   // sequencer 5: S400-S499 Robot3 FixtureCode reading
   STEP Robot3FixtrueScanStart:   // S400, max time T#10S, warning time T#7S
              N    "AutoProcessData".GripperCode_R3[1]:=''
              N    "AutoProcessData".GripperCode_R3[2]:=''
              N    "AutoProcessData".GripperCode_R3[3]:=''
              N    "AutoProcessData".GripperCode_R3[4]:=''
              N    "AutoProcessData".FixtureCode_A2[1]:=''
              N    "AutoProcessData".FixtureCode_A2[2]:=''
              N    "AutoProcessData".FixtureCode_A2[3]:=''
              N    "AutoProcessData".FixtureCode_A2[4]:=''
              N    "AutoProcessData".FixtureCode_A2[5]:=''
              N    "AutoProcessData".FixtureCode_A2[6]:=''
              N    "AutoProcessData".FixtureCode_A2[7]:=''
              N    "AutoProcessData".FixtureCode_A2[8]:=''
   END_STEP
   TRANSITION Trans400 FROM Robot3FixtrueScanStart TO Robot3CheckScanStatus   // T400
      := NOT "KukaRobot2_CtrlDB".sROBtoPLC.User.Cycle.DO297_MaintainInside;
   END_TRANSITION
   STEP AllScanFinish:   // S408, max time T#10S, warning time T#7S
   END_STEP
   TRANSITION Trans403 FROM AllScanFinish TO ProcessStart   // T403, jump
      := "AutoProcessData".GlobalData.Table1CodeOKFlag AND "AutoProcessData".GlobalData.Table2CodeOKFlag AND "AutoProcessData".GlobalData.Robot1GripperCodeOKFlag AND "AutoProcessData".GlobalData.Robot2GripperCodeOKFlag AND "AutoProcessData".GlobalData.Robot3GripperCodeOKFlag AND "AutoProcessData".GlobalData.Fixture1CodeOKFlag AND "AutoProcessData".GlobalData.Fixture2CodeOKFlag AND "ST10_RecipeDB".Recipe.Equal AND NOT "ChangeOver_DB".Global.ScanFixtureFlag AND NOT "ChangeOver_DB".Global.ChangeOverRequest;
   END_TRANSITION
   TRANSITION Trans420 FROM AllScanFinish TO ProcessStart   // T420, jump
      := ("ChangeOver_DB".Global.ChangeOverRequest OR "ChangeOver_DB".Global.ChangeOverSelected) AND NOT "ChangeOver_DB".Global.ChangeOverSelected;
   END_TRANSITION
   STEP DataMove_7:   // S279, max time T#10S, warning time T#7S
              N    "AutoProcessData".FixtureCode_A2[2]:="KeyenceSR1000Ctrl_807A1DB".sHMI.Status.CurrentCode
   END_STEP
   TRANSITION Trans336 FROM DataMove_7 TO WaitRobotScanPos3Reach_1   // T312
      := "AlwaysTRUE";
   END_TRANSITION
   STEP Robot3StartToMaintenance:   // S409, max time T#10S, warning time T#7S
   END_STEP
   TRANSITION Trans405 FROM Robot3StartToMaintenance TO Step712   // T405, jump
      := TRUE;
   END_TRANSITION
   STEP DataMove_8:   // S284, max time T#10S, warning time T#7S
              N    "AutoProcessData".FixtureCode_A2[1]:="KeyenceSR1000Ctrl_807A1DB".sHMI.Status.CurrentCode
   END_STEP
   TRANSITION Trans290 FROM DataMove_8 TO WaitRobotScanPos2Reach_1   // T301
      := "AlwaysTRUE";
   END_TRANSITION
   STEP RequestRobotScanFixture:   // S312, max time T#10S, warning time T#7S
              N    "AutoProcessControl".Fixture2Code.Robot3CodeReadReq
   END_STEP
   TRANSITION Trans609 FROM RequestRobotScanFixture TO WaitRobotScanPos1Reach_3   // T634
      := "KukaRobot3_CtrlDB".sROBtoPLC.User.Cycle.DO225_ScanPosInside;
   END_TRANSITION
   STEP "Start 1st reading_1":   // S289, max time T#10S, warning time T#7S
          S1  S    "KeyenceSR1000Ctrl_807A1DB".ioAutoTrigger
   END_STEP
   TRANSITION Trans284 FROM "Start 1st reading_1" TO "Wait reading complete_6"   // T283
      := NOT "KeyenceSR1000Ctrl_807A1DB".sHMI.Status.Ready;
   END_TRANSITION
   STEP "Check reader Ready_6":   // S290, max time T#10S, warning time T#7S
   END_STEP
   TRANSITION Trans280 FROM "Check reader Ready_6" TO "Start 1st reading_1"   // T297
      := "KeyenceSR1000Ctrl_807A1DB".sHMI.Status.Ready;
   END_TRANSITION
   STEP "Wait reading complete_6":   // S291, max time T#10S, warning time T#7S
   END_STEP
   TRANSITION ReadOK_8 FROM "Wait reading complete_6" TO DataMove_8   // T285
      := "KeyenceSR1000Ctrl_807A1DB".sHMI.Status.Complete;
   END_TRANSITION
   STEP WaitRobotScanPos1Reach_2:   // S367, max time T#10S, warning time T#7S
              N    "KukaRobot3_CtrlDB".sPLCtoROB.User.Cycle.DI230_ScanPos5Complete
   END_STEP
   TRANSITION Trans618 FROM WaitRobotScanPos1Reach_2 TO "Check reader Ready_23"   // T636
      := "KukaRobot3_CtrlDB".sROBtoPLC.User.Cycle.DO233_ScanPoseFinish;
   END_TRANSITION
   STEP WaitRobotScanPos5Reach_1:   // S368, max time T#10S, warning time T#7S
              N    "KukaRobot3_CtrlDB".sPLCtoROB.User.Cycle.DI229_ScanPos4Complete
   END_STEP
   TRANSITION Trans619 FROM WaitRobotScanPos5Reach_1 TO "Check reader Ready_7"   // T637
      := "KukaRobot3_CtrlDB".sROBtoPLC.User.Cycle.DO230_ScanPos5Reach;
   END_TRANSITION
   STEP WaitRobotScanPos2Reach_1:   // S369, max time T#10S, warning time T#7S
              N    "KukaRobot3_CtrlDB".sPLCtoROB.User.Cycle.DI226_ScanPos1Complete
   END_STEP
   TRANSITION Trans623 FROM WaitRobotScanPos2Reach_1 TO "Check reader Ready_18"   // T641
      := "KukaRobot3_CtrlDB".sROBtoPLC.User.Cycle.DO227_ScanPos2Reach;
   END_TRANSITION
   STEP WaitRobotScanPos4Reach_1:   // S370, max time T#10S, warning time T#7S
              N    "KukaRobot3_CtrlDB".sPLCtoROB.User.Cycle.DI228_ScanPos3Complete
   END_STEP
   TRANSITION Trans621 FROM WaitRobotScanPos4Reach_1 TO "Check reader Ready_8"   // T639
      := "KukaRobot3_CtrlDB".sROBtoPLC.User.Cycle.DO229_ScanPos4Reach;
   END_TRANSITION
   STEP "Start 5st reading_1":   // S292, max time T#10S, warning time T#7S
          S1  S    "KeyenceSR1000Ctrl_807A1DB".ioAutoTrigger
   END_STEP
   TRANSITION Trans307 FROM "Start 5st reading_1" TO "Wait reading complete_7"   // T314
      := NOT "KeyenceSR1000Ctrl_807A1DB".sHMI.Status.Ready;
   END_TRANSITION
   STEP "Check reader Ready_7":   // S293, max time T#10S, warning time T#7S
   END_STEP
   TRANSITION Trans308 FROM "Check reader Ready_7" TO "Start 5st reading_1"   // T327
      := "KeyenceSR1000Ctrl_807A1DB".sHMI.Status.Ready;
   END_TRANSITION
   STEP "Wait reading complete_7":   // S294, max time T#10S, warning time T#7S
   END_STEP
   TRANSITION ReadOK_18 FROM "Wait reading complete_7" TO DataMove_9   // T316
      := "KeyenceSR1000Ctrl_807A1DB".sHMI.Status.Complete;
   END_TRANSITION
   STEP "Wait reading complete_8":   // S301, max time T#10S, warning time T#7S
   END_STEP
   TRANSITION ReadOK_9 FROM "Wait reading complete_8" TO DataMove_18   // T302
      := "KeyenceSR1000Ctrl_807A1DB".sHMI.Status.Complete;
   END_TRANSITION
   STEP "Check reader Ready_8":   // S302, max time T#10S, warning time T#7S
   END_STEP
   TRANSITION Trans298 FROM "Check reader Ready_8" TO "Start 4st reading_1"   // T308
      := "KeyenceSR1000Ctrl_807A1DB".sHMI.Status.Ready;
   END_TRANSITION
   STEP DataMove_9:   // S309, max time T#10S, warning time T#7S
              N    "AutoProcessData".FixtureCode_A2[5]:="KeyenceSR1000Ctrl_807A1DB".sHMI.Status.CurrentCode
   END_STEP
   TRANSITION Trans303 FROM DataMove_9 TO WaitRobotScanPos1Reach_2   // T324
      := "AlwaysTRUE";
   END_TRANSITION
   STEP DataMove_18:   // S310, max time T#10S, warning time T#7S
              N    "AutoProcessData".FixtureCode_A2[4]:="KeyenceSR1000Ctrl_807A1DB".sHMI.Status.CurrentCode
   END_STEP
   TRANSITION Trans309 FROM DataMove_18 TO WaitRobotScanPos5Reach_1   // T309
      := "AlwaysTRUE";
   END_TRANSITION
   STEP "Start 4st reading_1":   // S313, max time T#10S, warning time T#7S
          S1  S    "KeyenceSR1000Ctrl_807A1DB".ioAutoTrigger
   END_STEP
   TRANSITION Trans310 FROM "Start 4st reading_1" TO "Wait reading complete_8"   // T304
      := NOT "KeyenceSR1000Ctrl_807A1DB".sHMI.Status.Ready;
   END_TRANSITION
   STEP "Check reader Ready_9":   // S314, max time T#10S, warning time T#7S
   END_STEP
   TRANSITION Trans311 FROM "Check reader Ready_9" TO "Start 3st reading_1"   // T305
      := "KeyenceSR1000Ctrl_807A1DB".sHMI.Status.Ready;
   END_TRANSITION
   STEP "Wait reading complete_9":   // S315, max time T#10S, warning time T#7S
   END_STEP
   TRANSITION ReadOK_19 FROM "Wait reading complete_9" TO DataMove_19   // T311
      := "KeyenceSR1000Ctrl_807A1DB".sHMI.Status.Complete;
   END_TRANSITION
   STEP WaitRobotScanPos3Reach_1:   // S377, max time T#10S, warning time T#7S
              N    "KukaRobot3_CtrlDB".sPLCtoROB.User.Cycle.DI227_ScanPos2Complete
   END_STEP
   TRANSITION Trans622 FROM WaitRobotScanPos3Reach_1 TO "Check reader Ready_9"   // T640
      := "KukaRobot3_CtrlDB".sROBtoPLC.User.Cycle.DO228_ScanPos3Reach;
   END_TRANSITION
   STEP "Check reader Ready_18":   // S318, max time T#10S, warning time T#7S
   END_STEP
   TRANSITION Trans288 FROM "Check reader Ready_18" TO "Start 2st reading_1"   // T291
      := "KeyenceSR1000Ctrl_807A1DB".sHMI.Status.Ready;
   END_TRANSITION
   STEP "Wait reading complete_18":   // S319, max time T#10S, warning time T#7S
   END_STEP
   TRANSITION ReadOK_7 FROM "Wait reading complete_18" TO DataMove_7   // T288
      := "KeyenceSR1000Ctrl_807A1DB".sHMI.Status.Complete;
   END_TRANSITION
   STEP DataMove_19:   // S320, max time T#10S, warning time T#7S
              N    "AutoProcessData".FixtureCode_A2[3]:="KeyenceSR1000Ctrl_807A1DB".sHMI.Status.CurrentCode
   END_STEP
   TRANSITION Trans312 FROM DataMove_19 TO WaitRobotScanPos4Reach_1   // T310
      := "AlwaysTRUE";
   END_TRANSITION
   STEP "Start 3st reading_1":   // S321, max time T#10S, warning time T#7S
          S1  S    "KeyenceSR1000Ctrl_807A1DB".ioAutoTrigger
   END_STEP
   TRANSITION Trans294 FROM "Start 3st reading_1" TO "Wait reading complete_9"   // T303
      := NOT "KeyenceSR1000Ctrl_807A1DB".sHMI.Status.Ready;
   END_TRANSITION
   STEP "Start 2st reading_1":   // S322, max time T#10S, warning time T#7S
          S1  S    "KeyenceSR1000Ctrl_807A1DB".ioAutoTrigger
   END_STEP
   TRANSITION Trans289 FROM "Start 2st reading_1" TO "Wait reading complete_18"   // T294
      := NOT "KeyenceSR1000Ctrl_807A1DB".sHMI.Status.Ready;
   END_TRANSITION
   STEP Robot3CheckScanResult:   // S323, max time T#10S, warning time T#7S
   END_STEP
   TRANSITION R3ScanOk FROM Robot3CheckScanResult TO AllScanFinish   // T357
      := "AutoProcessData".GlobalData.Fixture2CodeOKFlag AND "AutoProcessData".GlobalData.Robot3GripperCodeOKFlag;
   END_TRANSITION
   TRANSITION R3ScanNG FROM Robot3CheckScanResult TO Robot3StartToMaintenance   // T404
      := #Robot3CheckScanResult.T > t#2S;
   END_TRANSITION
   STEP WaitRobotScanPos1Reach_3:   // S324, max time T#10S, warning time T#7S
   END_STEP
   TRANSITION Trans610 FROM WaitRobotScanPos1Reach_3 TO "Check reader Ready_6"   // T642
      := "KukaRobot3_CtrlDB".sROBtoPLC.User.Cycle.DO226_ScanPos1Reach;
   END_TRANSITION
   STEP RequestRobotScan_1:   // S379, max time T#10S, warning time T#7S
              N    "AutoProcessControl".Robot_3.GripScanRequest
   END_STEP
   TRANSITION Trans639 FROM RequestRobotScan_1 TO WaitRobotScanGripPos1Reach_1   // T643
      := NOT "KukaRobot3_CtrlDB".sROBtoPLC.User.Cycle.DO225_ScanPosInside AND "KukaRobot3_CtrlDB".sROBtoPLC.User.Cycle.DO305_GripScanInside;
   END_TRANSITION
   STEP WaitRobotScanGripPos1Reach_1:   // S380, max time T#10S, warning time T#7S
   END_STEP
   TRANSITION Trans640 FROM WaitRobotScanGripPos1Reach_1 TO "Check reader Ready_19"   // T644
      := "KukaRobot3_CtrlDB".sROBtoPLC.User.Cycle.DO307_ScanPos1Reach;
   END_TRANSITION
   STEP "Check reader Ready_19":   // S381, max time T#10S, warning time T#7S
   END_STEP
   TRANSITION Trans641 FROM "Check reader Ready_19" TO "Start 10st reading_2"   // T645
      := "KeyenceSR1000Ctrl_803A1DB".oReady;
   END_TRANSITION
   STEP "Start 10st reading_2":   // S382, max time T#10S, warning time T#7S
          S1  S    "KeyenceSR1000Ctrl_803A1DB".ioAutoTrigger
   END_STEP
   TRANSITION Trans643 FROM "Start 10st reading_2" TO "Wait reading complete_19"   // T646
      := NOT "KeyenceSR1000Ctrl_803A1DB".sHMI.Status.Ready;
   END_TRANSITION
   STEP "Wait reading complete_19":   // S325, max time T#10S, warning time T#7S
   END_STEP
   TRANSITION ReadOK_20 FROM "Wait reading complete_19" TO DataMove_20   // T386
      := "KeyenceSR1000Ctrl_803A1DB".sHMI.Status.Complete;
   END_TRANSITION
   STEP DataMove_20:   // S326, max time T#10S, warning time T#7S
              N    "AutoProcessData".GripperCode_R3[1]:="KeyenceSR1000Ctrl_803A1DB".sHMI.Status.CurrentCode
   END_STEP
   TRANSITION Trans337 FROM DataMove_20 TO RobotScanGripPos1Comp_2   // T387
      := "AlwaysTRUE";
   END_TRANSITION
   STEP RobotScanGripPos1Comp_2:   // S327, max time T#10S, warning time T#7S
              R    "KukaRobot3_CtrlDB".sPLCtoROB.User.Cycle.DI307_ScanPartFinish
              N    "KukaRobot3_CtrlDB".sPLCtoROB.User.Cycle.DI306_ScanPartComplete
   END_STEP
   TRANSITION Trans338 FROM RobotScanGripPos1Comp_2 TO WaitRobotScanGripPos2Reach_2   // T388
      := NOT "KukaRobot3_CtrlDB".sROBtoPLC.User.Cycle.DO307_ScanPos1Reach;
   END_TRANSITION
   STEP WaitRobotScanGripPos2Reach_2:   // S328, max time T#10S, warning time T#7S
   END_STEP
   TRANSITION Trans339 FROM WaitRobotScanGripPos2Reach_2 TO "Check reader Ready_20"   // T389
      := "KukaRobot3_CtrlDB".sROBtoPLC.User.Cycle.DO308_ScanPos2Reach;
   END_TRANSITION
   STEP "Check reader Ready_20":   // S384, max time T#10S, warning time T#7S
   END_STEP
   TRANSITION Trans644 FROM "Check reader Ready_20" TO "Start 11st reading_6"   // T647
      := "KeyenceSR1000Ctrl_803A1DB".oReady;
   END_TRANSITION
   STEP "Start 11st reading_6":   // S387, max time T#10S, warning time T#7S
          S1  S    "KeyenceSR1000Ctrl_803A1DB".ioAutoTrigger
   END_STEP
   TRANSITION Trans645 FROM "Start 11st reading_6" TO "Wait reading complete_20"   // T648
      := NOT "KeyenceSR1000Ctrl_803A1DB".sHMI.Status.Ready;
   END_TRANSITION
   STEP "Wait reading complete_20":   // S390, max time T#10S, warning time T#7S
   END_STEP
   TRANSITION ReadOK_21 FROM "Wait reading complete_20" TO DataMove_21   // T390
      := "KeyenceSR1000Ctrl_803A1DB".sHMI.Status.Complete;
   END_TRANSITION
   STEP DataMove_21:   // S392, max time T#10S, warning time T#7S
              N    "AutoProcessData".GripperCode_R3[2]:="KeyenceSR1000Ctrl_803A1DB".sHMI.Status.CurrentCode
   END_STEP
   TRANSITION Trans340 FROM DataMove_21 TO RobotScanGripPos2Comp_2   // T391
      := "AlwaysTRUE";
   END_TRANSITION
   STEP RobotScanGripPos2Comp_2:   // S393, max time T#10S, warning time T#7S
              R    "KukaRobot3_CtrlDB".sPLCtoROB.User.Cycle.DI307_ScanPartFinish
              N    "KukaRobot3_CtrlDB".sPLCtoROB.User.Cycle.DI306_ScanPartComplete
   END_STEP
   TRANSITION Trans341 FROM RobotScanGripPos2Comp_2 TO WaitRobotScanGripPos3Reach_2   // T392
      := NOT "KukaRobot3_CtrlDB".sROBtoPLC.User.Cycle.DO308_ScanPos2Reach;
   END_TRANSITION
   STEP WaitRobotScanGripPos3Reach_2:   // S394, max time T#10S, warning time T#7S
   END_STEP
   TRANSITION Trans342 FROM WaitRobotScanGripPos3Reach_2 TO "Check reader Ready_21"   // T393
      := "KukaRobot3_CtrlDB".sROBtoPLC.User.Cycle.DO309_ScanPos3Reach;
   END_TRANSITION
   STEP "Check reader Ready_21":   // S395, max time T#10S, warning time T#7S
   END_STEP
   TRANSITION Trans646 FROM "Check reader Ready_21" TO "Start 11st reading_7"   // T649
      := "KeyenceSR1000Ctrl_803A1DB".oReady;
   END_TRANSITION
   STEP "Start 11st reading_7":   // S396, max time T#10S, warning time T#7S
          S1  S    "KeyenceSR1000Ctrl_803A1DB".ioAutoTrigger
   END_STEP
   TRANSITION Trans647 FROM "Start 11st reading_7" TO "Wait reading complete_21"   // T650
      := NOT "KeyenceSR1000Ctrl_803A1DB".sHMI.Status.Ready;
   END_TRANSITION
   STEP "Wait reading complete_21":   // S397, max time T#10S, warning time T#7S
   END_STEP
   TRANSITION ReadOK_22 FROM "Wait reading complete_21" TO DataMove_22   // T394
      := "KeyenceSR1000Ctrl_803A1DB".sHMI.Status.Complete;
   END_TRANSITION
   STEP DataMove_22:   // S398, max time T#10S, warning time T#7S
              N    "AutoProcessData".GripperCode_R3[3]:="KeyenceSR1000Ctrl_803A1DB".sHMI.Status.CurrentCode
   END_STEP
   TRANSITION Trans343 FROM DataMove_22 TO RobotScanGripPos3Comp_2   // T395
      := "AlwaysTRUE";
   END_TRANSITION
   STEP RobotScanGripPos3Comp_2:   // S399, max time T#10S, warning time T#7S
              R    "KukaRobot3_CtrlDB".sPLCtoROB.User.Cycle.DI307_ScanPartFinish
              N    "KukaRobot3_CtrlDB".sPLCtoROB.User.Cycle.DI306_ScanPartComplete
   END_STEP
   TRANSITION Trans344 FROM RobotScanGripPos3Comp_2 TO WaitRobotScanGripPos4Reach_2   // T396
      := NOT "KukaRobot3_CtrlDB".sROBtoPLC.User.Cycle.DO309_ScanPos3Reach;
   END_TRANSITION
   STEP WaitRobotScanGripPos4Reach_2:   // S401, max time T#10S, warning time T#7S
   END_STEP
   TRANSITION Trans345 FROM WaitRobotScanGripPos4Reach_2 TO "Check reader Ready_22"   // T397
      := "KukaRobot3_CtrlDB".sROBtoPLC.User.Cycle.DO310_ScanPos4Reach;
   END_TRANSITION
   STEP "Check reader Ready_22":   // S402, max time T#10S, warning time T#7S
   END_STEP
   TRANSITION Trans648 FROM "Check reader Ready_22" TO "Start 11st reading_8"   // T651
      := "KeyenceSR1000Ctrl_803A1DB".oReady;
   END_TRANSITION
   STEP "Start 11st reading_8":   // S403, max time T#10S, warning time T#7S
          S1  S    "KeyenceSR1000Ctrl_803A1DB".ioAutoTrigger
   END_STEP
   TRANSITION Trans649 FROM "Start 11st reading_8" TO "Wait reading complete_22"   // T652
      := NOT "KeyenceSR1000Ctrl_803A1DB".sHMI.Status.Ready;
   END_TRANSITION
   STEP "Wait reading complete_22":   // S404, max time T#10S, warning time T#7S
   END_STEP
   TRANSITION ReadOK_23 FROM "Wait reading complete_22" TO DataMove_23   // T398
      := "KeyenceSR1000Ctrl_803A1DB".sHMI.Status.Complete;
   END_TRANSITION
   STEP DataMove_23:   // S405, max time T#10S, warning time T#7S
              N    "AutoProcessData".GripperCode_R3[4]:="KeyenceSR1000Ctrl_803A1DB".sHMI.Status.CurrentCode
   END_STEP
   TRANSITION Trans346 FROM DataMove_23 TO RobotScanGripPos4Comp_2   // T399
      := "AlwaysTRUE";
   END_TRANSITION
   STEP RobotScanGripPos4Comp_2:   // S406, max time T#10S, warning time T#7S
              N    "KukaRobot3_CtrlDB".sPLCtoROB.User.Cycle.DI307_ScanPartFinish
              N    "KukaRobot3_CtrlDB".sPLCtoROB.User.Cycle.DI306_ScanPartComplete
   END_STEP
   TRANSITION Trans347 FROM RobotScanGripPos4Comp_2 TO WaitRobot2ScanFinishAndInHome   // T401
      := "KukaRobot3_CtrlDB".sROBtoPLC.User.Cycle.DO306_GripScanFinish;
   END_TRANSITION
   STEP WaitRobot2ScanFinishAndInHome:   // S407, max time T#10S, warning time T#7S
   END_STEP
   TRANSITION Trans371 FROM WaitRobot2ScanFinishAndInHome TO RequestRobotScanFixture   // T402
      := "Robot_DB".Robot_2.GripCompareCodeOK AND "KukaRobot2_CtrlDB".sROBtoPLC.Sys.SO.IN_HOME AND "KukaRobot2_CtrlDB".sROBtoPLC.User.Home.DO181_Robot3Area;
   END_TRANSITION
   STEP Robot3CheckScanStatus:   // S411, max time T#10S, warning time T#7S
   END_STEP
   TRANSITION GripScanNG1 FROM Robot3CheckScanStatus TO RequestRobotScan_1   // T406
      := NOT "AutoProcessData".GlobalData.Robot3GripperCodeOKFlag;
   END_TRANSITION
   TRANSITION GripScanOK FROM Robot3CheckScanStatus TO RequestRobotScanFixture   // T407
      := "AutoProcessData".GlobalData.Robot3GripperCodeOKFlag AND NOT "AutoProcessData".GlobalData.Fixture2CodeOKFlag;
   END_TRANSITION
   TRANSITION ALLScanOk FROM Robot3CheckScanStatus TO Robot3CheckScanResult   // T712
      := "AutoProcessData".GlobalData.Robot3GripperCodeOKFlag AND "AutoProcessData".GlobalData.Fixture2CodeOKFlag;
   END_TRANSITION
   STEP WaitRobotScanPos1Reach_4:   // S412, max time T#10S, warning time T#7S
   END_STEP
   TRANSITION Trans624 FROM WaitRobotScanPos1Reach_4 TO Robot3CheckScanResult   // T653
      := TRUE;
   END_TRANSITION
   STEP "Start 5st reading_2":   // S298, max time T#10S, warning time T#7S
   END_STEP
   TRANSITION Trans349 FROM "Start 5st reading_2" TO "Wait reading complete_23"   // T318
      := TRUE;
   END_TRANSITION
   STEP "Check reader Ready_23":   // S349, max time T#10S, warning time T#7S
   END_STEP
   TRANSITION Trans350 FROM "Check reader Ready_23" TO "Start 5st reading_2"   // T330
      := TRUE;
   END_TRANSITION
   STEP "Wait reading complete_23":   // S413, max time T#10S, warning time T#7S
   END_STEP
   TRANSITION ReadOK_24 FROM "Wait reading complete_23" TO DataMove_24   // T320
      := TRUE;
   END_TRANSITION
   STEP DataMove_24:   // S414, max time T#10S, warning time T#7S
   END_STEP
   TRANSITION Trans348 FROM DataMove_24 TO WaitRobotScanPos1Reach_4   // T328
      := "AlwaysTRUE";
   END_TRANSITION

   // sequencer 6: S700-S710 Robot1_Maintenance Pos
   STEP MaintenanceProcess:   // S700, max time T#10S, warning time T#7S
   END_STEP
   TRANSITION Trans625 FROM MaintenanceProcess TO ReqRobotToMantenPos   // T700
      := "KukaRobot2_CtrlDB".sROBtoPLC.User.Cycle.DO298_MaintainFinish OR "KukaRobot2_CtrlDB".sROBtoPLC.Sys.SO.IN_HOME;
   END_TRANSITION
   STEP ReqRobotToMantenPos:   // S701, max time T#10S, warning time T#7S
              N    "ChangeOver_DB".Robot_1.Req_RobotToMaintenancePos
   END_STEP
   TRANSITION Trans626 FROM ReqRobotToMantenPos TO WaitR1MaintenPosFinsh   // T701
      := "KukaRobot1_CtrlDB".sROBtoPLC.User.Cycle.DO297_MaintainInside;
   END_TRANSITION
   STEP WaitR1MaintenPosFinsh:   // S702, max time T#10S, warning time T#7S
   END_STEP
   TRANSITION Trans627 FROM WaitR1MaintenPosFinsh TO Robot2ToMaintenance   // T702
      := "KukaRobot1_CtrlDB".sROBtoPLC.User.Cycle.DO298_MaintainFinish;
   END_TRANSITION
   STEP Robot2ToMaintenance:   // S704, max time T#10S, warning time T#7S
   END_STEP
   TRANSITION Trans650 FROM Robot2ToMaintenance TO Step720   // T704, jump
      := ("KukaRobot1_CtrlDB".sROBtoPLC.User.Cycle.DO298_MaintainFinish OR "KukaRobot1_CtrlDB".sROBtoPLC.Sys.SO.IN_HOME) AND ("KukaRobot3_CtrlDB".sROBtoPLC.User.Cycle.DO301_HomeFinish OR "KukaRobot3_CtrlDB".sROBtoPLC.Sys.SO.IN_HOME) AND NOT "KukaRobot3_CtrlDB".sROBtoPLC.User.Cycle.DO225_ScanPosInside AND NOT "AutoProcessData".GlobalData.Robot2GripperCodeOKFlag;
   END_TRANSITION

   // sequencer 7: S720-S730 Robot2_Maintenance Pos
   STEP Step720:   // S720, max time T#10S, warning time T#7S
   END_STEP
   TRANSITION Trans720 FROM Step720 TO MaintenanceProcess_1   // T720
      := TRUE;
   END_TRANSITION
   STEP MaintenanceProcess_1:   // S706, max time T#10S, warning time T#7S
   END_STEP
   TRANSITION Trans655 FROM MaintenanceProcess_1 TO ReqRobotToMantenPos_1   // T706
      := ("KukaRobot3_CtrlDB".sROBtoPLC.User.Cycle.DO298_MaintainFinish OR "KukaRobot3_CtrlDB".sROBtoPLC.Sys.SO.IN_HOME) AND NOT "KukaRobot3_CtrlDB".sROBtoPLC.User.Cycle.DO225_ScanPosInside;
   END_TRANSITION
   STEP ReqRobotToMantenPos_1:   // S707, max time T#10S, warning time T#7S
              N    "ChangeOver_DB".Robot_2.Req_RobotToMaintenancePos
   END_STEP
   TRANSITION Trans656 FROM ReqRobotToMantenPos_1 TO WaitR1MaintenPosFinsh_1   // T707
      := "KukaRobot2_CtrlDB".sROBtoPLC.User.Cycle.DO297_MaintainInside;
   END_TRANSITION
   STEP WaitR1MaintenPosFinsh_1:   // S708, max time T#10S, warning time T#7S
   END_STEP
   TRANSITION Trans657 FROM WaitR1MaintenPosFinsh_1 TO Robot3ToMaintenance   // T708
      := "KukaRobot2_CtrlDB".sROBtoPLC.User.Cycle.DO298_MaintainFinish;
   END_TRANSITION
   STEP Robot3ToMaintenance:   // S710, max time T#10S, warning time T#7S
   END_STEP
   TRANSITION Trans659 FROM Robot3ToMaintenance TO Step712   // T710, jump
      := ("KukaRobot2_CtrlDB".sROBtoPLC.User.Cycle.DO298_MaintainFinish OR "KukaRobot2_CtrlDB".sROBtoPLC.Sys.SO.IN_HOME) AND NOT "KukaRobot2_CtrlDB".sROBtoPLC.User.Cycle.DO249_ScanNGPutInside AND NOT "KukaRobot2_CtrlDB".sROBtoPLC.User.Cycle.DO253_GlueNGPutInside AND NOT "KukaRobot2_CtrlDB".sROBtoPLC.User.Cycle.DO273_PressPutPart1Inside AND NOT "AutoProcessData".GlobalData.Robot3GripperCodeOKFlag AND NOT "AutoProcessData".GlobalData.Fixture2CodeOKFlag;
   END_TRANSITION

   // sequencer 8: S740-S750 Robot3_Maintenance Pos
   STEP Step712:   // S740, max time T#10S, warning time T#7S
   END_STEP
   TRANSITION Trans740 FROM Step712 TO MaintenanceProcess_2   // T740
      := TRUE;
   END_TRANSITION
   STEP MaintenanceProcess_2:   // S713, max time T#10S, warning time T#7S
   END_STEP
   TRANSITION Trans661 FROM MaintenanceProcess_2 TO ReqRobotToMantenPos_2   // T713
      := TRUE;
   END_TRANSITION
   STEP ReqRobotToMantenPos_2:   // S714, max time T#10S, warning time T#7S
              N    "ChangeOver_DB".Robot_3.Req_RobotToMaintenancePos
   END_STEP
   TRANSITION Trans662 FROM ReqRobotToMantenPos_2 TO WaitR1MaintenPosFinsh_2   // T714
      := "KukaRobot3_CtrlDB".sROBtoPLC.User.Cycle.DO297_MaintainInside;
   END_TRANSITION
   STEP WaitR1MaintenPosFinsh_2:   // S715, max time T#10S, warning time T#7S
   END_STEP
   TRANSITION Trans663 FROM WaitR1MaintenPosFinsh_2 TO CheckStationEmpty   // T715
      := "KukaRobot3_CtrlDB".sROBtoPLC.User.Cycle.DO298_MaintainFinish;
   END_TRANSITION
   STEP CycleEnd_2:   // S716, max time T#10S, warning time T#7S
              R    "ChangeOver_DB".Global.ChangeOverRequest
   END_STEP
   TRANSITION Trans664 FROM CycleEnd_2 TO END   // T716
      := "AlwaysFALSE";
   END_TRANSITION
   STEP CheckStationEmpty:   // S416, max time T#10S, warning time T#7S
   END_STEP
   TRANSITION Trans413 FROM CheckStationEmpty TO CheckTypeChenge   // T413
      := "ChangeOver_DB".Global.Station_empty AND "AutoProcessControl".Global.ALL_BeltPalletEmptyFinish;
   END_TRANSITION
   STEP CheckTypeChenge:   // S418, max time T#10S, warning time T#7S
   END_STEP
   TRANSITION ChengeOk FROM CheckTypeChenge TO TypeCheckOk   // T415
      := "ST10_RecipeDB".Recipe.Equal AND ("ST10_RecipeDB".Recipe.RecordName <> '');
   END_TRANSITION
   TRANSITION TypeChange FROM CheckTypeChenge TO CheckTypeTrigger   // T417
      := NOT "ST10_RecipeDB".Recipe.Equal AND "ChangeOver_DB".Global.ChangeOverSelected AND "ChangeOver_DB".Global.ChangeOverRequest;
   END_TRANSITION
   STEP TypeCheckOk:   // S419, max time T#10S, warning time T#7S
   END_STEP
   TRANSITION Trans416 FROM TypeCheckOk TO CycleEnd_2   // T416
      := TRUE;
   END_TRANSITION
   STEP CheckTypeTrigger:   // S420, max time T#10S, warning time T#7S
              N    "ChangeOver_DB".Global.ChangeOverActive
   END_STEP
   TRANSITION Trans418 FROM CheckTypeTrigger TO ResetChangeOverReq   // T418
      := "ST10_RecipeDB".Recipe.Equal AND ("ST10_RecipeDB".Recipe.RecordName <> '') AND NOT "ChangeOver_DB".Global.ChangeOverSelected;
   END_TRANSITION
   STEP ResetChangeOverReq:   // S421, max time T#10S, warning time T#7S
              R    "ChangeOver_DB".Global.ChangeOverRequest
   END_STEP
   TRANSITION Trans419 FROM ResetChangeOverReq TO CycleEnd_2   // T419
      := NOT "ChangeOver_DB".Global.ChangeOverSelected AND NOT "ChangeOver_DB".Global.ChangeOverRequest;
   END_TRANSITION

   // permanent post-instructions
   NETWORK 1
      #ioPM_Inface.StepNum := #RT_DATA.S_DISPLAY;
   NETWORK 2
      IF #iSysInface.Reset THEN #AlarmID := 0; END_IF;
   NETWORK 3
      #TON[10].TON(IN := #工件放行中, PT := T#0.5S);
      IF #TON[10].Q THEN #工件放行中 := FALSE; END_IF;
END_FUNCTION_BLOCK

FUNCTION_BLOCK "ST10_Flow7_CGlueing"   // FB1077, GRAPH
// stored: AcknowledgeErrorsRequired false, AutoNumber false, GraphVersion 6.0, InitialValuesAcquisition false, SetENOAutomatically false
   // inherited from GRAPH_BASE
   VAR_INPUT
      iSysInface : "RCS_SysComInterface_V1";
   END_VAR
   VAR_IN_OUT
      ioPM_Inface : "RCS_PMInterface_V1";
      ioStatus : Int;
   END_VAR
   VAR
      sCtrlMode { S7_SetPoint := 'True'} : "SysFlowCtrlGraph";
      sUpdMES_Data : Bool;   // 更新MES数据
      工件放行中 : Bool;
      前站站号 { ExternalAccessible := 'False'; ExternalVisible := 'False'; ExternalWritable := 'False'} : UInt;
      本站站号 { ExternalAccessible := 'False'; ExternalVisible := 'False'; ExternalWritable := 'False'} : UInt;
      弹窗Temp : Array[1..10] of Int;
      AlarmID : Int;
      TON { S7_SetPoint := 'True'} : Array[0..10] of TON_TIME;
      TOF { S7_SetPoint := 'True'} : Array[0..10] of TOF_TIME;
      sUP { S7_SetPoint := 'True'} : Array[0..10] of Bool;
      更新RFID完成 : Bool;
   END_VAR
   VAR_TEMP
      Tempresult : USInt;
      本站站号乘10 : UInt;
   END_VAR
   VAR CONSTANT
      Z_Axis : Int := 1;
      Y_axis : Int := 3;
      X_Axis : Int := 2;
   END_VAR
   // // TON[0] : 托盘流入1托盘到位传感器 / iA-Rotating product Check
   // // TON[1] : 托盘流入1托盘到位传感器
   // // TON[2] : 托盘流入1产品有无传感器
   // // TON[3] : 托盘流入1产品有无传感器
   // // TON[4] : 托盘流入1姿态检测光电2
   // // TON[5] : 托盘流入1姿态检测光电3
   // // TON[0].Q : 托盘流入1托盘到位 / iA-Rotating product Check
   // // TON[1].Q : 托盘流入1托盘无
   // // TON[2].Q : 托盘流入1有产品
   // // TON[3].Q : 托盘流入1无产品
   // // TON[4].Q : 托盘流入1姿态检测光电2
   // // TON[5].Q : 托盘流入1姿态检测光电3
   // // TOF[1] : iA-Rotating product Check
BEGIN
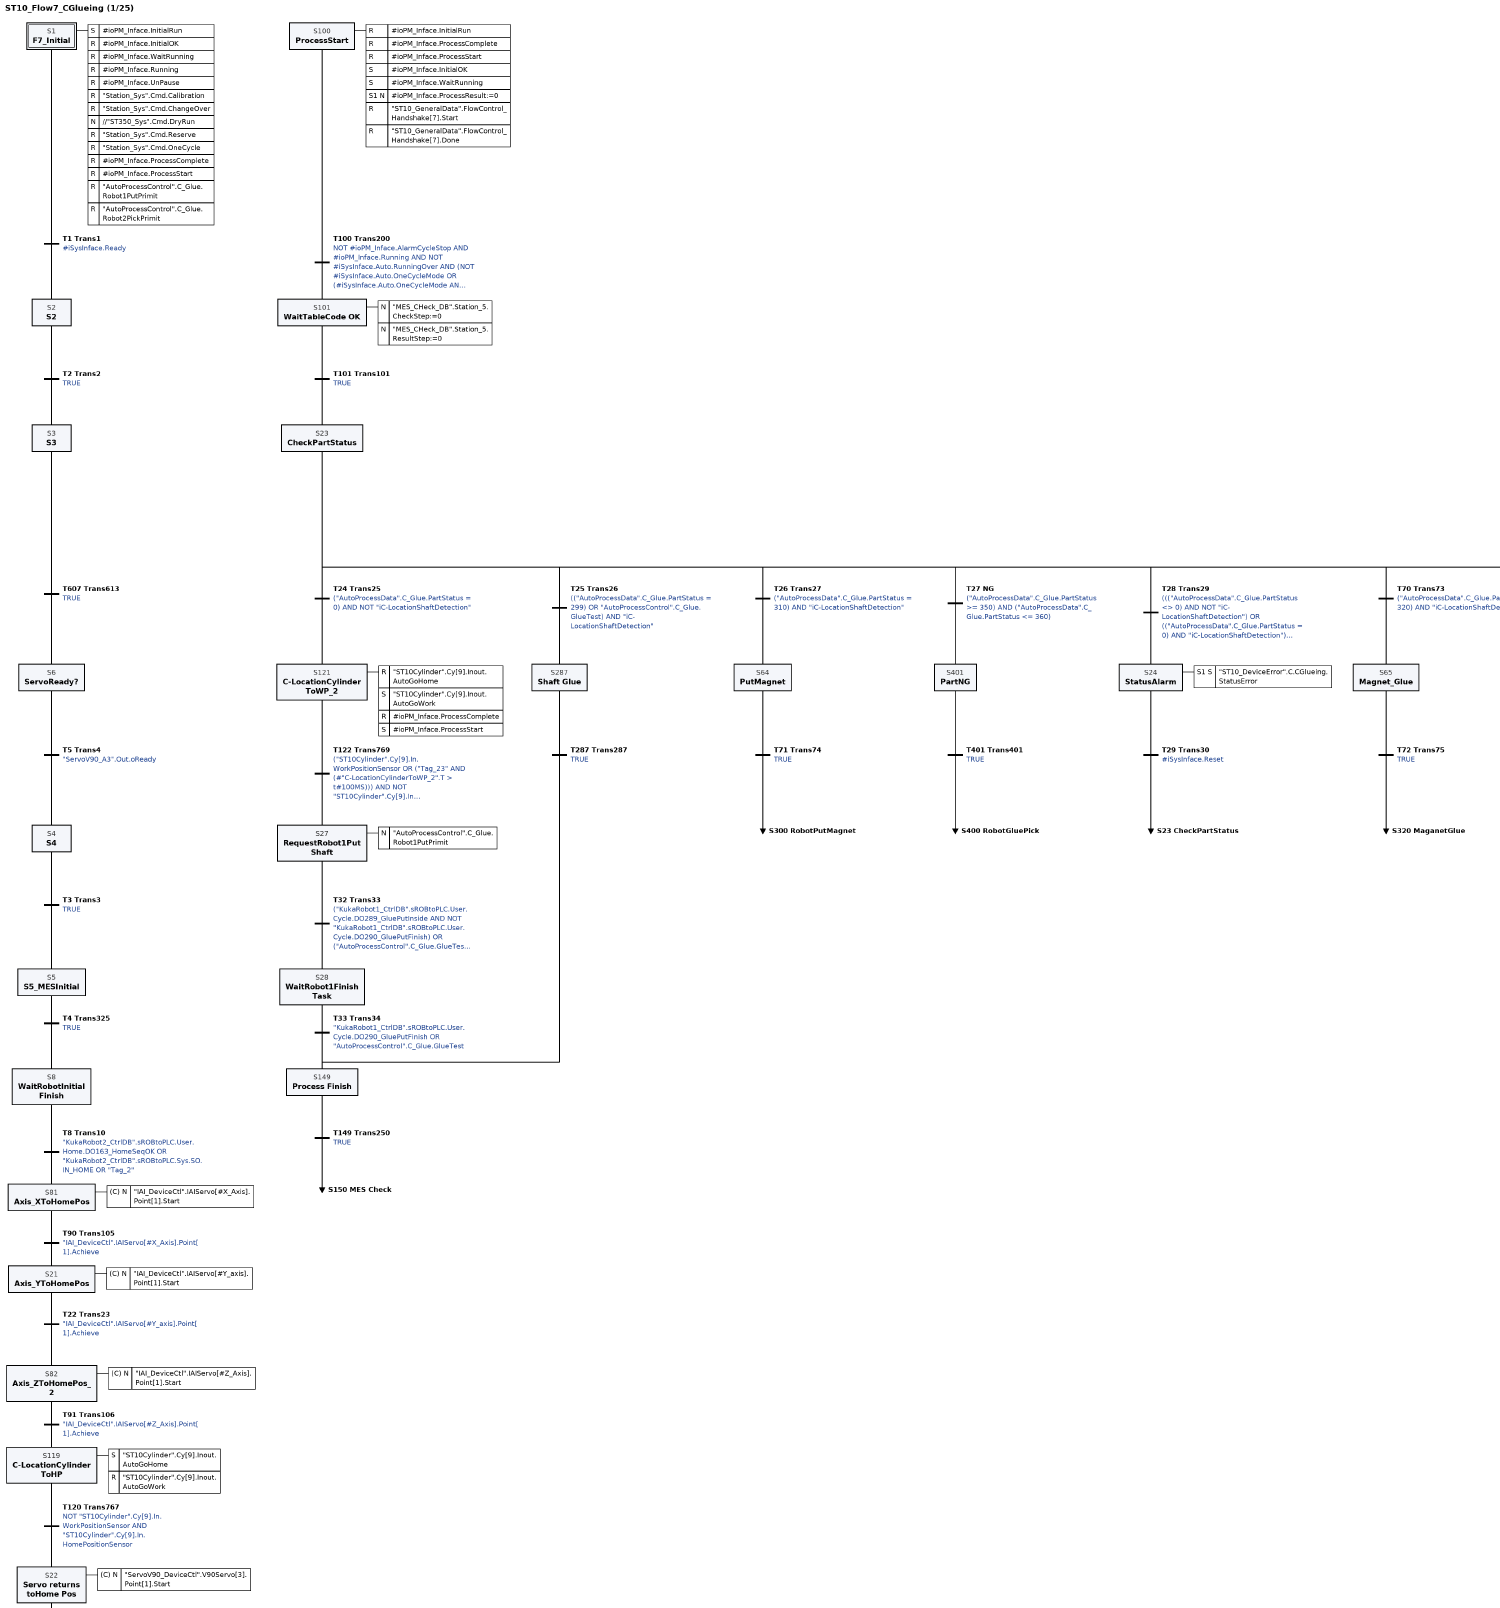
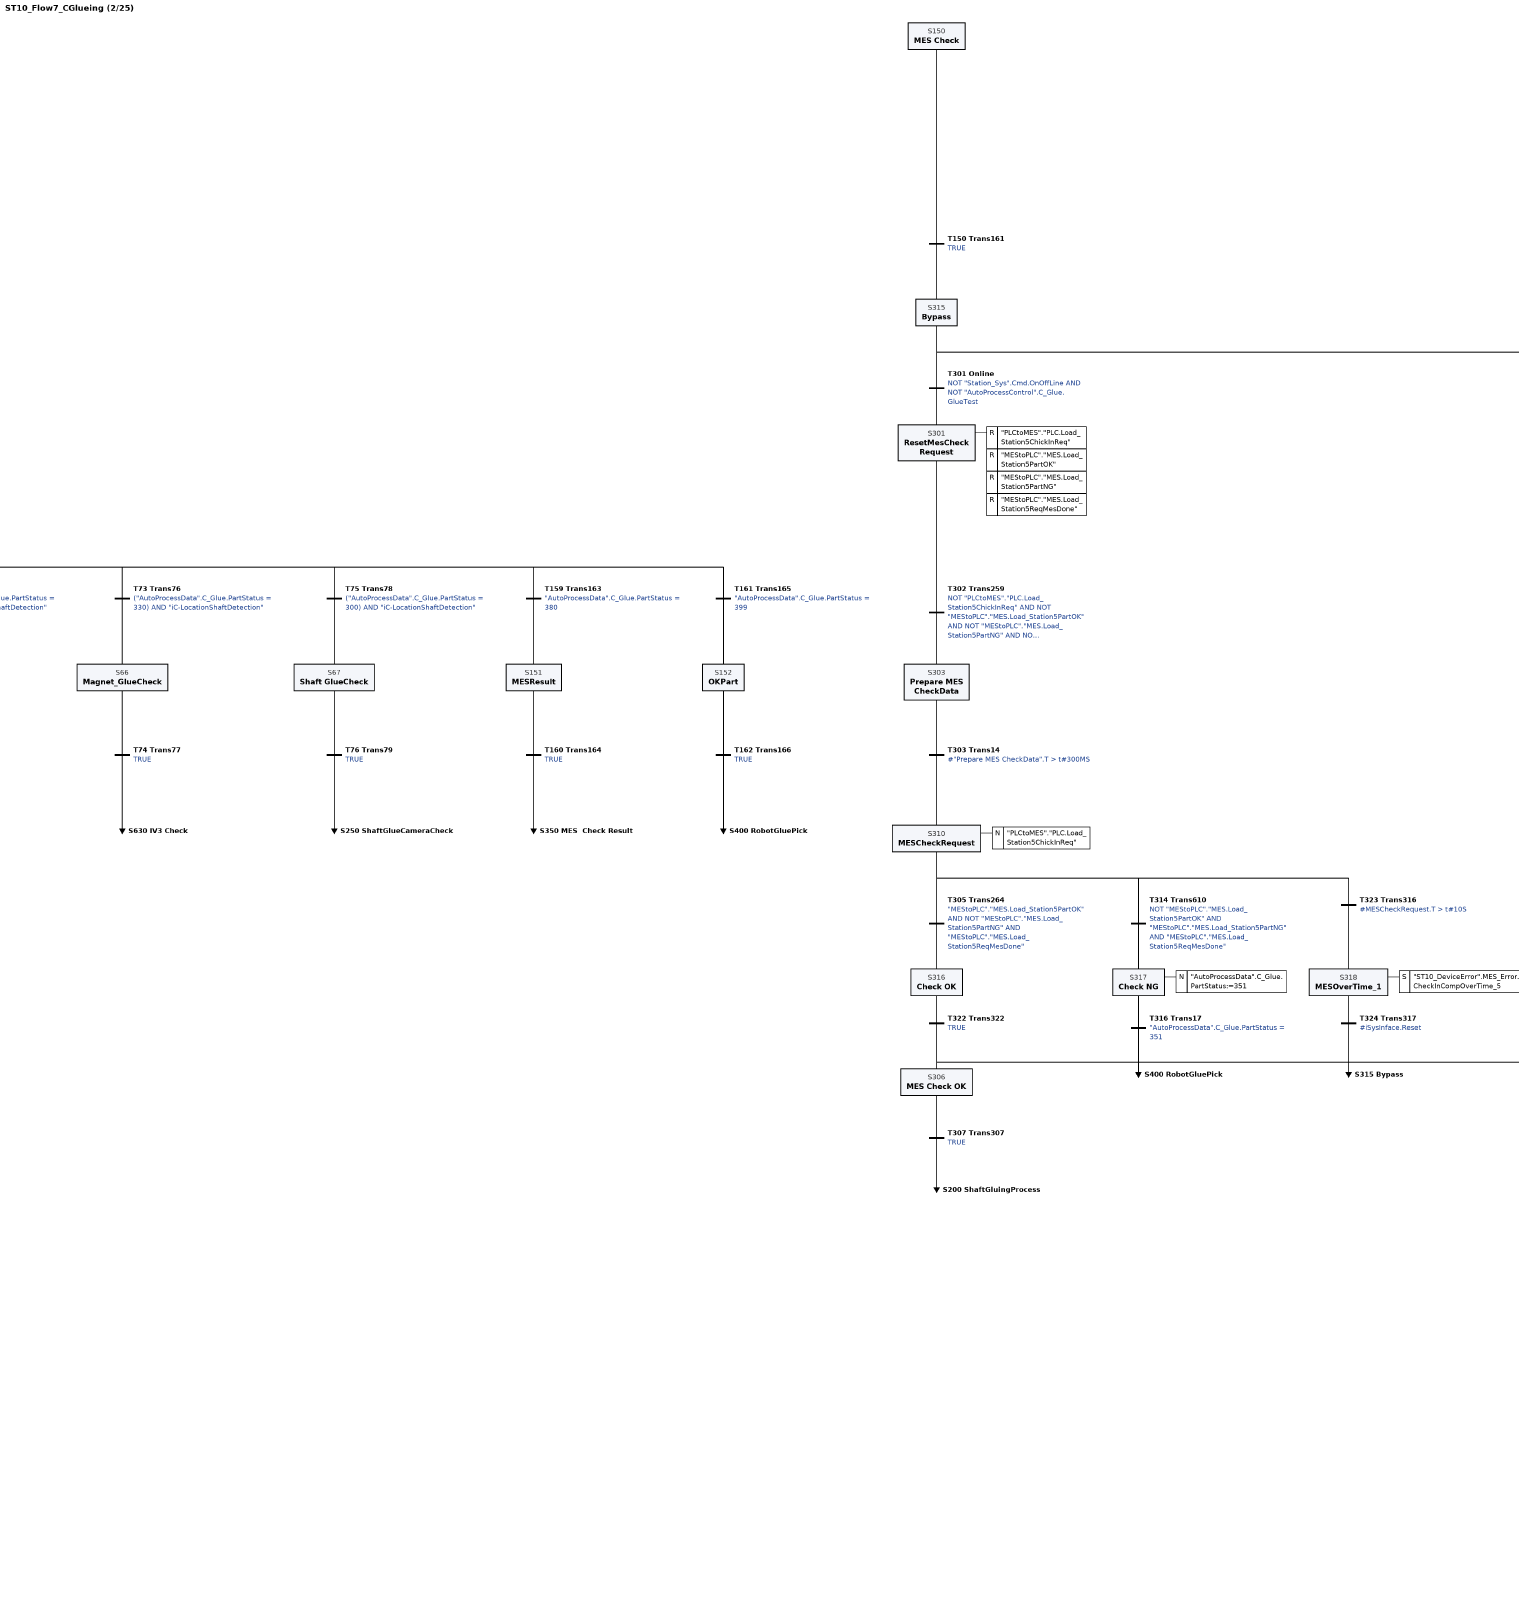
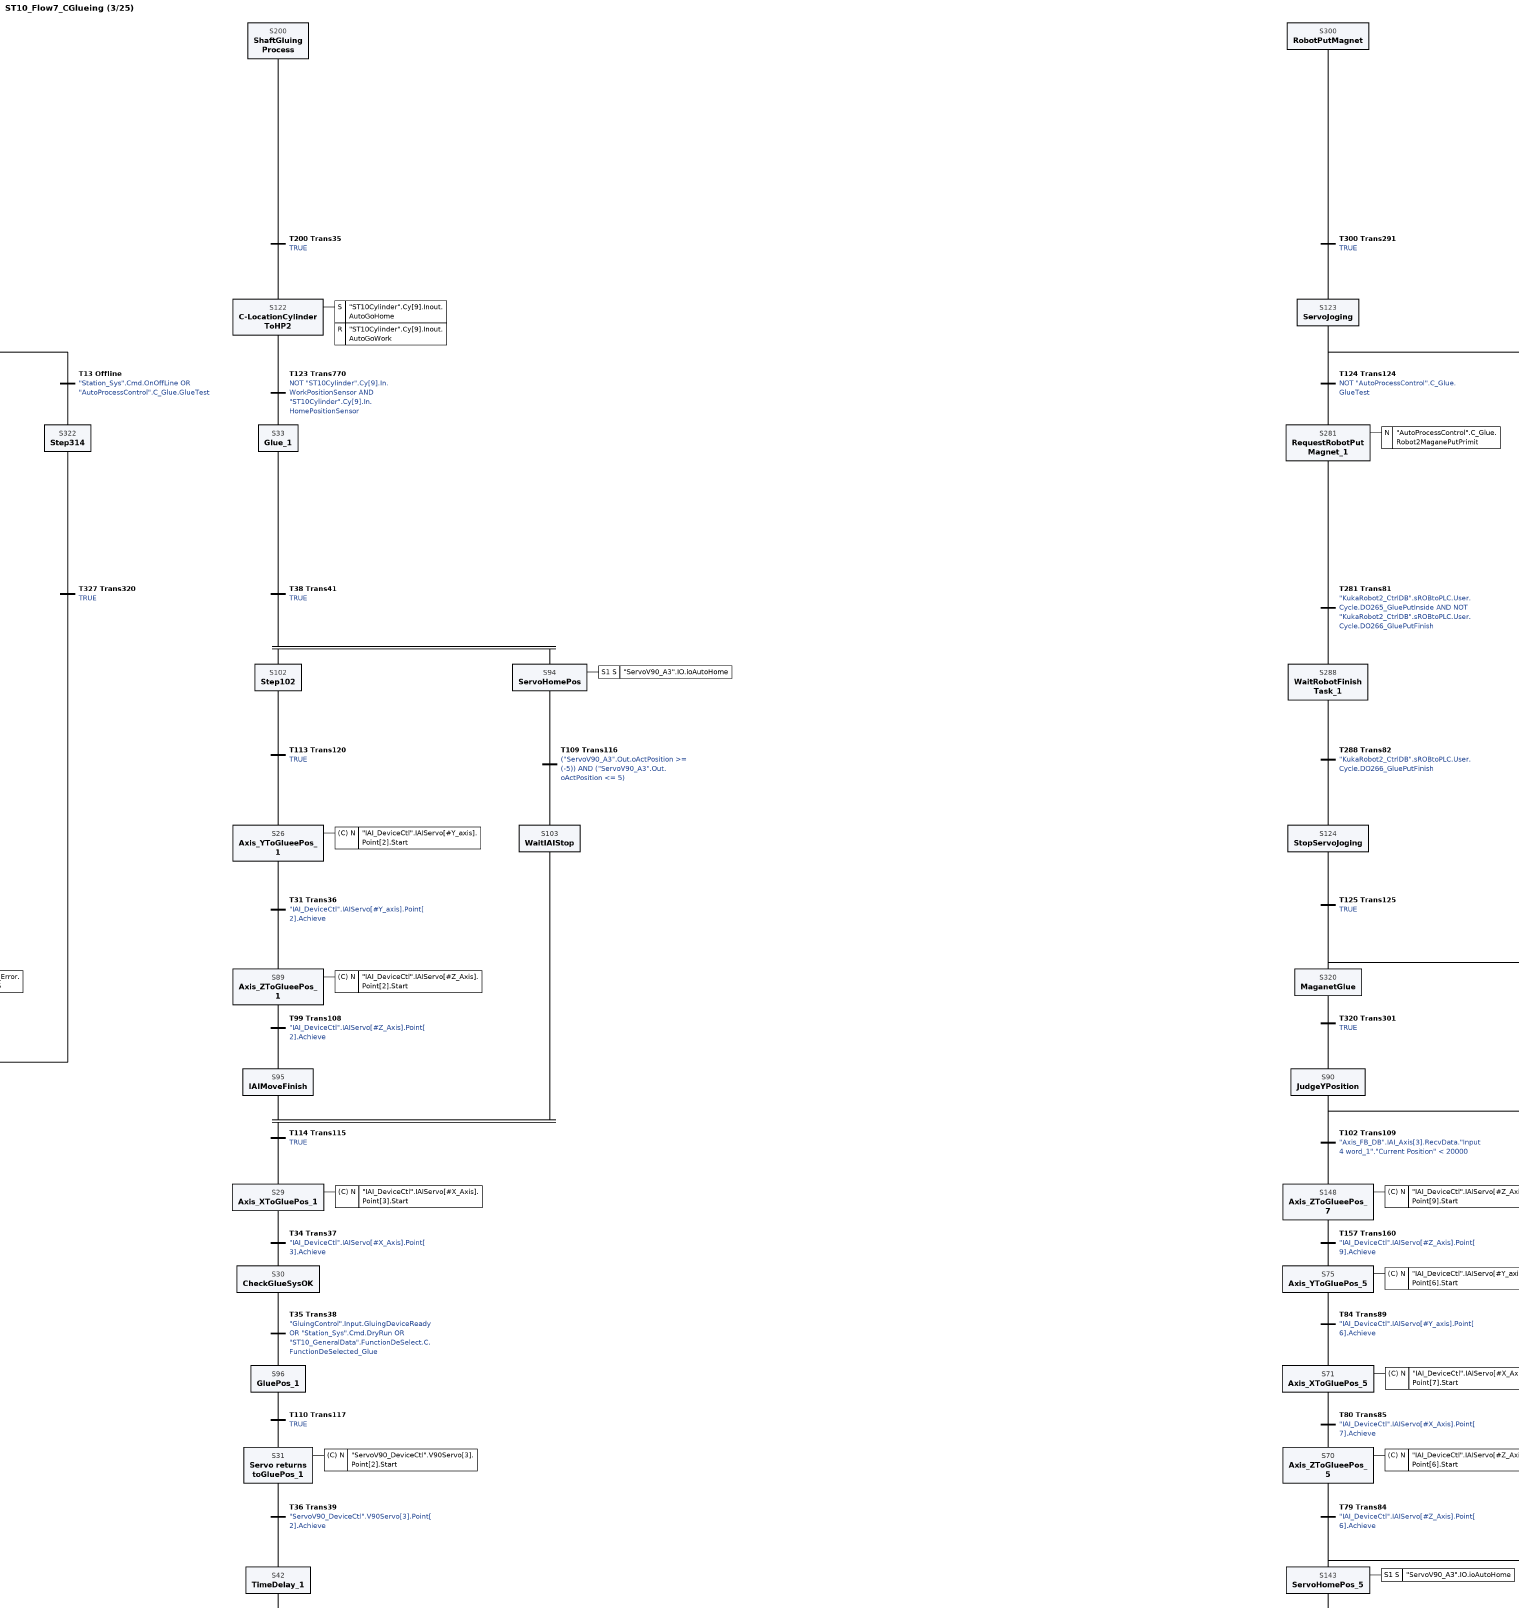
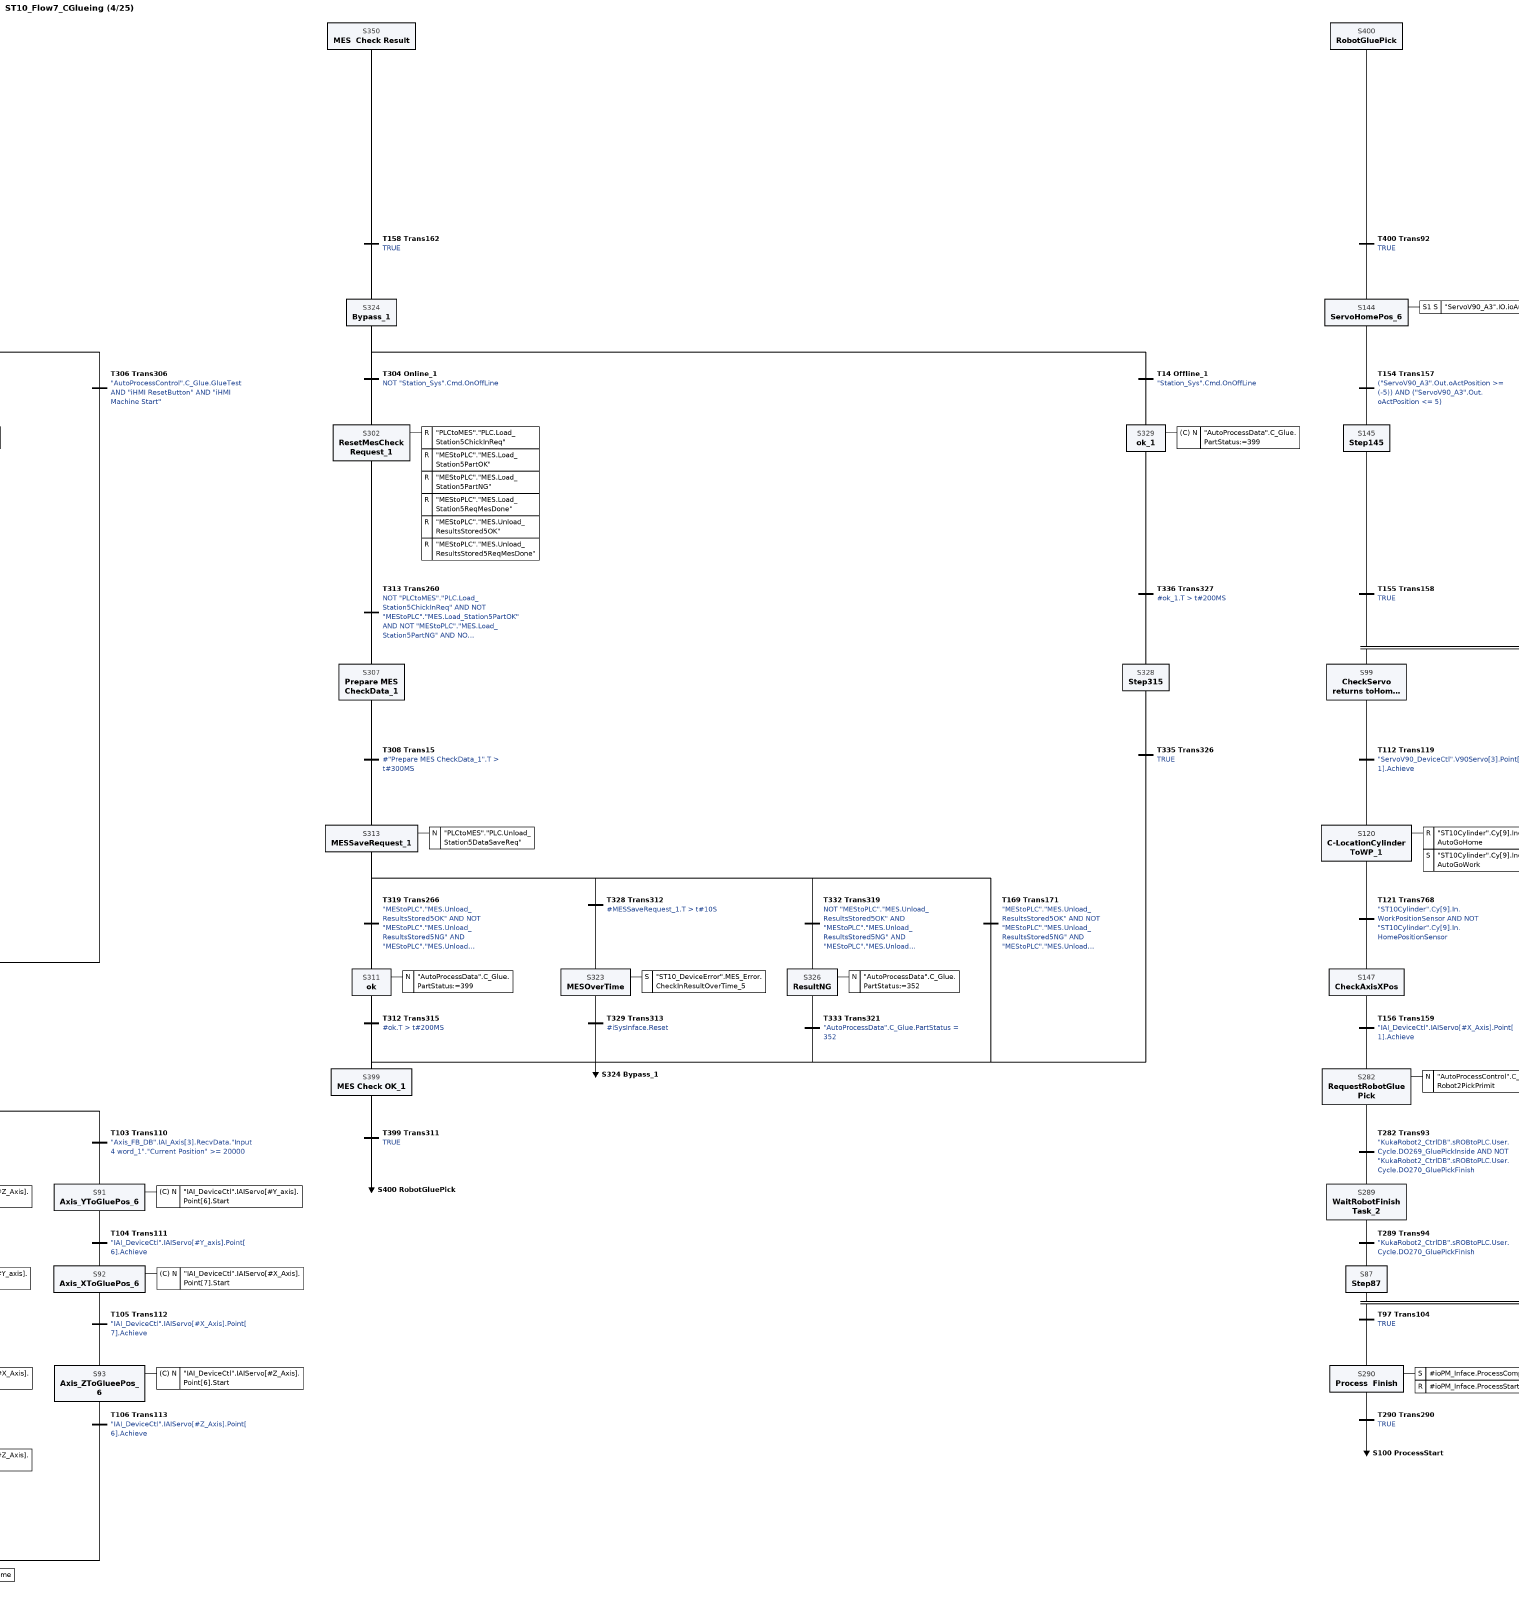
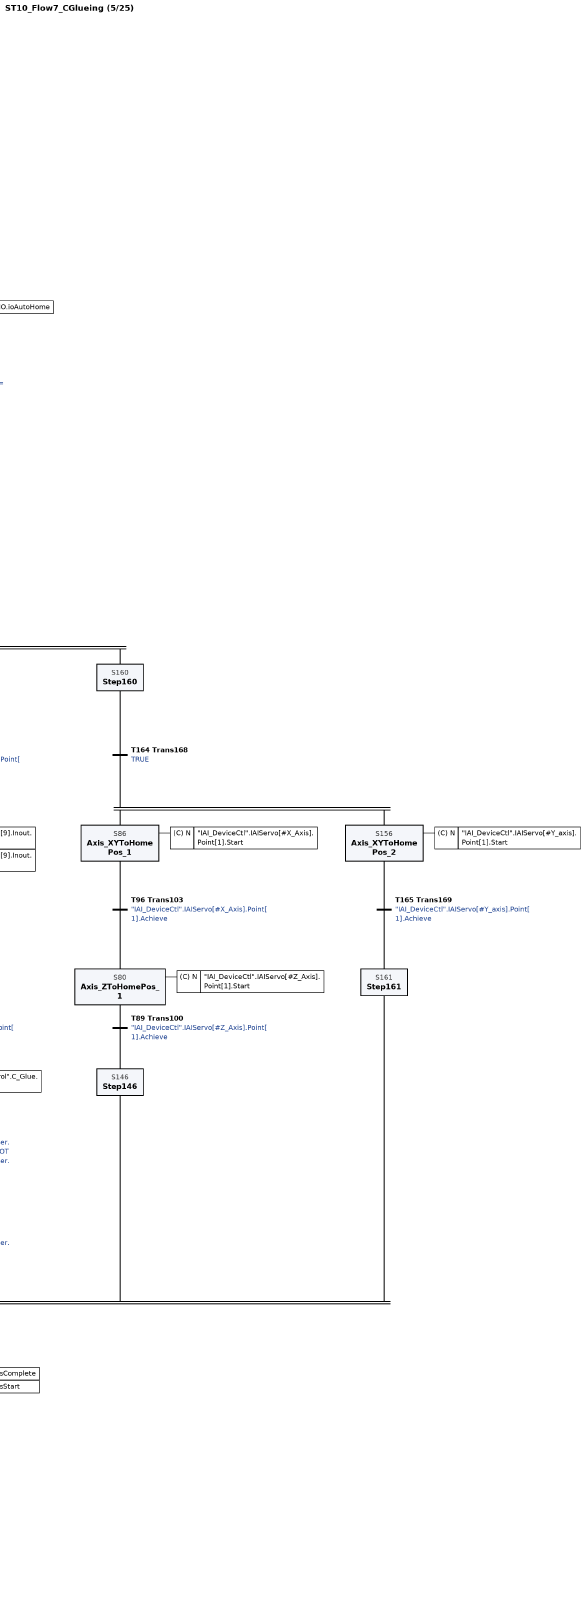
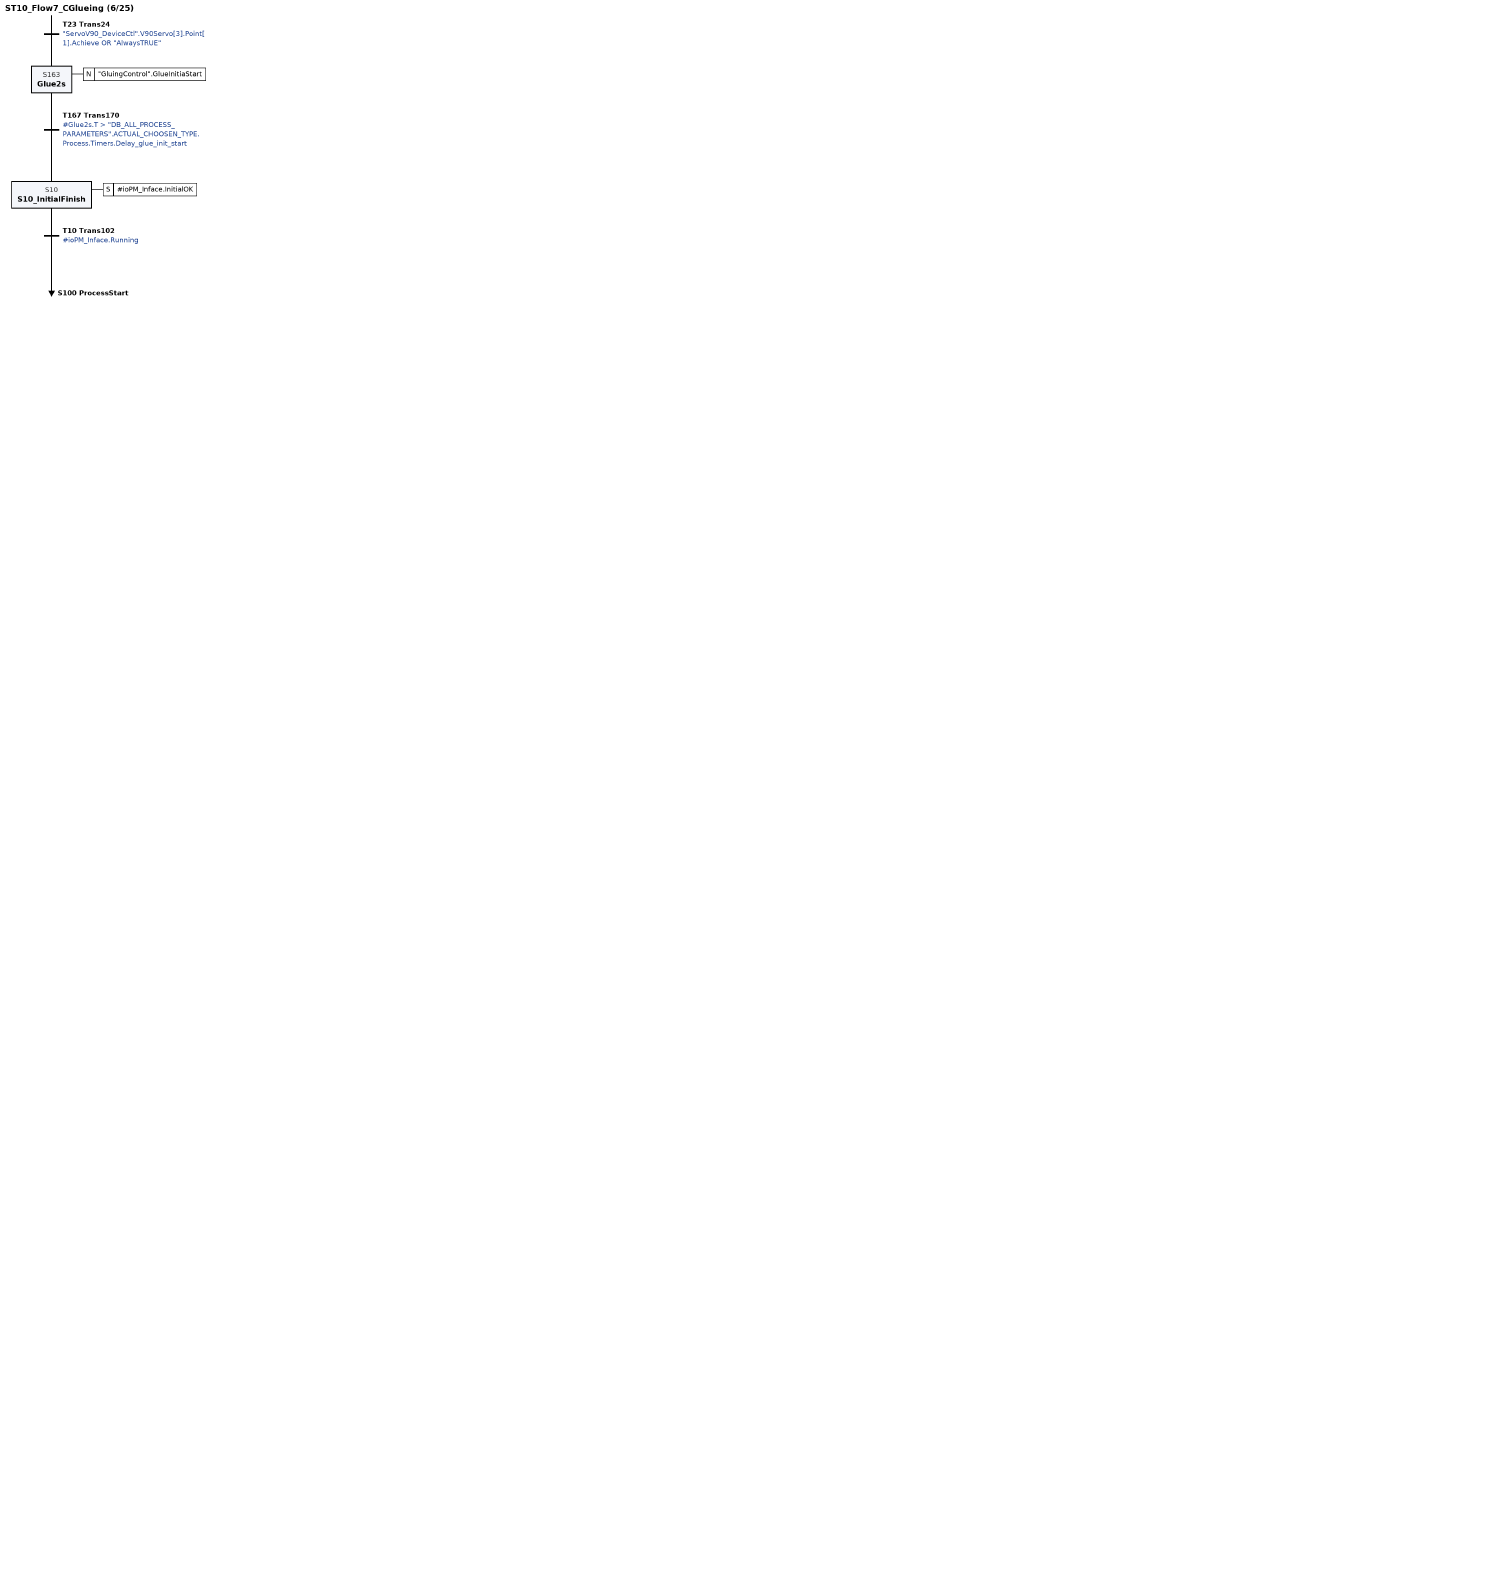
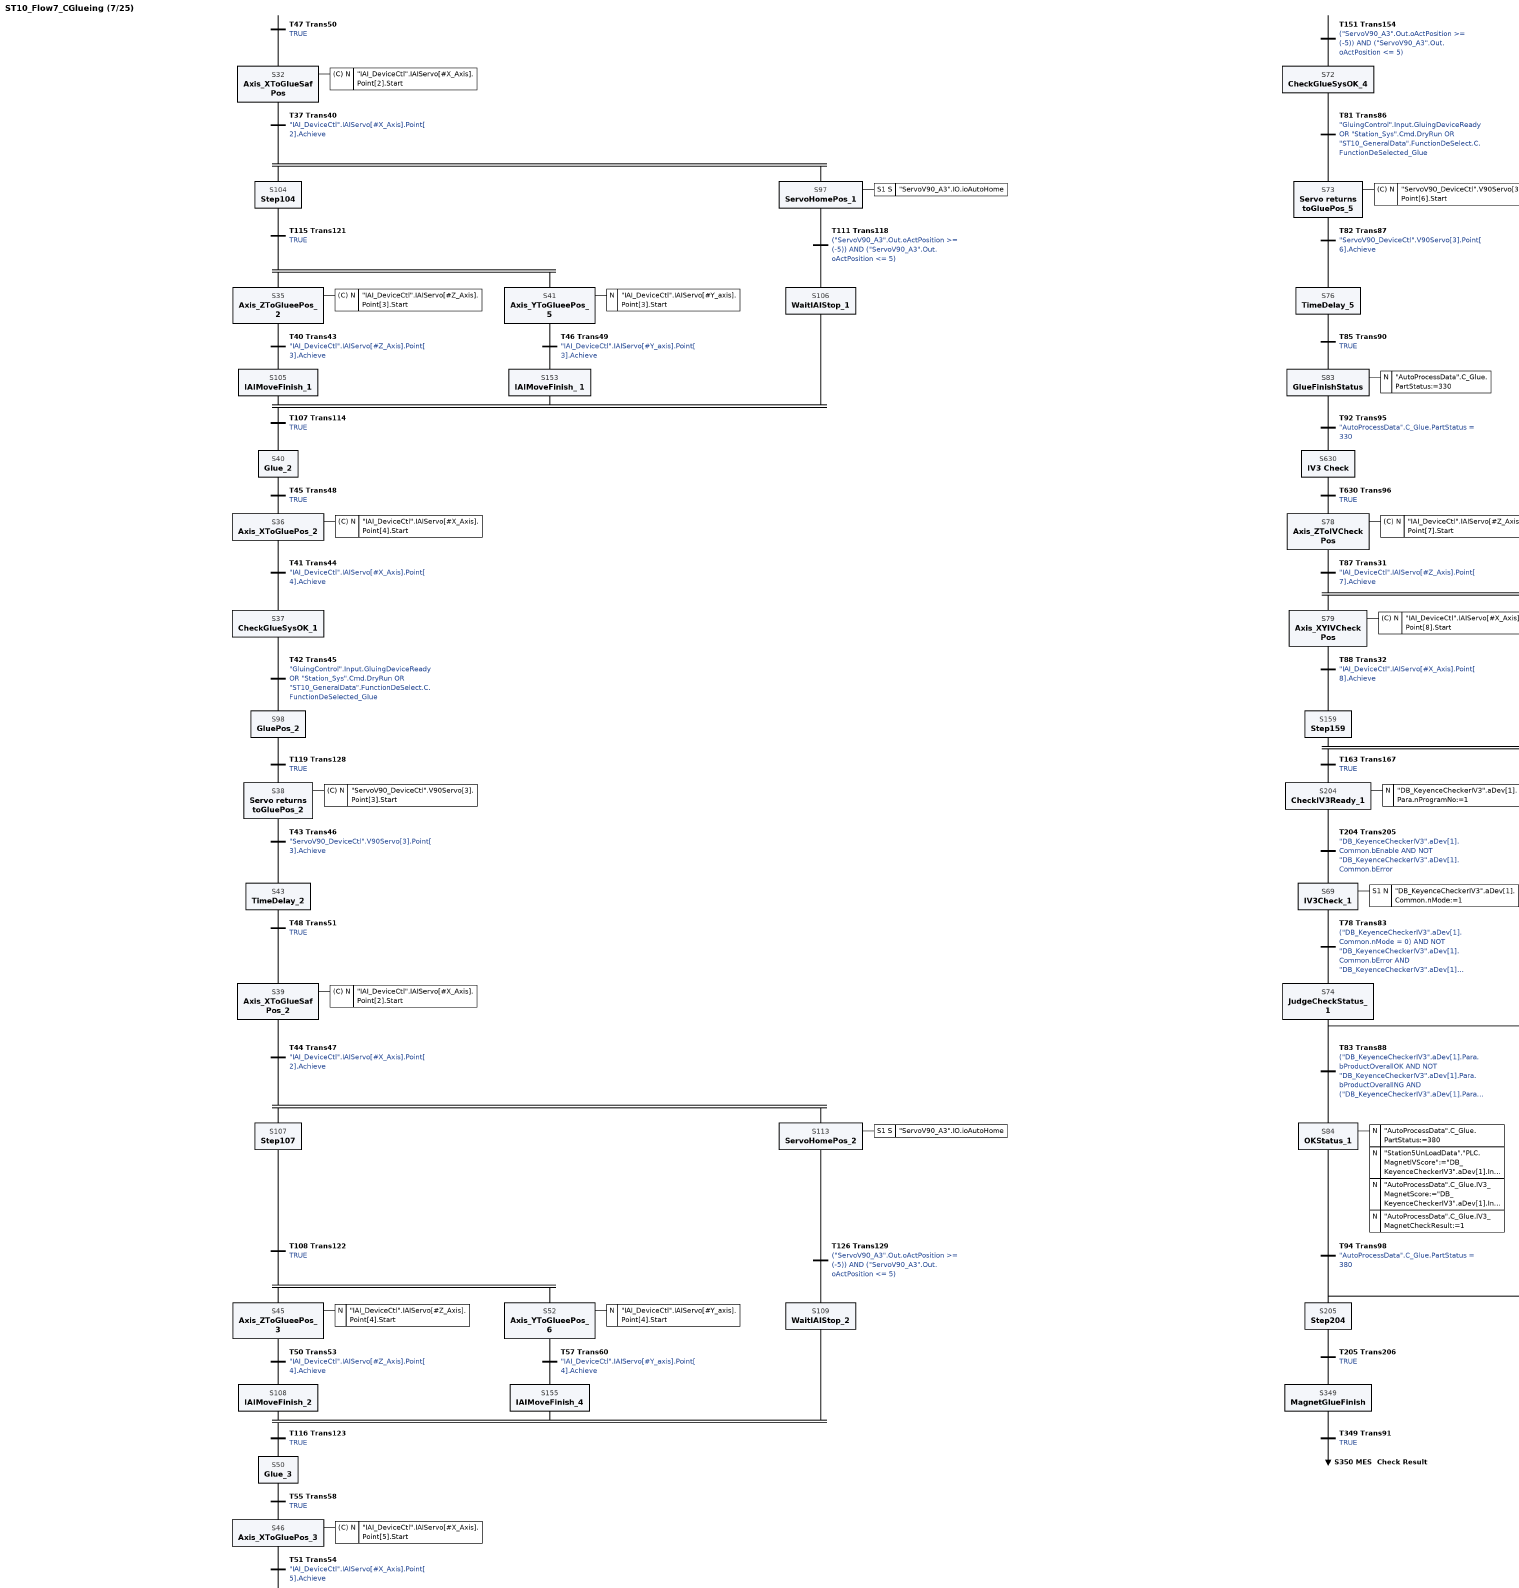
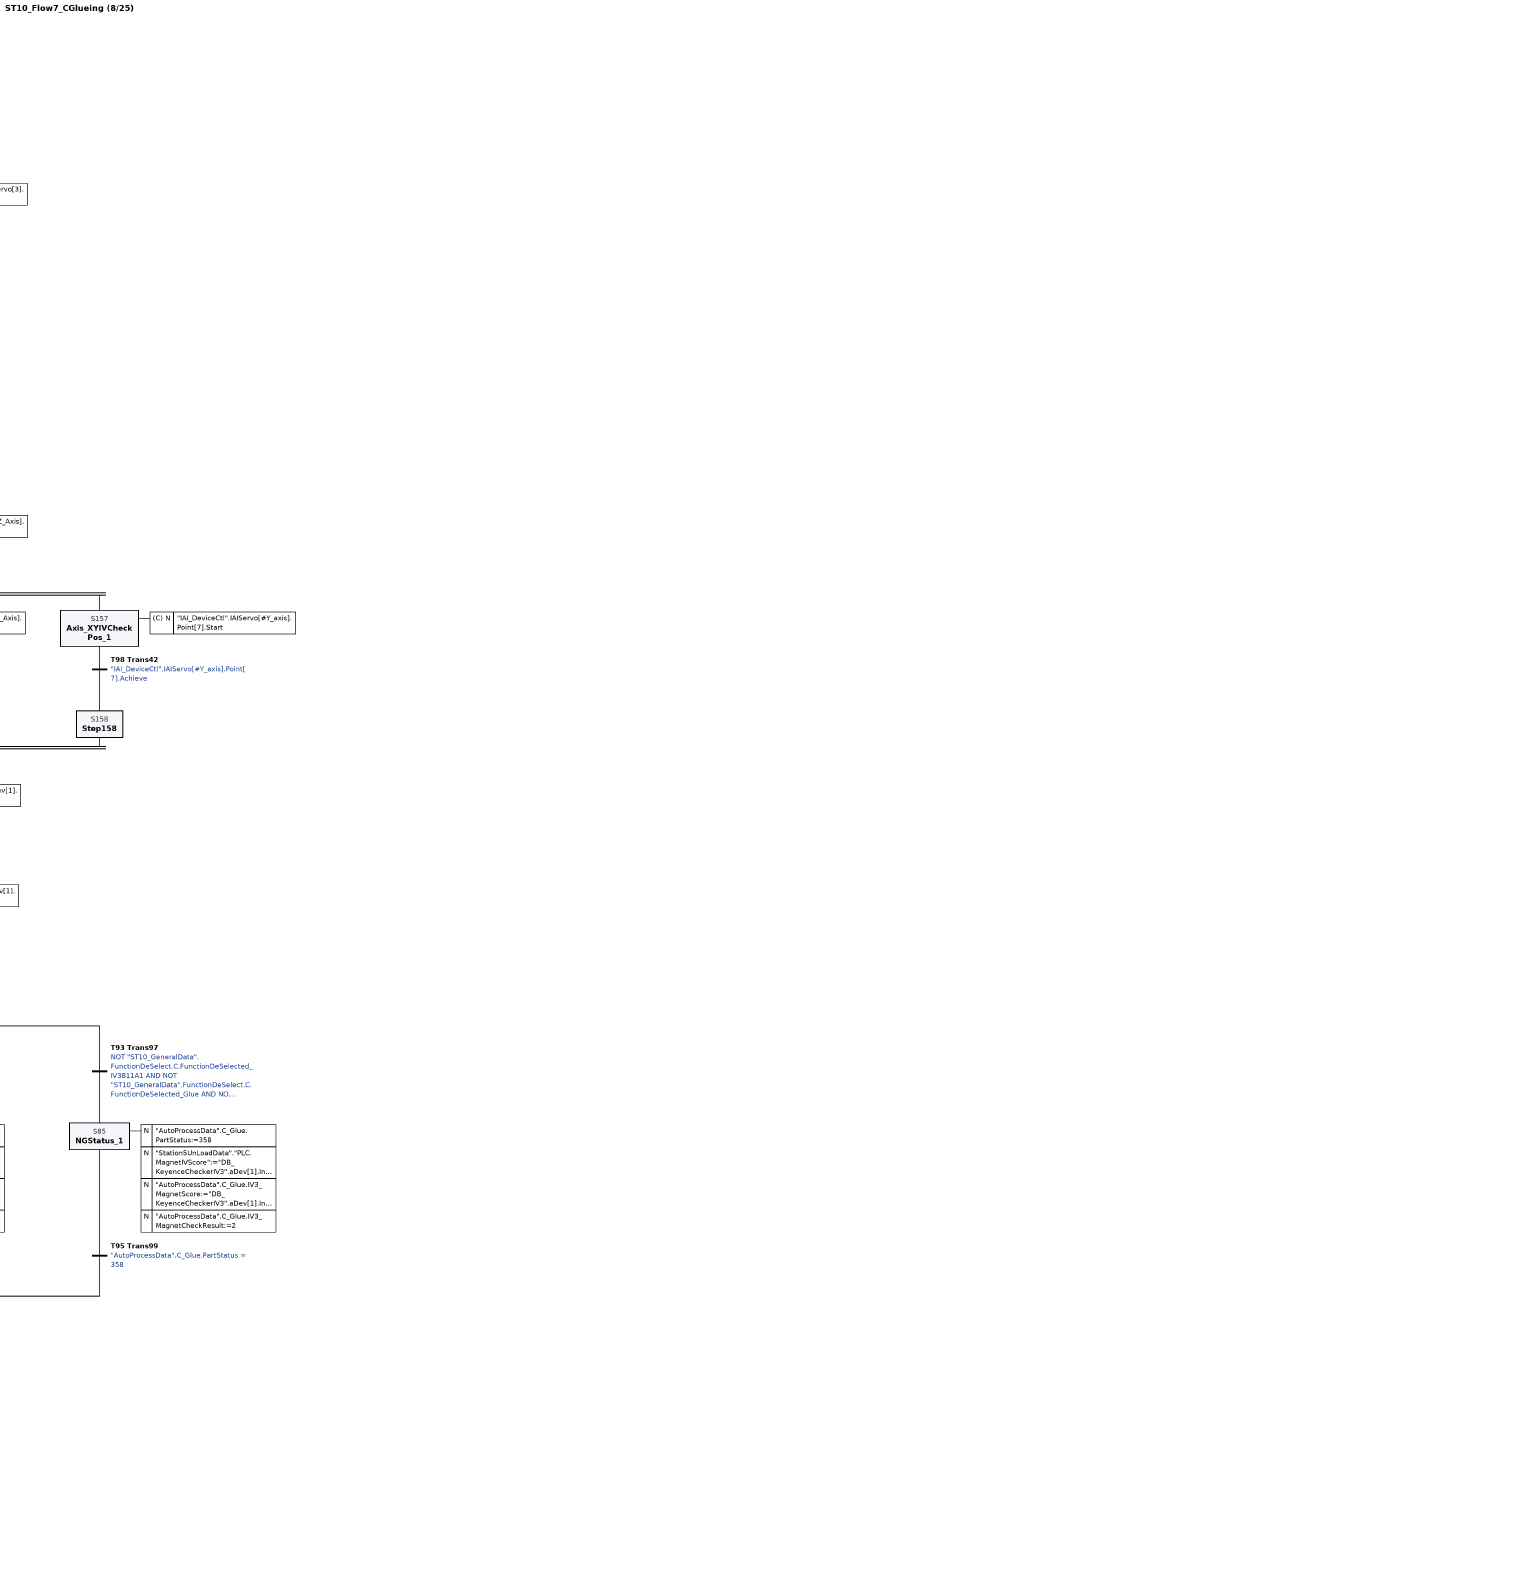
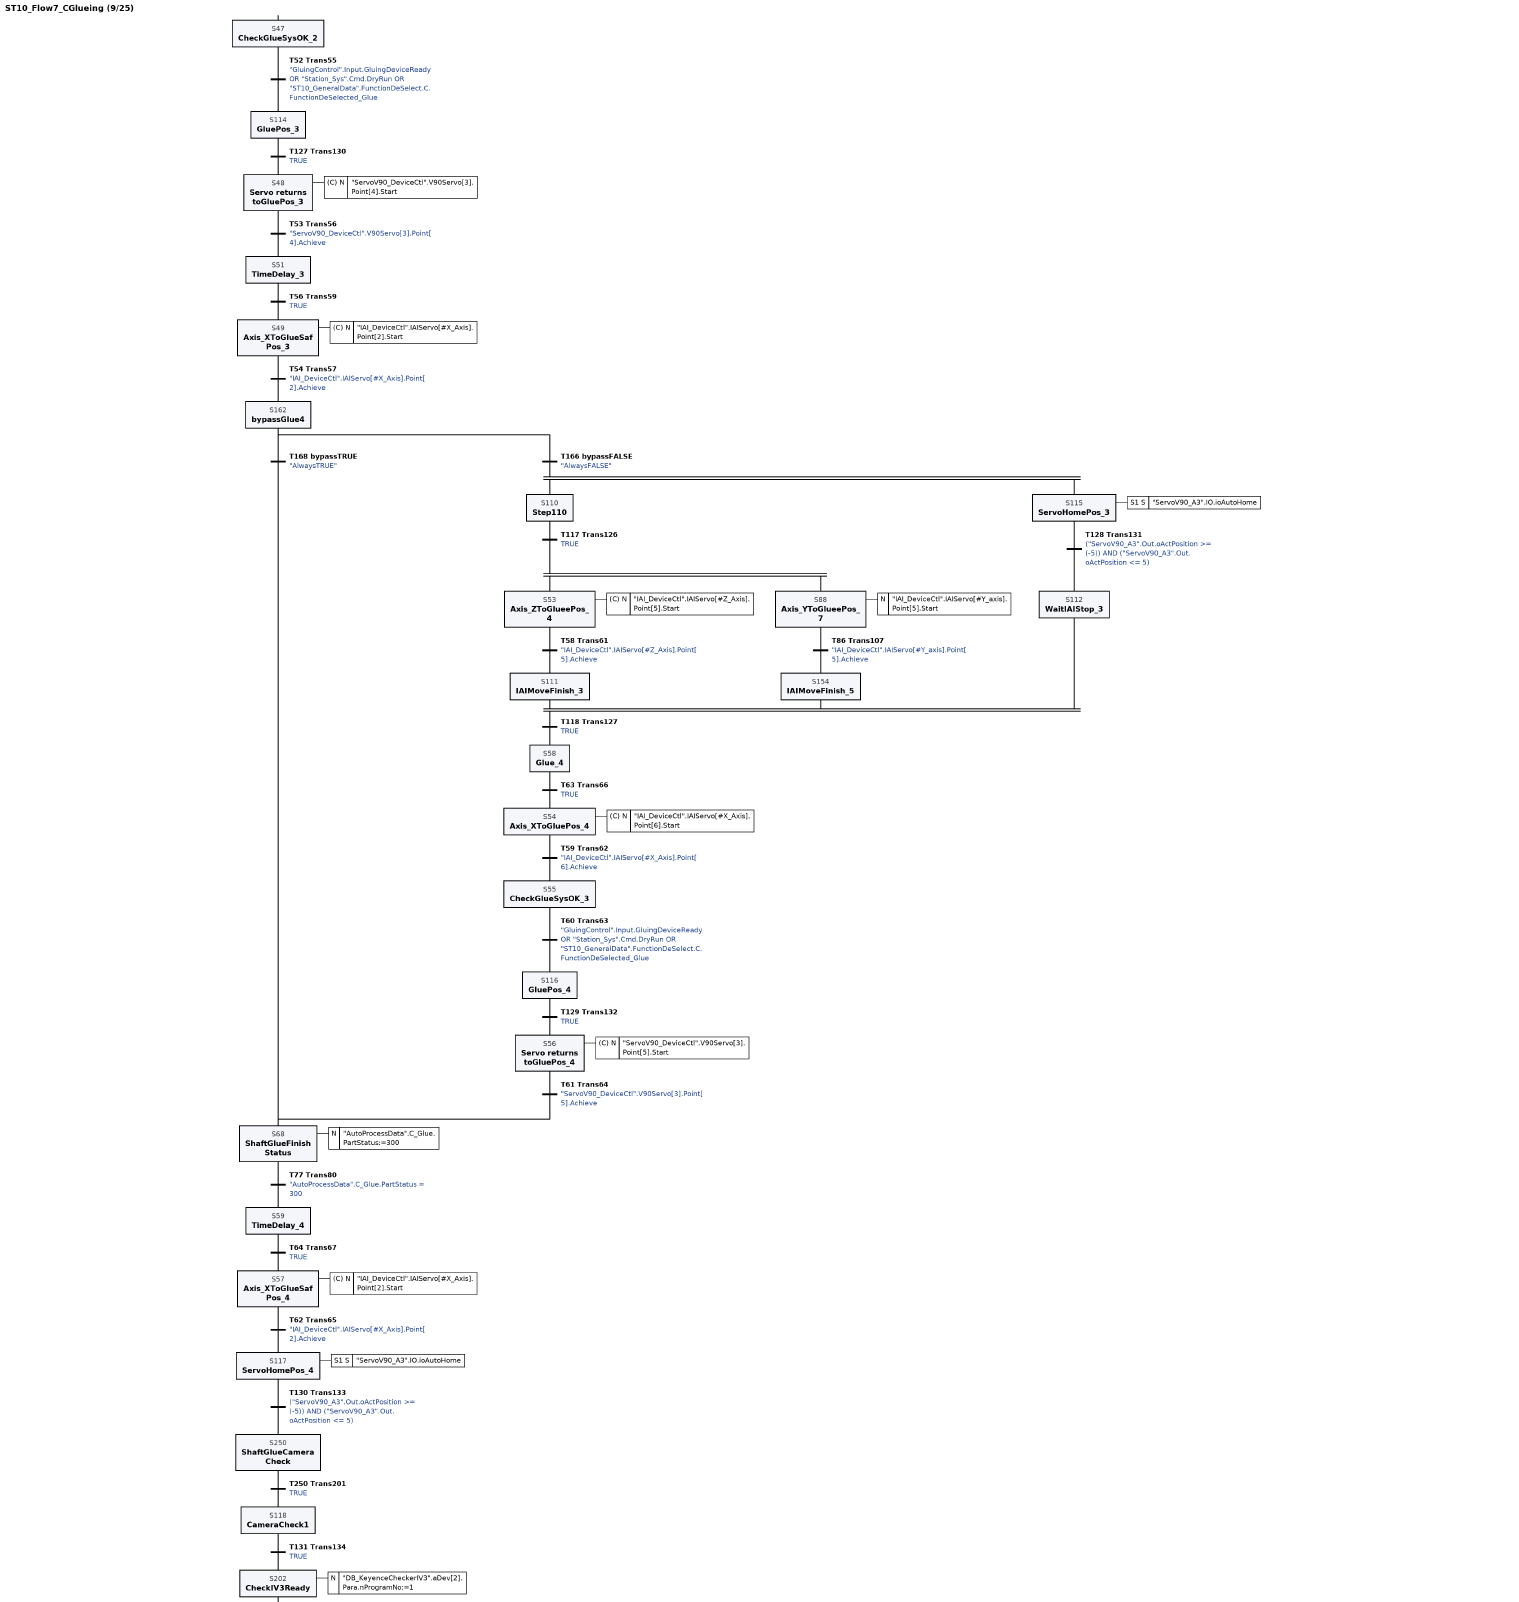
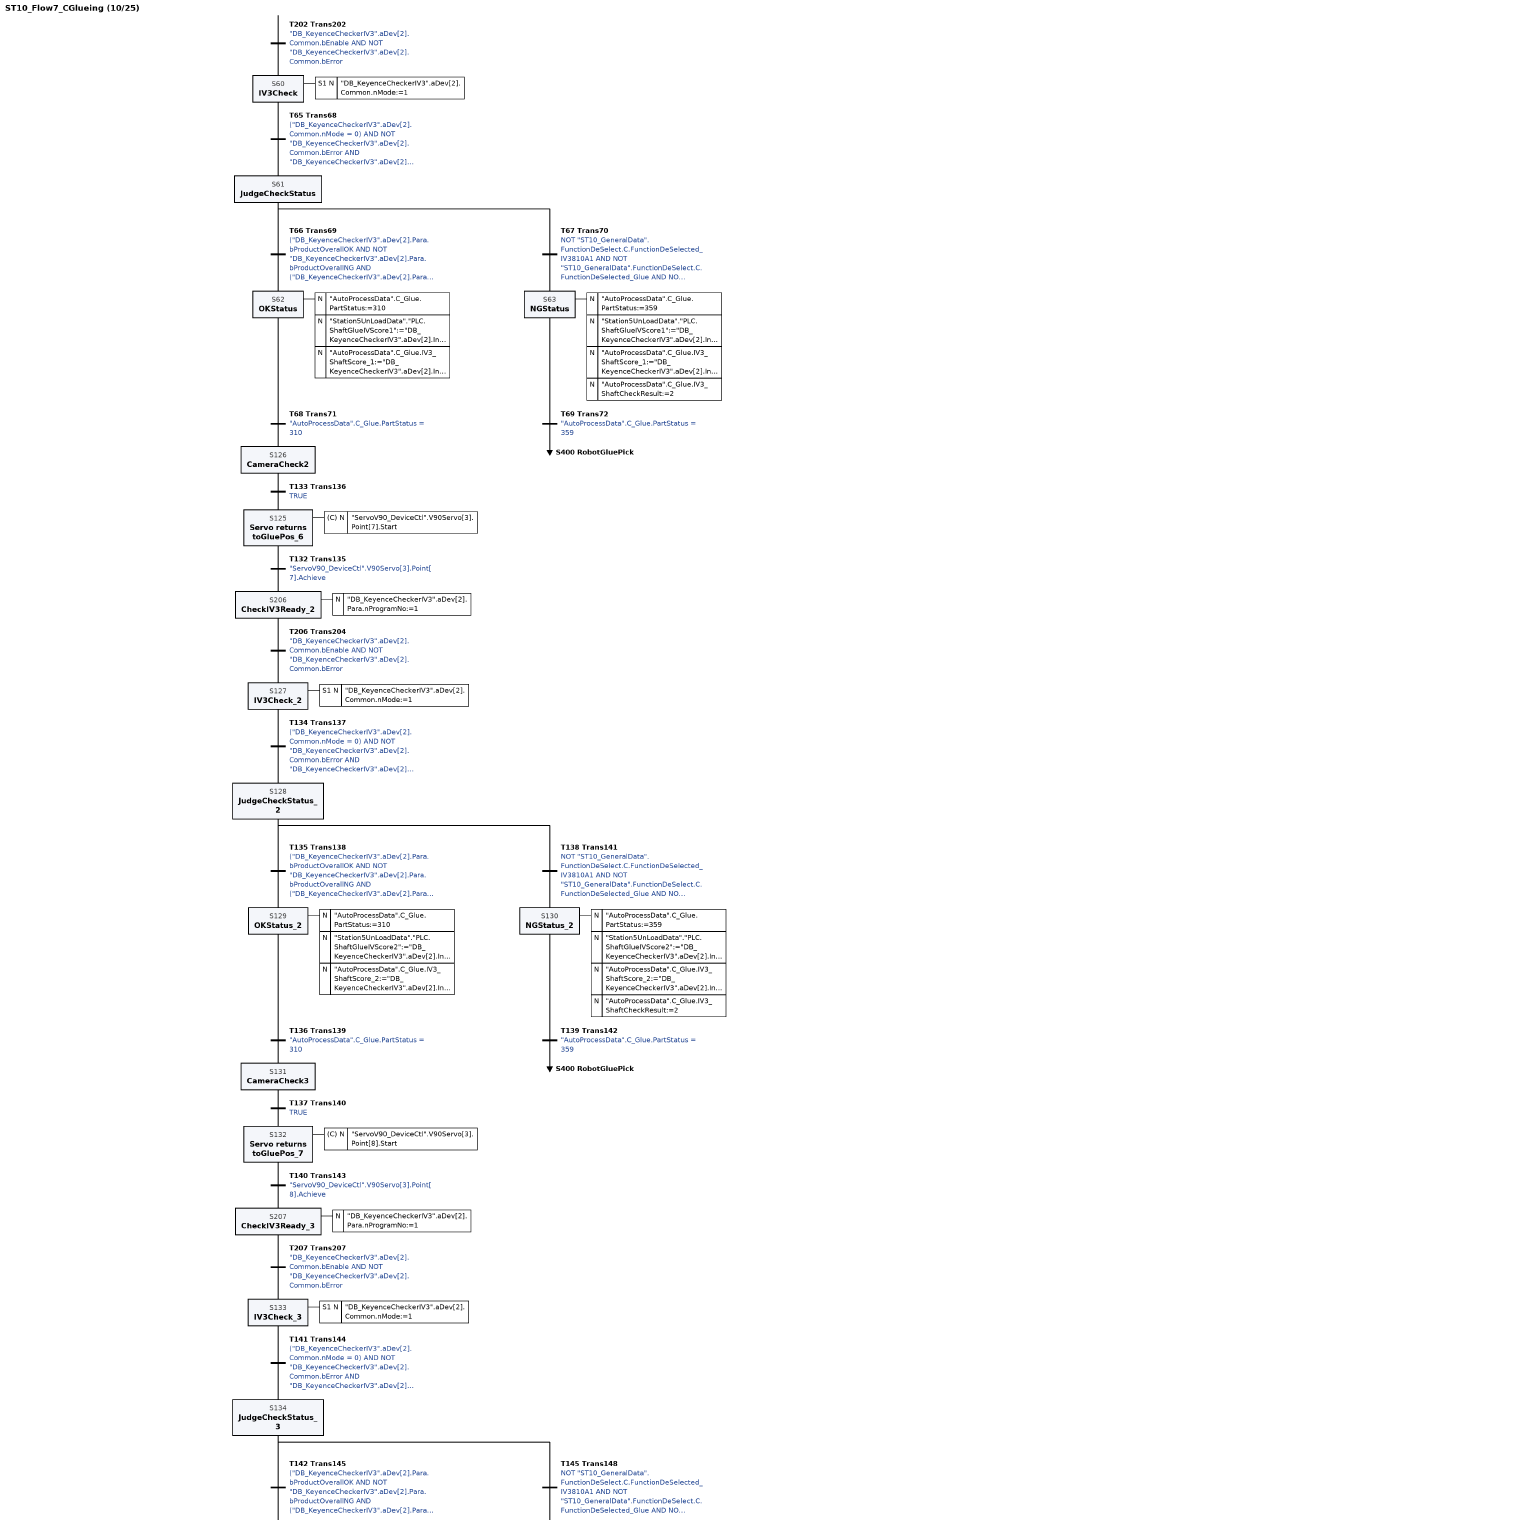
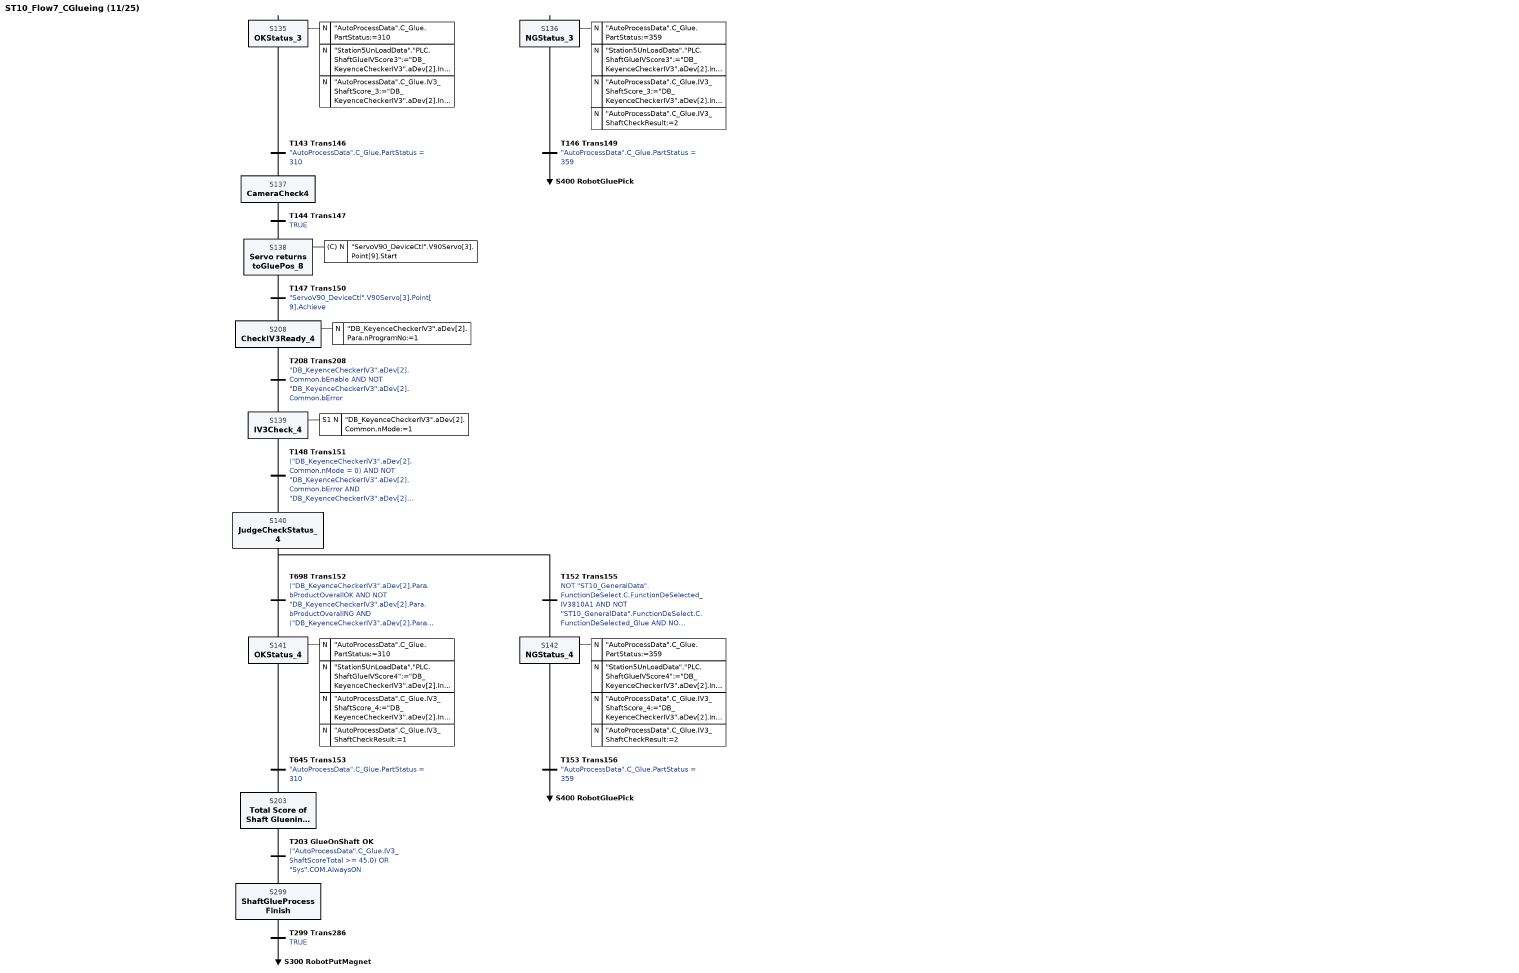
   // permanent pre-instructions
   NETWORK 1
      #TON[10].TON(IN := "AlwaysTRUE" AND "Station_Sys".Alarm.ImmediatelyStop, PT := T#300ms);
      #ioPM_Inface.AlarmImdilyStop := #TON[10].Q;
      #ioPM_Inface.AlarmCycleStop := "AlwaysTRUE" AND "Station_Sys".Alarm.CycleStop;
   NETWORK 2
      IF NOT False THEN
          #sCtrlMode(iSysInface := #iSysInface, ioPM_Inface := #ioPM_Inface, ioGraphCtrl := #RT_DATA.MOP);   // "SysFlowCtrlGraph"
      END_IF;
   NETWORK 3
      #TON[0].TON(IN := "AlwaysTRUE" AND "iA-Loading-01PipeDetection", PT := t#500ms);   // 工位11有托盘
      #TOF[1].TOF(IN := "AlwaysTRUE" AND NOT "iA-Loading-01PipeDetection", PT := T#300ms);   // 工位无托盘
      #TON[2].TON(IN := "AlwaysTRUE" AND "iA-Loading-01Detection", PT := T#300ms);
      #TOF[3].TOF(IN := "AlwaysTRUE" AND NOT "iA-Loading-01Detection", PT := T#300ms);
      #TON[4].TON(IN := "AlwaysTRUE" AND "iA-Loading-01GripperTakeDetection", PT := T#300ms);
      #TOF[5].TOF(IN := "AlwaysTRUE" AND NOT "iA-Loading-01GripperTakeDetection", PT := T#300ms);
   NETWORK 4
      #前站站号 := 345;
      #本站站号 := 350;
   NETWORK 5
      IF ("AutoProcessData".C_Glue.IV3_ShaftScore_1 <> 0) AND ("AutoProcessData".C_Glue.IV3_ShaftScore_2 <> 0) AND ("AutoProcessData".C_Glue.IV3_ShaftScore_3 <> 0) AND ("AutoProcessData".C_Glue.IV3_ShaftScore_4 <> 0) THEN
          "AutoProcessData".C_Glue.IV3_ShaftScoreTotal := "AutoProcessData".C_Glue.IV3_ShaftScore_1 + "AutoProcessData".C_Glue.IV3_ShaftScore_2 + "AutoProcessData".C_Glue.IV3_ShaftScore_3 + "AutoProcessData".C_Glue.IV3_ShaftScore_4;
          "AutoProcessData".C_Glue.IV3_ShaftScoreTotal := "AutoProcessData".C_Glue.IV3_ShaftScoreTotal - 4.0;
      END_IF;

   // sequencer 1: S01-S99 初始化 / S01-S99 Initial
   INITIAL_STEP F7_Initial:   // S1, max time T#10S, warning time T#7S
              S    #ioPM_Inface.InitialRun
              R    #ioPM_Inface.InitialOK
              R    #ioPM_Inface.WaitRunning
              R    #ioPM_Inface.Running
              R    #ioPM_Inface.UnPause
              R    "Station_Sys".Cmd.Calibration
              R    "Station_Sys".Cmd.ChangeOver
                   //"ST350_Sys".Cmd.DryRun
              R    "Station_Sys".Cmd.Reserve
              R    "Station_Sys".Cmd.OneCycle
              R    #ioPM_Inface.ProcessComplete
              R    #ioPM_Inface.ProcessStart
              R    "AutoProcessControl".C_Glue.Robot1PutPrimit
              R    "AutoProcessControl".C_Glue.Robot2PickPrimit
              R    "AutoProcessControl".C_Glue.Robot2MaganePutPrimit
   END_STEP
   TRANSITION Trans1 FROM F7_Initial TO S2   // T1
      := #iSysInface.Ready;
   END_TRANSITION
   STEP S2:   // S2, max time T#10S, warning time T#7S
   END_STEP
   TRANSITION Trans2 FROM S2 TO S3   // T2
      := TRUE;
   END_TRANSITION
   STEP S4:   // S4, max time T#10S, warning time T#7S
   END_STEP
   TRANSITION Trans3 FROM S4 TO S5_MESInitial   // T3
      := TRUE;
   END_TRANSITION
   STEP S5_MESInitial:   // S5, max time T#10S, warning time T#7S
   END_STEP
   TRANSITION Trans325 FROM S5_MESInitial TO WaitRobotInitialFinish   // T4
      := TRUE;
   END_TRANSITION
   STEP S10_InitialFinish:   // S10, max time T#10S, warning time T#7S
              S    #ioPM_Inface.InitialOK
   END_STEP
   TRANSITION Trans102 FROM S10_InitialFinish TO ProcessStart   // T10, jump
      := #ioPM_Inface.Running;
   END_TRANSITION
   STEP S3:   // S3, max time T#10S, warning time T#7S
   END_STEP
   TRANSITION Trans613 FROM S3 TO "ServoReady?"   // T607
      := TRUE;
   END_TRANSITION
   STEP WaitRobotInitialFinish:   // S8, max time T#10S, warning time T#7S
   END_STEP
   TRANSITION Trans10 FROM WaitRobotInitialFinish TO Axis_XToHomePos   // T8
      := "KukaRobot2_CtrlDB".sROBtoPLC.User.Home.DO163_HomeSeqOK OR "KukaRobot2_CtrlDB".sROBtoPLC.Sys.SO.IN_HOME OR "Tag_2";
   END_TRANSITION
   STEP Axis_ZToHomePos_2:   // S82, max time T#10S, warning time T#7S
      interlock C := NOT "IAI_DeviceCtl".IAIServo[#Z_Axis].Point[1].Achieve;
      (C)     N    "IAI_DeviceCtl".IAIServo[#Z_Axis].Point[1].Start
   END_STEP
   TRANSITION Trans106 FROM Axis_ZToHomePos_2 TO "C-LocationCylinderToHP"   // T91
      := "IAI_DeviceCtl".IAIServo[#Z_Axis].Point[1].Achieve;
   END_TRANSITION
   STEP Axis_XToHomePos:   // S81, max time T#10S, warning time T#7S
      interlock C := NOT "IAI_DeviceCtl".IAIServo[#X_Axis].Point[1].Achieve;
      (C)     N    "IAI_DeviceCtl".IAIServo[#X_Axis].Point[1].Start
   END_STEP
   TRANSITION Trans105 FROM Axis_XToHomePos TO Axis_YToHomePos   // T90
      := "IAI_DeviceCtl".IAIServo[#X_Axis].Point[1].Achieve;
   END_TRANSITION
   STEP "Servo returns toHome Pos":   // S22, max time T#10S, warning time T#7S
      interlock C := "ServoV90_A3".Out.oReady;
      (C)     N    "ServoV90_DeviceCtl".V90Servo[3].Point[1].Start
   END_STEP
   TRANSITION Trans24 FROM "Servo returns toHome Pos" TO Glue2s   // T23
      := "ServoV90_DeviceCtl".V90Servo[3].Point[1].Achieve OR "AlwaysTRUE";
   END_TRANSITION
   STEP Axis_YToHomePos:   // S21, max time T#10S, warning time T#7S
      interlock C := NOT "IAI_DeviceCtl".IAIServo[#Y_axis].Point[1].Achieve;
      (C)     N    "IAI_DeviceCtl".IAIServo[#Y_axis].Point[1].Start
   END_STEP
   TRANSITION Trans23 FROM Axis_YToHomePos TO Axis_ZToHomePos_2   // T22
      := "IAI_DeviceCtl".IAIServo[#Y_axis].Point[1].Achieve;
   END_TRANSITION
   STEP "ServoReady?":   // S6, max time T#10S, warning time T#7S
   END_STEP
   TRANSITION Trans4 FROM "ServoReady?" TO S4   // T5
      := "ServoV90_A3".Out.oReady;
   END_TRANSITION
   STEP "C-LocationCylinderToHP":   // S119, max time T#10S, warning time T#7S
              S    "ST10Cylinder".Cy[9].Inout.AutoGoHome
              R    "ST10Cylinder".Cy[9].Inout.AutoGoWork
   END_STEP
   TRANSITION Trans767 FROM "C-LocationCylinderToHP" TO "Servo returns toHome Pos"   // T120
      := NOT "ST10Cylinder".Cy[9].In.WorkPositionSensor AND "ST10Cylinder".Cy[9].In.HomePositionSensor;
   END_TRANSITION
   STEP Glue2s:   // S163, max time T#10S, warning time T#7S
              N    "GluingControl".GlueInitiaStart
   END_STEP
   TRANSITION Trans170 FROM Glue2s TO S10_InitialFinish   // T167
      := #Glue2s.T > "DB_ALL_PROCESS_PARAMETERS".ACTUAL_CHOOSEN_TYPE.Process.Timers.Delay_glue_init_start;
   END_TRANSITION

   // sequencer 2: S100-S199 等待到位 / S100-S149 CheckPartStatus
   STEP ProcessStart:   // S100, max time T#10S, warning time T#7S
      // 自动等待开始运行
              R    #ioPM_Inface.InitialRun
              R    #ioPM_Inface.ProcessComplete
              R    #ioPM_Inface.ProcessStart
              S    #ioPM_Inface.InitialOK
              S    #ioPM_Inface.WaitRunning
          S1  N    #ioPM_Inface.ProcessResult:=0
              R    "ST10_GeneralData".FlowControl_Handshake[7].Start
              R    "ST10_GeneralData".FlowControl_Handshake[7].Done
   END_STEP
   TRANSITION Trans200 FROM ProcessStart TO "WaitTableCode OK"   // T100
      := NOT #ioPM_Inface.AlarmCycleStop AND #ioPM_Inface.Running AND NOT #iSysInface.Auto.RunningOver AND (NOT #iSysInface.Auto.OneCycleMode OR (#iSysInface.Auto.OneCycleMode AND #ioPM_Inface.TriggerOneCycle));
   END_TRANSITION
   STEP "Process Finish":   // S149, max time T#10S, warning time T#7S
   END_STEP
   TRANSITION Trans250 FROM "Process Finish" TO "MES Check"   // T149, jump
      := TRUE;
   END_TRANSITION
   STEP StatusAlarm:   // S24, max time T#10S, warning time T#7S
          S1  S    "ST10_DeviceError".C.CGlueing.StatusError
   END_STEP
   TRANSITION Trans30 FROM StatusAlarm TO CheckPartStatus   // T29, jump
      := #iSysInface.Reset;
   END_TRANSITION
   STEP "Shaft Glue":   // S287, max time T#10S, warning time T#7S
   END_STEP
   TRANSITION Trans287 FROM "Shaft Glue" TO "Process Finish"   // T287
      := TRUE;
   END_TRANSITION
   STEP "WaitTableCode OK":   // S101, max time T#10S, warning time T#7S
              N    "MES_CHeck_DB".Station_5.CheckStep:=0
              N    "MES_CHeck_DB".Station_5.ResultStep:=0
   END_STEP
   TRANSITION Trans101 FROM "WaitTableCode OK" TO CheckPartStatus   // T101
      := TRUE;
   END_TRANSITION
   STEP RequestRobot1PutShaft:   // S27, max time T#10S, warning time T#7S
              N    "AutoProcessControl".C_Glue.Robot1PutPrimit
   END_STEP
   TRANSITION Trans33 FROM RequestRobot1PutShaft TO WaitRobot1FinishTask   // T32
      := ("KukaRobot1_CtrlDB".sROBtoPLC.User.Cycle.DO289_GluePutInside AND NOT "KukaRobot1_CtrlDB".sROBtoPLC.User.Cycle.DO290_GluePutFinish) OR ("AutoProcessControl".C_Glue.GlueTest AND "iC-LocationShaftDetection" AND "iHMI Machine Start");
   END_TRANSITION
   STEP WaitRobot1FinishTask:   // S28, max time T#10S, warning time T#7S
   END_STEP
   TRANSITION Trans34 FROM WaitRobot1FinishTask TO "Process Finish"   // T33
      := "KukaRobot1_CtrlDB".sROBtoPLC.User.Cycle.DO290_GluePutFinish OR "AutoProcessControl".C_Glue.GlueTest;
   END_TRANSITION
   STEP CheckPartStatus:   // S23, max time T#10S, warning time T#7S
   END_STEP
   TRANSITION Trans25 FROM CheckPartStatus TO "C-LocationCylinderToWP_2"   // T24
      := ("AutoProcessData".C_Glue.PartStatus = 0) AND NOT "iC-LocationShaftDetection";
   END_TRANSITION
   TRANSITION Trans26 FROM CheckPartStatus TO "Shaft Glue"   // T25
      := (("AutoProcessData".C_Glue.PartStatus = 299) OR "AutoProcessControl".C_Glue.GlueTest) AND "iC-LocationShaftDetection";
   END_TRANSITION
   TRANSITION Trans27 FROM CheckPartStatus TO PutMagnet   // T26
      := ("AutoProcessData".C_Glue.PartStatus = 310) AND "iC-LocationShaftDetection";
   END_TRANSITION
   TRANSITION NG FROM CheckPartStatus TO PartNG   // T27
      := ("AutoProcessData".C_Glue.PartStatus >= 350) AND ("AutoProcessData".C_Glue.PartStatus <= 360);
   END_TRANSITION
   TRANSITION Trans29 FROM CheckPartStatus TO StatusAlarm   // T28
      := ((("AutoProcessData".C_Glue.PartStatus <> 0) AND NOT "iC-LocationShaftDetection") OR (("AutoProcessData".C_Glue.PartStatus = 0) AND "iC-LocationShaftDetection")) AND NOT "AutoProcessControl".C_Glue.GlueTest;
   END_TRANSITION
   TRANSITION Trans73 FROM CheckPartStatus TO Magnet_Glue   // T70
      := ("AutoProcessData".C_Glue.PartStatus = 320) AND "iC-LocationShaftDetection";
   END_TRANSITION
   TRANSITION Trans76 FROM CheckPartStatus TO Magnet_GlueCheck   // T73
      := ("AutoProcessData".C_Glue.PartStatus = 330) AND "iC-LocationShaftDetection";
   END_TRANSITION
   TRANSITION Trans78 FROM CheckPartStatus TO "Shaft GlueCheck"   // T75
      := ("AutoProcessData".C_Glue.PartStatus = 300) AND "iC-LocationShaftDetection";
   END_TRANSITION
   TRANSITION Trans163 FROM CheckPartStatus TO MESResult   // T159
      := "AutoProcessData".C_Glue.PartStatus = 380;
   END_TRANSITION
   TRANSITION Trans165 FROM CheckPartStatus TO OKPart   // T161
      := "AutoProcessData".C_Glue.PartStatus = 399;
   END_TRANSITION
   STEP PutMagnet:   // S64, max time T#10S, warning time T#7S
   END_STEP
   TRANSITION Trans74 FROM PutMagnet TO RobotPutMagnet   // T71, jump
      := TRUE;
   END_TRANSITION
   STEP Magnet_Glue:   // S65, max time T#10S, warning time T#7S
   END_STEP
   TRANSITION Trans75 FROM Magnet_Glue TO MaganetGlue   // T72, jump
      := TRUE;
   END_TRANSITION
   STEP Magnet_GlueCheck:   // S66, max time T#10S, warning time T#7S
   END_STEP
   TRANSITION Trans77 FROM Magnet_GlueCheck TO "IV3 Check"   // T74, jump
      := TRUE;
   END_TRANSITION
   STEP "Shaft GlueCheck":   // S67, max time T#10S, warning time T#7S
   END_STEP
   TRANSITION Trans79 FROM "Shaft GlueCheck" TO ShaftGlueCameraCheck   // T76, jump
      := TRUE;
   END_TRANSITION
   STEP PartNG:   // S401, max time T#10S, warning time T#7S
   END_STEP
   TRANSITION Trans401 FROM PartNG TO RobotGluePick   // T401, jump
      := TRUE;
   END_TRANSITION
   STEP "C-LocationCylinderToWP_2":   // S121, max time T#10S, warning time T#7S
              R    "ST10Cylinder".Cy[9].Inout.AutoGoHome
              S    "ST10Cylinder".Cy[9].Inout.AutoGoWork
              R    #ioPM_Inface.ProcessComplete
              S    #ioPM_Inface.ProcessStart
   END_STEP
   TRANSITION Trans769 FROM "C-LocationCylinderToWP_2" TO RequestRobot1PutShaft   // T122
      := ("ST10Cylinder".Cy[9].In.WorkPositionSensor OR ("Tag_23" AND (#"C-LocationCylinderToWP_2".T > t#100MS))) AND NOT "ST10Cylinder".Cy[9].In.HomePositionSensor;
   END_TRANSITION
   STEP MESResult:   // S151, max time T#10S, warning time T#7S
   END_STEP
   TRANSITION Trans164 FROM MESResult TO "MES  Check Result"   // T160, jump
      := TRUE;
   END_TRANSITION
   STEP OKPart:   // S152, max time T#10S, warning time T#7S
   END_STEP
   TRANSITION Trans166 FROM OKPart TO RobotGluePick   // T162, jump
      := TRUE;
   END_TRANSITION

   // sequencer 3: S150-S199 MES Check
   STEP "MES Check":   // S150, max time T#10S, warning time T#7S
   END_STEP
   TRANSITION Trans161 FROM "MES Check" TO Bypass   // T150
      := TRUE;
   END_TRANSITION
   STEP "Prepare MES CheckData":   // S303, max time T#10S, warning time T#7S
   END_STEP
   TRANSITION Trans14 FROM "Prepare MES CheckData" TO MESCheckRequest   // T303
      := #"Prepare MES CheckData".T > t#300MS;
   END_TRANSITION
   STEP "MES Check OK":   // S306, max time T#10S, warning time T#7S
   END_STEP
   TRANSITION Trans307 FROM "MES Check OK" TO ShaftGluingProcess   // T307, jump
      := TRUE;
   END_TRANSITION
   STEP MESCheckRequest:   // S310, max time T#10S, warning time T#7S
              N    "PLCtoMES"."PLC.Load_Station5ChickInReq"
   END_STEP
   TRANSITION Trans264 FROM MESCheckRequest TO "Check OK"   // T305
      := "MEStoPLC"."MES.Load_Station5PartOK" AND NOT "MEStoPLC"."MES.Load_Station5PartNG" AND "MEStoPLC"."MES.Load_Station5ReqMesDone";
   END_TRANSITION
   TRANSITION Trans610 FROM MESCheckRequest TO "Check NG"   // T314
      := NOT "MEStoPLC"."MES.Load_Station5PartOK" AND "MEStoPLC"."MES.Load_Station5PartNG" AND "MEStoPLC"."MES.Load_Station5ReqMesDone";
   END_TRANSITION
   TRANSITION Trans316 FROM MESCheckRequest TO MESOverTime_1   // T323
      := #MESCheckRequest.T > t#10S;
   END_TRANSITION
   STEP ResetMesCheckRequest:   // S301, max time T#10S, warning time T#7S
              R    "PLCtoMES"."PLC.Load_Station5ChickInReq"
              R    "MEStoPLC"."MES.Load_Station5PartOK"
              R    "MEStoPLC"."MES.Load_Station5PartNG"
              R    "MEStoPLC"."MES.Load_Station5ReqMesDone"
   END_STEP
   TRANSITION Trans259 FROM ResetMesCheckRequest TO "Prepare MES CheckData"   // T302
      := NOT "PLCtoMES"."PLC.Load_Station5ChickInReq" AND NOT "MEStoPLC"."MES.Load_Station5PartOK" AND NOT "MEStoPLC"."MES.Load_Station5PartNG" AND NOT "MEStoPLC"."MES.Load_Station5ReqMesDone";
   END_TRANSITION
   STEP "Check OK":   // S316, max time T#10S, warning time T#7S
   END_STEP
   TRANSITION Trans322 FROM "Check OK" TO "MES Check OK"   // T322
      := TRUE;
   END_TRANSITION
   STEP "Check NG":   // S317, max time T#10S, warning time T#7S
              N    "AutoProcessData".C_Glue.PartStatus:=351
   END_STEP
   TRANSITION Trans17 FROM "Check NG" TO RobotGluePick   // T316, jump
      := "AutoProcessData".C_Glue.PartStatus = 351;
   END_TRANSITION
   STEP Bypass:   // S315, max time T#10S, warning time T#7S
   END_STEP
   TRANSITION Online FROM Bypass TO ResetMesCheckRequest   // T301
      := NOT "Station_Sys".Cmd.OnOffLine AND NOT "AutoProcessControl".C_Glue.GlueTest;
   END_TRANSITION
   TRANSITION Offline FROM Bypass TO Step314   // T13
      := "Station_Sys".Cmd.OnOffLine OR "AutoProcessControl".C_Glue.GlueTest;
   END_TRANSITION
   STEP MESOverTime_1:   // S318, max time T#10S, warning time T#7S
              S    "ST10_DeviceError".MES_Error.CheckInCompOverTime_5
   END_STEP
   TRANSITION Trans317 FROM MESOverTime_1 TO Bypass   // T324, jump
      := #iSysInface.Reset;
   END_TRANSITION
   STEP Step314:   // S322, max time T#10S, warning time T#7S
   END_STEP
   TRANSITION Trans320 FROM Step314 TO "MES Check OK"   // T327
      := TRUE;
   END_TRANSITION

   // sequencer 4: S200-S299 ShaftGluing
   STEP ShaftGluingProcess:   // S200, max time T#10S, warning time T#7S
   END_STEP
   TRANSITION Trans35 FROM ShaftGluingProcess TO "C-LocationCylinderToHP2"   // T200
      := TRUE;
   END_TRANSITION
   STEP ShaftGlueCameraCheck:   // S250, max time T#10S, warning time T#7S
   END_STEP
   TRANSITION Trans201 FROM ShaftGlueCameraCheck TO CameraCheck1   // T250
      := TRUE;
   END_TRANSITION
   STEP CheckIV3Ready:   // S202, max time T#10S, warning time T#7S
              N    "DB_KeyenceCheckerIV3".aDev[2].Para.nProgramNo:=1
   END_STEP
   TRANSITION Trans202 FROM CheckIV3Ready TO IV3Check   // T202
      := "DB_KeyenceCheckerIV3".aDev[2].Common.bEnable AND NOT "DB_KeyenceCheckerIV3".aDev[2].Common.bError;
   END_TRANSITION
   STEP "Total Score of Shaft Gluening check":   // S203, max time T#10S, warning time T#7S
   END_STEP
   TRANSITION "GlueOnShaft OK" FROM "Total Score of Shaft Gluening check" TO ShaftGlueProcessFinish   // T203
      := ("AutoProcessData".C_Glue.IV3_ShaftScoreTotal >= 45.0) OR "Sys".COM.AlwaysON;
   END_TRANSITION
   STEP ShaftGlueProcessFinish:   // S299, max time T#10S, warning time T#7S
   END_STEP
   TRANSITION Trans286 FROM ShaftGlueProcessFinish TO RobotPutMagnet   // T299, jump
      := TRUE;
   END_TRANSITION
   STEP WaitIAIStop:   // S103, max time T#10S, warning time T#7S
   END_STEP
   STEP Axis_XToGluePos_1:   // S29, max time T#10S, warning time T#7S
      interlock C := NOT "IAI_DeviceCtl".IAIServo[#X_Axis].Point[3].Achieve;
      (C)     N    "IAI_DeviceCtl".IAIServo[#X_Axis].Point[3].Start
   END_STEP
   TRANSITION Trans37 FROM Axis_XToGluePos_1 TO CheckGlueSysOK   // T34
      := "IAI_DeviceCtl".IAIServo[#X_Axis].Point[3].Achieve;
   END_TRANSITION
   STEP CheckGlueSysOK:   // S30, max time T#10S, warning time T#7S
   END_STEP
   TRANSITION Trans38 FROM CheckGlueSysOK TO GluePos_1   // T35
      := "GluingControl".Input.GluingDeviceReady OR "Station_Sys".Cmd.DryRun OR "ST10_GeneralData".FunctionDeSelect.C.FunctionDeSelected_Glue;
   END_TRANSITION
   STEP "Servo returns toGluePos_1":   // S31, max time T#10S, warning time T#7S
      (C)     N    "ServoV90_DeviceCtl".V90Servo[3].Point[2].Start
   END_STEP
   TRANSITION Trans39 FROM "Servo returns toGluePos_1" TO TimeDelay_1   // T36
      := "ServoV90_DeviceCtl".V90Servo[3].Point[2].Achieve;
   END_TRANSITION
   STEP Axis_XToGlueSafPos:   // S32, max time T#10S, warning time T#7S
      interlock C := NOT "IAI_DeviceCtl".IAIServo[#X_Axis].Point[2].Achieve;
      (C)     N    "IAI_DeviceCtl".IAIServo[#X_Axis].Point[2].Start
   END_STEP
   TRANSITION Trans40 FROM Axis_XToGlueSafPos TO (Step104, ServoHomePos_1)   // T37
      := "IAI_DeviceCtl".IAIServo[#X_Axis].Point[2].Achieve;
   END_TRANSITION
   STEP Glue_1:   // S33, max time T#10S, warning time T#7S
   END_STEP
   TRANSITION Trans41 FROM Glue_1 TO (Step102, ServoHomePos)   // T38
      := TRUE;
   END_TRANSITION
   STEP GluePos_3:   // S114, max time T#10S, warning time T#7S
   END_STEP
   TRANSITION Trans130 FROM GluePos_3 TO "Servo returns toGluePos_3"   // T127
      := TRUE;
   END_TRANSITION
   STEP IAIMoveFinish_1:   // S105, max time T#10S, warning time T#7S
   END_STEP
   STEP Axis_XToGluePos_2:   // S36, max time T#10S, warning time T#7S
      interlock C := NOT "IAI_DeviceCtl".IAIServo[#X_Axis].Point[4].Achieve;
      (C)     N    "IAI_DeviceCtl".IAIServo[#X_Axis].Point[4].Start
   END_STEP
   TRANSITION Trans44 FROM Axis_XToGluePos_2 TO CheckGlueSysOK_1   // T41
      := "IAI_DeviceCtl".IAIServo[#X_Axis].Point[4].Achieve;
   END_TRANSITION
   STEP CheckGlueSysOK_1:   // S37, max time T#10S, warning time T#7S
   END_STEP
   TRANSITION Trans45 FROM CheckGlueSysOK_1 TO GluePos_2   // T42
      := "GluingControl".Input.GluingDeviceReady OR "Station_Sys".Cmd.DryRun OR "ST10_GeneralData".FunctionDeSelect.C.FunctionDeSelected_Glue;
   END_TRANSITION
   STEP "Servo returns toGluePos_2":   // S38, max time T#10S, warning time T#7S
      (C)     N    "ServoV90_DeviceCtl".V90Servo[3].Point[3].Start
   END_STEP
   TRANSITION Trans46 FROM "Servo returns toGluePos_2" TO TimeDelay_2   // T43
      := "ServoV90_DeviceCtl".V90Servo[3].Point[3].Achieve;
   END_TRANSITION
   STEP Axis_XToGlueSafPos_2:   // S39, max time T#10S, warning time T#7S
      interlock C := NOT "IAI_DeviceCtl".IAIServo[#X_Axis].Point[2].Achieve;
      (C)     N    "IAI_DeviceCtl".IAIServo[#X_Axis].Point[2].Start
   END_STEP
   TRANSITION Trans47 FROM Axis_XToGlueSafPos_2 TO (Step107, ServoHomePos_2)   // T44
      := "IAI_DeviceCtl".IAIServo[#X_Axis].Point[2].Achieve;
   END_TRANSITION
   STEP Glue_2:   // S40, max time T#10S, warning time T#7S
   END_STEP
   TRANSITION Trans48 FROM Glue_2 TO Axis_XToGluePos_2   // T45
      := TRUE;
   END_TRANSITION
   STEP GluePos_2:   // S98, max time T#10S, warning time T#7S
   END_STEP
   TRANSITION Trans128 FROM GluePos_2 TO "Servo returns toGluePos_2"   // T119
      := TRUE;
   END_TRANSITION
   STEP TimeDelay_1:   // S42, max time T#10S, warning time T#7S
   END_STEP
   TRANSITION Trans50 FROM TimeDelay_1 TO Axis_XToGlueSafPos   // T47
      := TRUE;
   END_TRANSITION
   STEP TimeDelay_2:   // S43, max time T#10S, warning time T#7S
   END_STEP
   TRANSITION Trans51 FROM TimeDelay_2 TO Axis_XToGlueSafPos_2   // T48
      := TRUE;
   END_TRANSITION
   STEP GluePos_4:   // S116, max time T#10S, warning time T#7S
   END_STEP
   TRANSITION Trans132 FROM GluePos_4 TO "Servo returns toGluePos_4"   // T129
      := TRUE;
   END_TRANSITION
   STEP WaitIAIStop_2:   // S109, max time T#10S, warning time T#7S
   END_STEP
   STEP Axis_XToGluePos_3:   // S46, max time T#10S, warning time T#7S
      interlock C := NOT "IAI_DeviceCtl".IAIServo[#X_Axis].Point[5].Achieve;
      (C)     N    "IAI_DeviceCtl".IAIServo[#X_Axis].Point[5].Start
   END_STEP
   TRANSITION Trans54 FROM Axis_XToGluePos_3 TO CheckGlueSysOK_2   // T51
      := "IAI_DeviceCtl".IAIServo[#X_Axis].Point[5].Achieve;
   END_TRANSITION
   STEP CheckGlueSysOK_2:   // S47, max time T#10S, warning time T#7S
   END_STEP
   TRANSITION Trans55 FROM CheckGlueSysOK_2 TO GluePos_3   // T52
      := "GluingControl".Input.GluingDeviceReady OR "Station_Sys".Cmd.DryRun OR "ST10_GeneralData".FunctionDeSelect.C.FunctionDeSelected_Glue;
   END_TRANSITION
   STEP "Servo returns toGluePos_3":   // S48, max time T#10S, warning time T#7S
      (C)     N    "ServoV90_DeviceCtl".V90Servo[3].Point[4].Start
   END_STEP
   TRANSITION Trans56 FROM "Servo returns toGluePos_3" TO TimeDelay_3   // T53
      := "ServoV90_DeviceCtl".V90Servo[3].Point[4].Achieve;
   END_TRANSITION
   STEP Axis_XToGlueSafPos_3:   // S49, max time T#10S, warning time T#7S
      interlock C := NOT "IAI_DeviceCtl".IAIServo[#X_Axis].Point[2].Achieve;
      (C)     N    "IAI_DeviceCtl".IAIServo[#X_Axis].Point[2].Start
   END_STEP
   TRANSITION Trans57 FROM Axis_XToGlueSafPos_3 TO bypassGlue4   // T54
      := "IAI_DeviceCtl".IAIServo[#X_Axis].Point[2].Achieve;
   END_TRANSITION
   STEP Glue_3:   // S50, max time T#10S, warning time T#7S
   END_STEP
   TRANSITION Trans58 FROM Glue_3 TO Axis_XToGluePos_3   // T55
      := TRUE;
   END_TRANSITION
   STEP TimeDelay_3:   // S51, max time T#10S, warning time T#7S
   END_STEP
   TRANSITION Trans59 FROM TimeDelay_3 TO Axis_XToGlueSafPos_3   // T56
      := TRUE;
   END_TRANSITION
   STEP CameraCheck1:   // S118, max time T#10S, warning time T#7S
   END_STEP
   TRANSITION Trans134 FROM CameraCheck1 TO CheckIV3Ready   // T131
      := TRUE;
   END_TRANSITION
   STEP IAIMoveFinish_3:   // S111, max time T#10S, warning time T#7S
   END_STEP
   STEP Axis_XToGluePos_4:   // S54, max time T#10S, warning time T#7S
      interlock C := NOT "IAI_DeviceCtl".IAIServo[#X_Axis].Point[6].Achieve;
      (C)     N    "IAI_DeviceCtl".IAIServo[#X_Axis].Point[6].Start
   END_STEP
   TRANSITION Trans62 FROM Axis_XToGluePos_4 TO CheckGlueSysOK_3   // T59
      := "IAI_DeviceCtl".IAIServo[#X_Axis].Point[6].Achieve;
   END_TRANSITION
   STEP CheckGlueSysOK_3:   // S55, max time T#10S, warning time T#7S
   END_STEP
   TRANSITION Trans63 FROM CheckGlueSysOK_3 TO GluePos_4   // T60
      := "GluingControl".Input.GluingDeviceReady OR "Station_Sys".Cmd.DryRun OR "ST10_GeneralData".FunctionDeSelect.C.FunctionDeSelected_Glue;
   END_TRANSITION
   STEP "Servo returns toGluePos_4":   // S56, max time T#10S, warning time T#7S
      (C)     N    "ServoV90_DeviceCtl".V90Servo[3].Point[5].Start
   END_STEP
   TRANSITION Trans64 FROM "Servo returns toGluePos_4" TO ShaftGlueFinishStatus   // T61
      := "ServoV90_DeviceCtl".V90Servo[3].Point[5].Achieve;
   END_TRANSITION
   STEP Axis_XToGlueSafPos_4:   // S57, max time T#10S, warning time T#7S
      interlock C := NOT "IAI_DeviceCtl".IAIServo[#X_Axis].Point[2].Achieve;
      (C)     N    "IAI_DeviceCtl".IAIServo[#X_Axis].Point[2].Start
   END_STEP
   TRANSITION Trans65 FROM Axis_XToGlueSafPos_4 TO ServoHomePos_4   // T62
      := "IAI_DeviceCtl".IAIServo[#X_Axis].Point[2].Achieve;
   END_TRANSITION
   STEP Glue_4:   // S58, max time T#10S, warning time T#7S
   END_STEP
   TRANSITION Trans66 FROM Glue_4 TO Axis_XToGluePos_4   // T63
      := TRUE;
   END_TRANSITION
   STEP TimeDelay_4:   // S59, max time T#10S, warning time T#7S
   END_STEP
   TRANSITION Trans67 FROM TimeDelay_4 TO Axis_XToGlueSafPos_4   // T64
      := TRUE;
   END_TRANSITION
   STEP IV3Check:   // S60, max time T#10S, warning time T#7S
          S1  N    "DB_KeyenceCheckerIV3".aDev[2].Common.nMode:=1
   END_STEP
   TRANSITION Trans68 FROM IV3Check TO JudgeCheckStatus   // T65
      := ("DB_KeyenceCheckerIV3".aDev[2].Common.nMode = 0) AND NOT "DB_KeyenceCheckerIV3".aDev[2].Common.bError AND "DB_KeyenceCheckerIV3".aDev[2].Common.bDone;
   END_TRANSITION
   STEP JudgeCheckStatus:   // S61, max time T#10S, warning time T#7S
   END_STEP
   TRANSITION Trans69 FROM JudgeCheckStatus TO OKStatus   // T66
      := ("DB_KeyenceCheckerIV3".aDev[2].Para.bProductOverallOK AND NOT "DB_KeyenceCheckerIV3".aDev[2].Para.bProductOverallNG AND ("DB_KeyenceCheckerIV3".aDev[2].Para.nProgramNo = "DB_KeyenceCheckerIV3".aDev[2].In."DeviceStatus".nCurrentProgramNo)) OR "Station_Sys".Cmd.DryRun OR "ST10_GeneralData".FunctionDeSelect.C.FunctionDeSelected_Glue OR "ST10_GeneralData".FunctionDeSelect.C.FunctionDeSelected_IV3810A1;
   END_TRANSITION
   TRANSITION Trans70 FROM JudgeCheckStatus TO NGStatus   // T67
      := NOT "ST10_GeneralData".FunctionDeSelect.C.FunctionDeSelected_IV3810A1 AND NOT "ST10_GeneralData".FunctionDeSelect.C.FunctionDeSelected_Glue AND NOT "Station_Sys".Cmd.DryRun AND NOT "DB_KeyenceCheckerIV3".aDev[2].Para.bProductOverallOK AND "DB_KeyenceCheckerIV3".aDev[2].Para.bProductOverallNG AND ("DB_KeyenceCheckerIV3".aDev[2].Para.nProgramNo = "DB_KeyenceCheckerIV3".aDev[2].In."DeviceStatus".nCurrentProgramNo);
   END_TRANSITION
   STEP OKStatus:   // S62, max time T#10S, warning time T#7S
              N    "AutoProcessData".C_Glue.PartStatus:=310
              N    "Station5UnLoadData"."PLC.ShaftGlueIVScore1":="DB_KeyenceCheckerIV3".aDev[2].In.ToolResult[2].nToolMatchingRate
              N    "AutoProcessData".C_Glue.IV3_ShaftScore_1:="DB_KeyenceCheckerIV3".aDev[2].In.ToolResult[2].nToolMatchingRate
   END_STEP
   TRANSITION Trans71 FROM OKStatus TO CameraCheck2   // T68
      := "AutoProcessData".C_Glue.PartStatus = 310;
   END_TRANSITION
   STEP NGStatus:   // S63, max time T#10S, warning time T#7S
              N    "AutoProcessData".C_Glue.PartStatus:=359
              N    "Station5UnLoadData"."PLC.ShaftGlueIVScore1":="DB_KeyenceCheckerIV3".aDev[2].In.ToolResult[2].nToolMatchingRate
              N    "AutoProcessData".C_Glue.IV3_ShaftScore_1:="DB_KeyenceCheckerIV3".aDev[2].In.ToolResult[2].nToolMatchingRate
              N    "AutoProcessData".C_Glue.IV3_ShaftCheckResult:=2
   END_STEP
   TRANSITION Trans72 FROM NGStatus TO RobotGluePick   // T69, jump
      := "AutoProcessData".C_Glue.PartStatus = 359;
   END_TRANSITION
   STEP "C-LocationCylinderToHP2":   // S122, max time T#10S, warning time T#7S
              S    "ST10Cylinder".Cy[9].Inout.AutoGoHome
              R    "ST10Cylinder".Cy[9].Inout.AutoGoWork
   END_STEP
   TRANSITION Trans770 FROM "C-LocationCylinderToHP2" TO Glue_1   // T123
      := NOT "ST10Cylinder".Cy[9].In.WorkPositionSensor AND "ST10Cylinder".Cy[9].In.HomePositionSensor;
   END_TRANSITION
   STEP Step104:   // S104, max time T#10S, warning time T#7S
   END_STEP
   TRANSITION Trans121 FROM Step104 TO (Axis_ZToGlueePos_2, Axis_YToGlueePos_5)   // T115
      := TRUE;
   END_TRANSITION
   STEP WaitIAIStop_1:   // S106, max time T#10S, warning time T#7S
   END_STEP
   STEP Step110:   // S110, max time T#10S, warning time T#7S
   END_STEP
   TRANSITION Trans126 FROM Step110 TO (Axis_ZToGlueePos_4, Axis_YToGlueePos_7)   // T117
      := TRUE;
   END_TRANSITION
   STEP ShaftGlueFinishStatus:   // S68, max time T#10S, warning time T#7S
              N    "AutoProcessData".C_Glue.PartStatus:=300
   END_STEP
   TRANSITION Trans80 FROM ShaftGlueFinishStatus TO TimeDelay_4   // T77
      := "AutoProcessData".C_Glue.PartStatus = 300;
   END_TRANSITION
   STEP IAIMoveFinish:   // S95, max time T#10S, warning time T#7S
   END_STEP
   TRANSITION Trans115 FROM (WaitIAIStop, IAIMoveFinish) TO Axis_XToGluePos_1   // T114
      := TRUE;
   END_TRANSITION
   STEP Step102:   // S102, max time T#10S, warning time T#7S
   END_STEP
   TRANSITION Trans120 FROM Step102 TO Axis_YToGlueePos_1   // T113
      := TRUE;
   END_TRANSITION
   STEP Axis_YToGlueePos_1:   // S26, max time T#10S, warning time T#7S
      interlock C := NOT "IAI_DeviceCtl".IAIServo[#Y_axis].Point[2].Achieve;
      (C)     N    "IAI_DeviceCtl".IAIServo[#Y_axis].Point[2].Start
   END_STEP
   TRANSITION Trans36 FROM Axis_YToGlueePos_1 TO Axis_ZToGlueePos_1   // T31
      := "IAI_DeviceCtl".IAIServo[#Y_axis].Point[2].Achieve;
   END_TRANSITION
   STEP Axis_ZToGlueePos_1:   // S89, max time T#10S, warning time T#7S
      interlock C := NOT "IAI_DeviceCtl".IAIServo[#Z_Axis].Point[2].Achieve;
      (C)     N    "IAI_DeviceCtl".IAIServo[#Z_Axis].Point[2].Start
   END_STEP
   TRANSITION Trans108 FROM Axis_ZToGlueePos_1 TO IAIMoveFinish   // T99
      := "IAI_DeviceCtl".IAIServo[#Z_Axis].Point[2].Achieve;
   END_TRANSITION
   STEP Axis_ZToGlueePos_2:   // S35, max time T#10S, warning time T#7S
      interlock C := NOT "IAI_DeviceCtl".IAIServo[#Z_Axis].Point[3].Achieve;
      (C)     N    "IAI_DeviceCtl".IAIServo[#Z_Axis].Point[3].Start
   END_STEP
   TRANSITION Trans43 FROM Axis_ZToGlueePos_2 TO IAIMoveFinish_1   // T40
      := "IAI_DeviceCtl".IAIServo[#Z_Axis].Point[3].Achieve;
   END_TRANSITION
   STEP Step107:   // S107, max time T#10S, warning time T#7S
   END_STEP
   TRANSITION Trans122 FROM Step107 TO (Axis_ZToGlueePos_3, Axis_YToGlueePos_6)   // T108
      := TRUE;
   END_TRANSITION
   STEP IAIMoveFinish_2:   // S108, max time T#10S, warning time T#7S
   END_STEP
   STEP Axis_ZToGlueePos_3:   // S45, max time T#10S, warning time T#7S
      interlock C := NOT "IAI_DeviceCtl".IAIServo[#Z_Axis].Point[4].Achieve;
              N    "IAI_DeviceCtl".IAIServo[#Z_Axis].Point[4].Start
   END_STEP
   TRANSITION Trans53 FROM Axis_ZToGlueePos_3 TO IAIMoveFinish_2   // T50
      := "IAI_DeviceCtl".IAIServo[#Z_Axis].Point[4].Achieve;
   END_TRANSITION
   STEP Axis_ZToGlueePos_4:   // S53, max time T#10S, warning time T#7S
      interlock C := NOT "IAI_DeviceCtl".IAIServo[#Z_Axis].Point[5].Achieve;
      (C)     N    "IAI_DeviceCtl".IAIServo[#Z_Axis].Point[5].Start
   END_STEP
   TRANSITION Trans61 FROM Axis_ZToGlueePos_4 TO IAIMoveFinish_3   // T58
      := "IAI_DeviceCtl".IAIServo[#Z_Axis].Point[5].Achieve;
   END_TRANSITION
   STEP WaitIAIStop_3:   // S112, max time T#10S, warning time T#7S
   END_STEP
   STEP ServoHomePos:   // S94, max time T#10S, warning time T#7S
          S1  S    "ServoV90_A3".IO.ioAutoHome
   END_STEP
   TRANSITION Trans116 FROM ServoHomePos TO WaitIAIStop   // T109
      := ("ServoV90_A3".Out.oActPosition >= (-5)) AND ("ServoV90_A3".Out.oActPosition <= 5);
   END_TRANSITION
   STEP GluePos_1:   // S96, max time T#10S, warning time T#7S
   END_STEP
   TRANSITION Trans117 FROM GluePos_1 TO "Servo returns toGluePos_1"   // T110
      := TRUE;
   END_TRANSITION
   STEP ServoHomePos_1:   // S97, max time T#10S, warning time T#7S
          S1  S    "ServoV90_A3".IO.ioAutoHome
   END_STEP
   TRANSITION Trans118 FROM ServoHomePos_1 TO WaitIAIStop_1   // T111
      := ("ServoV90_A3".Out.oActPosition >= (-5)) AND ("ServoV90_A3".Out.oActPosition <= 5);
   END_TRANSITION
   STEP ServoHomePos_2:   // S113, max time T#10S, warning time T#7S
          S1  S    "ServoV90_A3".IO.ioAutoHome
   END_STEP
   TRANSITION Trans129 FROM ServoHomePos_2 TO WaitIAIStop_2   // T126
      := ("ServoV90_A3".Out.oActPosition >= (-5)) AND ("ServoV90_A3".Out.oActPosition <= 5);
   END_TRANSITION
   STEP ServoHomePos_3:   // S115, max time T#10S, warning time T#7S
          S1  S    "ServoV90_A3".IO.ioAutoHome
   END_STEP
   TRANSITION Trans131 FROM ServoHomePos_3 TO WaitIAIStop_3   // T128
      := ("ServoV90_A3".Out.oActPosition >= (-5)) AND ("ServoV90_A3".Out.oActPosition <= 5);
   END_TRANSITION
   STEP ServoHomePos_4:   // S117, max time T#10S, warning time T#7S
          S1  S    "ServoV90_A3".IO.ioAutoHome
   END_STEP
   TRANSITION Trans133 FROM ServoHomePos_4 TO ShaftGlueCameraCheck   // T130
      := ("ServoV90_A3".Out.oActPosition >= (-5)) AND ("ServoV90_A3".Out.oActPosition <= 5);
   END_TRANSITION
   STEP "Servo returns toGluePos_6":   // S125, max time T#10S, warning time T#7S
      (C)     N    "ServoV90_DeviceCtl".V90Servo[3].Point[7].Start
   END_STEP
   TRANSITION Trans135 FROM "Servo returns toGluePos_6" TO CheckIV3Ready_2   // T132
      := "ServoV90_DeviceCtl".V90Servo[3].Point[7].Achieve;
   END_TRANSITION
   STEP CheckIV3Ready_2:   // S206, max time T#10S, warning time T#7S
              N    "DB_KeyenceCheckerIV3".aDev[2].Para.nProgramNo:=1
   END_STEP
   TRANSITION Trans204 FROM CheckIV3Ready_2 TO IV3Check_2   // T206
      := "DB_KeyenceCheckerIV3".aDev[2].Common.bEnable AND NOT "DB_KeyenceCheckerIV3".aDev[2].Common.bError;
   END_TRANSITION
   STEP CameraCheck3:   // S131, max time T#10S, warning time T#7S
   END_STEP
   TRANSITION Trans140 FROM CameraCheck3 TO "Servo returns toGluePos_7"   // T137
      := TRUE;
   END_TRANSITION
   STEP IV3Check_2:   // S127, max time T#10S, warning time T#7S
          S1  N    "DB_KeyenceCheckerIV3".aDev[2].Common.nMode:=1
   END_STEP
   TRANSITION Trans137 FROM IV3Check_2 TO JudgeCheckStatus_2   // T134
      := ("DB_KeyenceCheckerIV3".aDev[2].Common.nMode = 0) AND NOT "DB_KeyenceCheckerIV3".aDev[2].Common.bError AND "DB_KeyenceCheckerIV3".aDev[2].Common.bDone;
   END_TRANSITION
   STEP JudgeCheckStatus_2:   // S128, max time T#10S, warning time T#7S
   END_STEP
   TRANSITION Trans138 FROM JudgeCheckStatus_2 TO OKStatus_2   // T135
      := ("DB_KeyenceCheckerIV3".aDev[2].Para.bProductOverallOK AND NOT "DB_KeyenceCheckerIV3".aDev[2].Para.bProductOverallNG AND ("DB_KeyenceCheckerIV3".aDev[2].Para.nProgramNo = "DB_KeyenceCheckerIV3".aDev[2].In."DeviceStatus".nCurrentProgramNo)) OR "Station_Sys".Cmd.DryRun OR "ST10_GeneralData".FunctionDeSelect.C.FunctionDeSelected_Glue OR "ST10_GeneralData".FunctionDeSelect.C.FunctionDeSelected_IV3810A1;
   END_TRANSITION
   TRANSITION Trans141 FROM JudgeCheckStatus_2 TO NGStatus_2   // T138
      := NOT "ST10_GeneralData".FunctionDeSelect.C.FunctionDeSelected_IV3810A1 AND NOT "ST10_GeneralData".FunctionDeSelect.C.FunctionDeSelected_Glue AND NOT "Station_Sys".Cmd.DryRun AND NOT "DB_KeyenceCheckerIV3".aDev[2].Para.bProductOverallOK AND "DB_KeyenceCheckerIV3".aDev[2].Para.bProductOverallNG AND ("DB_KeyenceCheckerIV3".aDev[2].Para.nProgramNo = "DB_KeyenceCheckerIV3".aDev[2].In."DeviceStatus".nCurrentProgramNo);
   END_TRANSITION
   STEP OKStatus_2:   // S129, max time T#10S, warning time T#7S
              N    "AutoProcessData".C_Glue.PartStatus:=310
              N    "Station5UnLoadData"."PLC.ShaftGlueIVScore2":="DB_KeyenceCheckerIV3".aDev[2].In.ToolResult[2].nToolMatchingRate
              N    "AutoProcessData".C_Glue.IV3_ShaftScore_2:="DB_KeyenceCheckerIV3".aDev[2].In.ToolResult[2].nToolMatchingRate
   END_STEP
   TRANSITION Trans139 FROM OKStatus_2 TO CameraCheck3   // T136
      := "AutoProcessData".C_Glue.PartStatus = 310;
   END_TRANSITION
   STEP CameraCheck2:   // S126, max time T#10S, warning time T#7S
   END_STEP
   TRANSITION Trans136 FROM CameraCheck2 TO "Servo returns toGluePos_6"   // T133
      := TRUE;
   END_TRANSITION
   STEP NGStatus_2:   // S130, max time T#10S, warning time T#7S
              N    "AutoProcessData".C_Glue.PartStatus:=359
              N    "Station5UnLoadData"."PLC.ShaftGlueIVScore2":="DB_KeyenceCheckerIV3".aDev[2].In.ToolResult[2].nToolMatchingRate
              N    "AutoProcessData".C_Glue.IV3_ShaftScore_2:="DB_KeyenceCheckerIV3".aDev[2].In.ToolResult[2].nToolMatchingRate
              N    "AutoProcessData".C_Glue.IV3_ShaftCheckResult:=2
   END_STEP
   TRANSITION Trans142 FROM NGStatus_2 TO RobotGluePick   // T139, jump
      := "AutoProcessData".C_Glue.PartStatus = 359;
   END_TRANSITION
   STEP "Servo returns toGluePos_7":   // S132, max time T#10S, warning time T#7S
      (C)     N    "ServoV90_DeviceCtl".V90Servo[3].Point[8].Start
   END_STEP
   TRANSITION Trans143 FROM "Servo returns toGluePos_7" TO CheckIV3Ready_3   // T140
      := "ServoV90_DeviceCtl".V90Servo[3].Point[8].Achieve;
   END_TRANSITION
   STEP CheckIV3Ready_3:   // S207, max time T#10S, warning time T#7S
              N    "DB_KeyenceCheckerIV3".aDev[2].Para.nProgramNo:=1
   END_STEP
   TRANSITION Trans207 FROM CheckIV3Ready_3 TO IV3Check_3   // T207
      := "DB_KeyenceCheckerIV3".aDev[2].Common.bEnable AND NOT "DB_KeyenceCheckerIV3".aDev[2].Common.bError;
   END_TRANSITION
   STEP IV3Check_3:   // S133, max time T#10S, warning time T#7S
          S1  N    "DB_KeyenceCheckerIV3".aDev[2].Common.nMode:=1
   END_STEP
   TRANSITION Trans144 FROM IV3Check_3 TO JudgeCheckStatus_3   // T141
      := ("DB_KeyenceCheckerIV3".aDev[2].Common.nMode = 0) AND NOT "DB_KeyenceCheckerIV3".aDev[2].Common.bError AND "DB_KeyenceCheckerIV3".aDev[2].Common.bDone;
   END_TRANSITION
   STEP JudgeCheckStatus_3:   // S134, max time T#10S, warning time T#7S
   END_STEP
   TRANSITION Trans145 FROM JudgeCheckStatus_3 TO OKStatus_3   // T142
      := ("DB_KeyenceCheckerIV3".aDev[2].Para.bProductOverallOK AND NOT "DB_KeyenceCheckerIV3".aDev[2].Para.bProductOverallNG AND ("DB_KeyenceCheckerIV3".aDev[2].Para.nProgramNo = "DB_KeyenceCheckerIV3".aDev[2].In."DeviceStatus".nCurrentProgramNo)) OR "Station_Sys".Cmd.DryRun OR "ST10_GeneralData".FunctionDeSelect.C.FunctionDeSelected_Glue OR "ST10_GeneralData".FunctionDeSelect.C.FunctionDeSelected_IV3810A1;
   END_TRANSITION
   TRANSITION Trans148 FROM JudgeCheckStatus_3 TO NGStatus_3   // T145
      := NOT "ST10_GeneralData".FunctionDeSelect.C.FunctionDeSelected_IV3810A1 AND NOT "ST10_GeneralData".FunctionDeSelect.C.FunctionDeSelected_Glue AND NOT "Station_Sys".Cmd.DryRun AND NOT "DB_KeyenceCheckerIV3".aDev[2].Para.bProductOverallOK AND "DB_KeyenceCheckerIV3".aDev[2].Para.bProductOverallNG AND ("DB_KeyenceCheckerIV3".aDev[2].Para.nProgramNo = "DB_KeyenceCheckerIV3".aDev[2].In."DeviceStatus".nCurrentProgramNo);
   END_TRANSITION
   STEP OKStatus_3:   // S135, max time T#10S, warning time T#7S
              N    "AutoProcessData".C_Glue.PartStatus:=310
              N    "Station5UnLoadData"."PLC.ShaftGlueIVScore3":="DB_KeyenceCheckerIV3".aDev[2].In.ToolResult[2].nToolMatchingRate
              N    "AutoProcessData".C_Glue.IV3_ShaftScore_3:="DB_KeyenceCheckerIV3".aDev[2].In.ToolResult[2].nToolMatchingRate
   END_STEP
   TRANSITION Trans146 FROM OKStatus_3 TO CameraCheck4   // T143
      := "AutoProcessData".C_Glue.PartStatus = 310;
   END_TRANSITION
   STEP CameraCheck4:   // S137, max time T#10S, warning time T#7S
   END_STEP
   TRANSITION Trans147 FROM CameraCheck4 TO "Servo returns toGluePos_8"   // T144
      := TRUE;
   END_TRANSITION
   STEP NGStatus_3:   // S136, max time T#10S, warning time T#7S
              N    "AutoProcessData".C_Glue.PartStatus:=359
              N    "Station5UnLoadData"."PLC.ShaftGlueIVScore3":="DB_KeyenceCheckerIV3".aDev[2].In.ToolResult[2].nToolMatchingRate
              N    "AutoProcessData".C_Glue.IV3_ShaftScore_3:="DB_KeyenceCheckerIV3".aDev[2].In.ToolResult[2].nToolMatchingRate
              N    "AutoProcessData".C_Glue.IV3_ShaftCheckResult:=2
   END_STEP
   TRANSITION Trans149 FROM NGStatus_3 TO RobotGluePick   // T146, jump
      := "AutoProcessData".C_Glue.PartStatus = 359;
   END_TRANSITION
   STEP "Servo returns toGluePos_8":   // S138, max time T#10S, warning time T#7S
      (C)     N    "ServoV90_DeviceCtl".V90Servo[3].Point[9].Start
   END_STEP
   TRANSITION Trans150 FROM "Servo returns toGluePos_8" TO CheckIV3Ready_4   // T147
      := "ServoV90_DeviceCtl".V90Servo[3].Point[9].Achieve;
   END_TRANSITION
   STEP CheckIV3Ready_4:   // S208, max time T#10S, warning time T#7S
              N    "DB_KeyenceCheckerIV3".aDev[2].Para.nProgramNo:=1
   END_STEP
   TRANSITION Trans208 FROM CheckIV3Ready_4 TO IV3Check_4   // T208
      := "DB_KeyenceCheckerIV3".aDev[2].Common.bEnable AND NOT "DB_KeyenceCheckerIV3".aDev[2].Common.bError;
   END_TRANSITION
   STEP IV3Check_4:   // S139, max time T#10S, warning time T#7S
          S1  N    "DB_KeyenceCheckerIV3".aDev[2].Common.nMode:=1
   END_STEP
   TRANSITION Trans151 FROM IV3Check_4 TO JudgeCheckStatus_4   // T148
      := ("DB_KeyenceCheckerIV3".aDev[2].Common.nMode = 0) AND NOT "DB_KeyenceCheckerIV3".aDev[2].Common.bError AND "DB_KeyenceCheckerIV3".aDev[2].Common.bDone;
   END_TRANSITION
   STEP JudgeCheckStatus_4:   // S140, max time T#10S, warning time T#7S
   END_STEP
   TRANSITION Trans152 FROM JudgeCheckStatus_4 TO OKStatus_4   // T698
      := ("DB_KeyenceCheckerIV3".aDev[2].Para.bProductOverallOK AND NOT "DB_KeyenceCheckerIV3".aDev[2].Para.bProductOverallNG AND ("DB_KeyenceCheckerIV3".aDev[2].Para.nProgramNo = "DB_KeyenceCheckerIV3".aDev[2].In."DeviceStatus".nCurrentProgramNo)) OR "Station_Sys".Cmd.DryRun OR "ST10_GeneralData".FunctionDeSelect.C.FunctionDeSelected_Glue OR "ST10_GeneralData".FunctionDeSelect.C.FunctionDeSelected_IV3810A1;
   END_TRANSITION
   TRANSITION Trans155 FROM JudgeCheckStatus_4 TO NGStatus_4   // T152
      := NOT "ST10_GeneralData".FunctionDeSelect.C.FunctionDeSelected_IV3810A1 AND NOT "ST10_GeneralData".FunctionDeSelect.C.FunctionDeSelected_Glue AND NOT "Station_Sys".Cmd.DryRun AND NOT "DB_KeyenceCheckerIV3".aDev[2].Para.bProductOverallOK AND "DB_KeyenceCheckerIV3".aDev[2].Para.bProductOverallNG AND ("DB_KeyenceCheckerIV3".aDev[2].Para.nProgramNo = "DB_KeyenceCheckerIV3".aDev[2].In."DeviceStatus".nCurrentProgramNo);
   END_TRANSITION
   STEP OKStatus_4:   // S141, max time T#10S, warning time T#7S
              N    "AutoProcessData".C_Glue.PartStatus:=310
              N    "Station5UnLoadData"."PLC.ShaftGlueIVScore4":="DB_KeyenceCheckerIV3".aDev[2].In.ToolResult[2].nToolMatchingRate
              N    "AutoProcessData".C_Glue.IV3_ShaftScore_4:="DB_KeyenceCheckerIV3".aDev[2].In.ToolResult[2].nToolMatchingRate
              N    "AutoProcessData".C_Glue.IV3_ShaftCheckResult:=1
   END_STEP
   TRANSITION Trans153 FROM OKStatus_4 TO "Total Score of Shaft Gluening check"   // T645
      := "AutoProcessData".C_Glue.PartStatus = 310;
   END_TRANSITION
   STEP NGStatus_4:   // S142, max time T#10S, warning time T#7S
              N    "AutoProcessData".C_Glue.PartStatus:=359
              N    "Station5UnLoadData"."PLC.ShaftGlueIVScore4":="DB_KeyenceCheckerIV3".aDev[2].In.ToolResult[2].nToolMatchingRate
              N    "AutoProcessData".C_Glue.IV3_ShaftScore_4:="DB_KeyenceCheckerIV3".aDev[2].In.ToolResult[2].nToolMatchingRate
              N    "AutoProcessData".C_Glue.IV3_ShaftCheckResult:=2
   END_STEP
   TRANSITION Trans156 FROM NGStatus_4 TO RobotGluePick   // T153, jump
      := "AutoProcessData".C_Glue.PartStatus = 359;
   END_TRANSITION
   STEP Axis_YToGlueePos_5:   // S41, max time T#10S, warning time T#7S
      interlock C := NOT "IAI_DeviceCtl".IAIServo[#Y_axis].Point[3].Achieve;
              N    "IAI_DeviceCtl".IAIServo[#Y_axis].Point[3].Start
   END_STEP
   TRANSITION Trans49 FROM Axis_YToGlueePos_5 TO "IAIMoveFinish_ 1"   // T46
      := "IAI_DeviceCtl".IAIServo[#Y_axis].Point[3].Achieve;
   END_TRANSITION
   STEP "IAIMoveFinish_ 1":   // S153, max time T#10S, warning time T#7S
   END_STEP
   TRANSITION Trans114 FROM (WaitIAIStop_1, IAIMoveFinish_1, "IAIMoveFinish_ 1") TO Glue_2   // T107
      := TRUE;
   END_TRANSITION
   STEP IAIMoveFinish_4:   // S155, max time T#10S, warning time T#7S
   END_STEP
   TRANSITION Trans123 FROM (WaitIAIStop_2, IAIMoveFinish_2, IAIMoveFinish_4) TO Glue_3   // T116
      := TRUE;
   END_TRANSITION
   STEP Axis_YToGlueePos_6:   // S52, max time T#10S, warning time T#7S
      interlock C := NOT "IAI_DeviceCtl".IAIServo[#Y_axis].Point[4].Achieve;
              N    "IAI_DeviceCtl".IAIServo[#Y_axis].Point[4].Start
   END_STEP
   TRANSITION Trans60 FROM Axis_YToGlueePos_6 TO IAIMoveFinish_4   // T57
      := "IAI_DeviceCtl".IAIServo[#Y_axis].Point[4].Achieve;
   END_TRANSITION
   STEP IAIMoveFinish_5:   // S154, max time T#10S, warning time T#7S
   END_STEP
   TRANSITION Trans127 FROM (WaitIAIStop_3, IAIMoveFinish_3, IAIMoveFinish_5) TO Glue_4   // T118
      := TRUE;
   END_TRANSITION
   STEP Axis_YToGlueePos_7:   // S88, max time T#10S, warning time T#7S
      interlock C := NOT "IAI_DeviceCtl".IAIServo[#Y_axis].Point[5].Achieve;
              N    "IAI_DeviceCtl".IAIServo[#Y_axis].Point[5].Start
   END_STEP
   TRANSITION Trans107 FROM Axis_YToGlueePos_7 TO IAIMoveFinish_5   // T86
      := "IAI_DeviceCtl".IAIServo[#Y_axis].Point[5].Achieve;
   END_TRANSITION
   STEP bypassGlue4:   // S162, max time T#10S, warning time T#7S
   END_STEP
   TRANSITION bypassTRUE FROM bypassGlue4 TO ShaftGlueFinishStatus   // T168
      := "AlwaysTRUE";
   END_TRANSITION
   TRANSITION bypassFALSE FROM bypassGlue4 TO (Step110, ServoHomePos_3)   // T166
      := "AlwaysFALSE";
   END_TRANSITION

   // sequencer 5: S300-S349 RobotPutMagnet
   STEP RobotPutMagnet:   // S300, max time T#10S, warning time T#7S
   END_STEP
   TRANSITION Trans291 FROM RobotPutMagnet TO ServoJoging   // T300
      := TRUE;
   END_TRANSITION
   STEP MaganetGlue:   // S320, max time T#10S, warning time T#7S
   END_STEP
   TRANSITION Trans301 FROM MaganetGlue TO JudgeYPosition   // T320
      := TRUE;
   END_TRANSITION
   STEP RequestRobotPutMagnet_1:   // S281, max time T#10S, warning time T#7S
              N    "AutoProcessControl".C_Glue.Robot2MaganePutPrimit
   END_STEP
   TRANSITION Trans81 FROM RequestRobotPutMagnet_1 TO WaitRobotFinishTask_1   // T281
      := "KukaRobot2_CtrlDB".sROBtoPLC.User.Cycle.DO265_GluePutInside AND NOT "KukaRobot2_CtrlDB".sROBtoPLC.User.Cycle.DO266_GluePutFinish;
   END_TRANSITION
   STEP WaitRobotFinishTask_1:   // S288, max time T#10S, warning time T#7S
   END_STEP
   TRANSITION Trans82 FROM WaitRobotFinishTask_1 TO StopServoJoging   // T288
      := "KukaRobot2_CtrlDB".sROBtoPLC.User.Cycle.DO266_GluePutFinish;
   END_TRANSITION
   STEP CheckIV3Ready_1:   // S204, max time T#10S, warning time T#7S
              N    "DB_KeyenceCheckerIV3".aDev[1].Para.nProgramNo:=1
   END_STEP
   TRANSITION Trans205 FROM CheckIV3Ready_1 TO IV3Check_1   // T204
      := "DB_KeyenceCheckerIV3".aDev[1].Common.bEnable AND NOT "DB_KeyenceCheckerIV3".aDev[1].Common.bError;
   END_TRANSITION
   STEP Axis_ZToIVCheckPos:   // S78, max time T#10S, warning time T#7S
      interlock C := NOT "IAI_DeviceCtl".IAIServo[#Z_Axis].Point[7].Achieve;
      (C)     N    "IAI_DeviceCtl".IAIServo[#Z_Axis].Point[7].Start
   END_STEP
   TRANSITION Trans31 FROM Axis_ZToIVCheckPos TO (Axis_XYIVCheckPos, Axis_XYIVCheckPos_1)   // T87
      := "IAI_DeviceCtl".IAIServo[#Z_Axis].Point[7].Achieve;
   END_TRANSITION
   STEP CheckGlueSysOK_4:   // S72, max time T#10S, warning time T#7S
   END_STEP
   TRANSITION Trans86 FROM CheckGlueSysOK_4 TO "Servo returns toGluePos_5"   // T81
      := "GluingControl".Input.GluingDeviceReady OR "Station_Sys".Cmd.DryRun OR "ST10_GeneralData".FunctionDeSelect.C.FunctionDeSelected_Glue;
   END_TRANSITION
   STEP "Servo returns toGluePos_5":   // S73, max time T#10S, warning time T#7S
      (C)     N    "ServoV90_DeviceCtl".V90Servo[3].Point[6].Start
   END_STEP
   TRANSITION Trans87 FROM "Servo returns toGluePos_5" TO TimeDelay_5   // T82
      := "ServoV90_DeviceCtl".V90Servo[3].Point[6].Achieve;
   END_TRANSITION
   STEP ServoJoging:   // S123, max time T#10S, warning time T#7S
   END_STEP
   TRANSITION Trans124 FROM ServoJoging TO RequestRobotPutMagnet_1   // T124
      := NOT "AutoProcessControl".C_Glue.GlueTest;
   END_TRANSITION
   TRANSITION Trans306 FROM ServoJoging TO MaganetGlue   // T306
      := "AutoProcessControl".C_Glue.GlueTest AND "iHMI ResetButton" AND "iHMI Machine Start";
   END_TRANSITION
   STEP Axis_YToGluePos_5:   // S75, max time T#10S, warning time T#7S
      interlock C := NOT "IAI_DeviceCtl".IAIServo[#Y_axis].Point[6].Achieve;
      (C)     N    "IAI_DeviceCtl".IAIServo[#Y_axis].Point[6].Start
   END_STEP
   TRANSITION Trans89 FROM Axis_YToGluePos_5 TO Axis_XToGluePos_5   // T84
      := "IAI_DeviceCtl".IAIServo[#Y_axis].Point[6].Achieve;
   END_TRANSITION
   STEP TimeDelay_5:   // S76, max time T#10S, warning time T#7S
   END_STEP
   TRANSITION Trans90 FROM TimeDelay_5 TO GlueFinishStatus   // T85
      := TRUE;
   END_TRANSITION
   STEP MagnetGlueFinish:   // S349, max time T#10S, warning time T#7S
   END_STEP
   TRANSITION Trans91 FROM MagnetGlueFinish TO "MES  Check Result"   // T349, jump
      := TRUE;
   END_TRANSITION
   STEP Axis_XToGluePos_5:   // S71, max time T#10S, warning time T#7S
      interlock C := NOT "IAI_DeviceCtl".IAIServo[#X_Axis].Point[7].Achieve;
      (C)     N    "IAI_DeviceCtl".IAIServo[#X_Axis].Point[7].Start
   END_STEP
   TRANSITION Trans85 FROM Axis_XToGluePos_5 TO Axis_ZToGlueePos_5   // T80
      := "IAI_DeviceCtl".IAIServo[#X_Axis].Point[7].Achieve;
   END_TRANSITION
   STEP Axis_XYIVCheckPos:   // S79, max time T#10S, warning time T#7S
      interlock C := NOT "IAI_DeviceCtl".IAIServo[#X_Axis].Point[8].Achieve;
      (C)     N    "IAI_DeviceCtl".IAIServo[#X_Axis].Point[8].Start
   END_STEP
   TRANSITION Trans32 FROM Axis_XYIVCheckPos TO Step159   // T88
      := "IAI_DeviceCtl".IAIServo[#X_Axis].Point[8].Achieve;
   END_TRANSITION
   STEP GlueFinishStatus:   // S83, max time T#10S, warning time T#7S
              N    "AutoProcessData".C_Glue.PartStatus:=330
   END_STEP
   TRANSITION Trans95 FROM GlueFinishStatus TO "IV3 Check"   // T92
      := "AutoProcessData".C_Glue.PartStatus = 330;
   END_TRANSITION
   STEP "IV3 Check":   // S630, max time T#10S, warning time T#7S
   END_STEP
   TRANSITION Trans96 FROM "IV3 Check" TO Axis_ZToIVCheckPos   // T630
      := TRUE;
   END_TRANSITION
   STEP Step204:   // S205, max time T#10S, warning time T#7S
   END_STEP
   TRANSITION Trans206 FROM Step204 TO MagnetGlueFinish   // T205
      := TRUE;
   END_TRANSITION
   STEP IV3Check_1:   // S69, max time T#10S, warning time T#7S
          S1  N    "DB_KeyenceCheckerIV3".aDev[1].Common.nMode:=1
   END_STEP
   TRANSITION Trans83 FROM IV3Check_1 TO JudgeCheckStatus_1   // T78
      := ("DB_KeyenceCheckerIV3".aDev[1].Common.nMode = 0) AND NOT "DB_KeyenceCheckerIV3".aDev[1].Common.bError AND "DB_KeyenceCheckerIV3".aDev[1].Common.bDone;
   END_TRANSITION
   STEP JudgeCheckStatus_1:   // S74, max time T#10S, warning time T#7S
   END_STEP
   TRANSITION Trans88 FROM JudgeCheckStatus_1 TO OKStatus_1   // T83
      := ("DB_KeyenceCheckerIV3".aDev[1].Para.bProductOverallOK AND NOT "DB_KeyenceCheckerIV3".aDev[1].Para.bProductOverallNG AND ("DB_KeyenceCheckerIV3".aDev[1].Para.nProgramNo = "DB_KeyenceCheckerIV3".aDev[1].In."DeviceStatus".nCurrentProgramNo)) OR "Station_Sys".Cmd.DryRun OR "ST10_GeneralData".FunctionDeSelect.C.FunctionDeSelected_Glue OR "ST10_GeneralData".FunctionDeSelect.C.FunctionDeSelected_IV3811A1;
   END_TRANSITION
   TRANSITION Trans97 FROM JudgeCheckStatus_1 TO NGStatus_1   // T93
      := NOT "ST10_GeneralData".FunctionDeSelect.C.FunctionDeSelected_IV3811A1 AND NOT "ST10_GeneralData".FunctionDeSelect.C.FunctionDeSelected_Glue AND NOT "DB_KeyenceCheckerIV3".aDev[1].Para.bProductOverallOK AND NOT "Station_Sys".Cmd.DryRun AND "DB_KeyenceCheckerIV3".aDev[1].Para.bProductOverallNG AND ("DB_KeyenceCheckerIV3".aDev[1].Para.nProgramNo = "DB_KeyenceCheckerIV3".aDev[1].In."DeviceStatus".nCurrentProgramNo);
   END_TRANSITION
   STEP OKStatus_1:   // S84, max time T#10S, warning time T#7S
              N    "AutoProcessData".C_Glue.PartStatus:=380
              N    "Station5UnLoadData"."PLC.MagnetIVScore":="DB_KeyenceCheckerIV3".aDev[1].In.ToolResult[2].nToolMatchingRate
              N    "AutoProcessData".C_Glue.IV3_MagnetScore:="DB_KeyenceCheckerIV3".aDev[1].In.ToolResult[2].nToolMatchingRate
              N    "AutoProcessData".C_Glue.IV3_MagnetCheckResult:=1
   END_STEP
   TRANSITION Trans98 FROM OKStatus_1 TO Step204   // T94
      := "AutoProcessData".C_Glue.PartStatus = 380;
   END_TRANSITION
   STEP NGStatus_1:   // S85, max time T#10S, warning time T#7S
              N    "AutoProcessData".C_Glue.PartStatus:=358
              N    "Station5UnLoadData"."PLC.MagnetIVScore":="DB_KeyenceCheckerIV3".aDev[1].In.ToolResult[1].nToolMatchingRate
              N    "AutoProcessData".C_Glue.IV3_MagnetScore:="DB_KeyenceCheckerIV3".aDev[1].In.ToolResult[1].nToolMatchingRate
              N    "AutoProcessData".C_Glue.IV3_MagnetCheckResult:=2
   END_STEP
   TRANSITION Trans99 FROM NGStatus_1 TO Step204   // T95
      := "AutoProcessData".C_Glue.PartStatus = 358;
   END_TRANSITION
   STEP StopServoJoging:   // S124, max time T#10S, warning time T#7S
   END_STEP
   TRANSITION Trans125 FROM StopServoJoging TO MaganetGlue   // T125
      := TRUE;
   END_TRANSITION
   STEP JudgeYPosition:   // S90, max time T#10S, warning time T#7S
   END_STEP
   TRANSITION Trans109 FROM JudgeYPosition TO Axis_ZToGlueePos_7   // T102
      := "Axis_FB_DB".IAI_Axis[3].RecvData."Input 4 word_1"."Current Position" < 20000;
   END_TRANSITION
   TRANSITION Trans110 FROM JudgeYPosition TO Axis_YToGluePos_6   // T103
      := "Axis_FB_DB".IAI_Axis[3].RecvData."Input 4 word_1"."Current Position" >= 20000;
   END_TRANSITION
   STEP Axis_YToGluePos_6:   // S91, max time T#10S, warning time T#7S
      interlock C := NOT "IAI_DeviceCtl".IAIServo[#Y_axis].Point[6].Achieve;
      (C)     N    "IAI_DeviceCtl".IAIServo[#Y_axis].Point[6].Start
   END_STEP
   TRANSITION Trans111 FROM Axis_YToGluePos_6 TO Axis_XToGluePos_6   // T104
      := "IAI_DeviceCtl".IAIServo[#Y_axis].Point[6].Achieve;
   END_TRANSITION
   STEP Axis_XToGluePos_6:   // S92, max time T#10S, warning time T#7S
      interlock C := NOT "IAI_DeviceCtl".IAIServo[#X_Axis].Point[7].Achieve;
      (C)     N    "IAI_DeviceCtl".IAIServo[#X_Axis].Point[7].Start
   END_STEP
   TRANSITION Trans112 FROM Axis_XToGluePos_6 TO Axis_ZToGlueePos_6   // T105
      := "IAI_DeviceCtl".IAIServo[#X_Axis].Point[7].Achieve;
   END_TRANSITION
   STEP Axis_ZToGlueePos_6:   // S93, max time T#10S, warning time T#7S
      interlock C := NOT "IAI_DeviceCtl".IAIServo[#Z_Axis].Point[6].Achieve;
      (C)     N    "IAI_DeviceCtl".IAIServo[#Z_Axis].Point[6].Start
   END_STEP
   TRANSITION Trans113 FROM Axis_ZToGlueePos_6 TO ServoHomePos_5   // T106
      := "IAI_DeviceCtl".IAIServo[#Z_Axis].Point[6].Achieve;
   END_TRANSITION
   STEP ServoHomePos_5:   // S143, max time T#10S, warning time T#7S
          S1  S    "ServoV90_A3".IO.ioAutoHome
   END_STEP
   TRANSITION Trans154 FROM ServoHomePos_5 TO CheckGlueSysOK_4   // T151
      := ("ServoV90_A3".Out.oActPosition >= (-5)) AND ("ServoV90_A3".Out.oActPosition <= 5);
   END_TRANSITION
   STEP Axis_ZToGlueePos_5:   // S70, max time T#10S, warning time T#7S
      interlock C := NOT "IAI_DeviceCtl".IAIServo[#Z_Axis].Point[6].Achieve;
      (C)     N    "IAI_DeviceCtl".IAIServo[#Z_Axis].Point[6].Start
   END_STEP
   TRANSITION Trans84 FROM Axis_ZToGlueePos_5 TO ServoHomePos_5   // T79
      := "IAI_DeviceCtl".IAIServo[#Z_Axis].Point[6].Achieve;
   END_TRANSITION
   STEP Axis_ZToGlueePos_7:   // S148, max time T#10S, warning time T#7S
      interlock C := NOT "IAI_DeviceCtl".IAIServo[#Z_Axis].Point[9].Achieve;
      (C)     N    "IAI_DeviceCtl".IAIServo[#Z_Axis].Point[9].Start
   END_STEP
   TRANSITION Trans160 FROM Axis_ZToGlueePos_7 TO Axis_YToGluePos_5   // T157
      := "IAI_DeviceCtl".IAIServo[#Z_Axis].Point[9].Achieve;
   END_TRANSITION
   STEP Step158:   // S158, max time T#10S, warning time T#7S
   END_STEP
   TRANSITION Trans167 FROM (Step159, Step158) TO CheckIV3Ready_1   // T163
      := TRUE;
   END_TRANSITION
   STEP Axis_XYIVCheckPos_1:   // S157, max time T#10S, warning time T#7S
      interlock C := NOT "IAI_DeviceCtl".IAIServo[#Y_axis].Point[7].Achieve;
      (C)     N    "IAI_DeviceCtl".IAIServo[#Y_axis].Point[7].Start
   END_STEP
   TRANSITION Trans42 FROM Axis_XYIVCheckPos_1 TO Step158   // T98
      := "IAI_DeviceCtl".IAIServo[#Y_axis].Point[7].Achieve;
   END_TRANSITION
   STEP Step159:   // S159, max time T#10S, warning time T#7S
   END_STEP

   // sequencer 6: S350-S399 MES Check Result
   STEP "MES  Check Result":   // S350, max time T#10S, warning time T#7S
   END_STEP
   TRANSITION Trans162 FROM "MES  Check Result" TO Bypass_1   // T158
      := TRUE;
   END_TRANSITION
   STEP "MES Check OK_1":   // S399, max time T#10S, warning time T#7S
   END_STEP
   TRANSITION Trans311 FROM "MES Check OK_1" TO RobotGluePick   // T399, jump
      := TRUE;
   END_TRANSITION
   STEP ResetMesCheckRequest_1:   // S302, max time T#10S, warning time T#7S
              R    "PLCtoMES"."PLC.Load_Station5ChickInReq"
              R    "MEStoPLC"."MES.Load_Station5PartOK"
              R    "MEStoPLC"."MES.Load_Station5PartNG"
              R    "MEStoPLC"."MES.Load_Station5ReqMesDone"
              R    "MEStoPLC"."MES.Unload_ResultsStored5OK"
              R    "MEStoPLC"."MES.Unload_ResultsStored5ReqMesDone"
   END_STEP
   TRANSITION Trans260 FROM ResetMesCheckRequest_1 TO "Prepare MES CheckData_1"   // T313
      := NOT "PLCtoMES"."PLC.Load_Station5ChickInReq" AND NOT "MEStoPLC"."MES.Load_Station5PartOK" AND NOT "MEStoPLC"."MES.Load_Station5PartNG" AND NOT "MEStoPLC"."MES.Load_Station5ReqMesDone" AND NOT "MEStoPLC"."MES.Unload_ResultsStored5ReqMesDone" AND NOT "MEStoPLC"."MES.Unload_ResultsStored5OK";
   END_TRANSITION
   STEP ok:   // S311, max time T#10S, warning time T#7S
      interlock C := "AutoProcessData".C_Glue.PartStatus = 399;
              N    "AutoProcessData".C_Glue.PartStatus:=399
   END_STEP
   TRANSITION Trans315 FROM ok TO "MES Check OK_1"   // T312
      := #ok.T > t#200MS;
   END_TRANSITION
   STEP "Prepare MES CheckData_1":   // S307, max time T#10S, warning time T#7S
   END_STEP
   TRANSITION Trans15 FROM "Prepare MES CheckData_1" TO MESSaveRequest_1   // T308
      := #"Prepare MES CheckData_1".T > t#300MS;
   END_TRANSITION
   STEP MESSaveRequest_1:   // S313, max time T#10S, warning time T#7S
      interlock C := "AutoProcessData".C_Glue.PartStatus = 380;
              N    "PLCtoMES"."PLC.Unload_Station5DataSaveReq"
   END_STEP
   TRANSITION Trans266 FROM MESSaveRequest_1 TO ok   // T319
      := "MEStoPLC"."MES.Unload_ResultsStored5OK" AND NOT "MEStoPLC"."MES.Unload_ResultsStored5NG" AND "MEStoPLC"."MES.Unload_ResultsStored5ReqMesDone" AND (("AutoProcessData".C_Glue.PartStatus < 350) OR ("AutoProcessData".C_Glue.PartStatus > 360));
   END_TRANSITION
   TRANSITION Trans312 FROM MESSaveRequest_1 TO MESOverTime   // T328
      := #MESSaveRequest_1.T > t#10S;
   END_TRANSITION
   TRANSITION Trans319 FROM MESSaveRequest_1 TO ResultNG   // T332
      := NOT "MEStoPLC"."MES.Unload_ResultsStored5OK" AND "MEStoPLC"."MES.Unload_ResultsStored5NG" AND "MEStoPLC"."MES.Unload_ResultsStored5ReqMesDone";
   END_TRANSITION
   TRANSITION Trans171 FROM MESSaveRequest_1 TO "MES Check OK_1"   // T169
      := "MEStoPLC"."MES.Unload_ResultsStored5OK" AND NOT "MEStoPLC"."MES.Unload_ResultsStored5NG" AND "MEStoPLC"."MES.Unload_ResultsStored5ReqMesDone" AND ("AutoProcessData".C_Glue.PartStatus >= 350) AND ("AutoProcessData".C_Glue.PartStatus <= 360);
   END_TRANSITION
   STEP MESOverTime:   // S323, max time T#10S, warning time T#7S
              S    "ST10_DeviceError".MES_Error.CheckInResultOverTime_5
   END_STEP
   TRANSITION Trans313 FROM MESOverTime TO Bypass_1   // T329, jump
      := #iSysInface.Reset;
   END_TRANSITION
   STEP Bypass_1:   // S324, max time T#10S, warning time T#7S
   END_STEP
   TRANSITION Online_1 FROM Bypass_1 TO ResetMesCheckRequest_1   // T304
      := NOT "Station_Sys".Cmd.OnOffLine;
   END_TRANSITION
   TRANSITION Offline_1 FROM Bypass_1 TO ok_1   // T14
      := "Station_Sys".Cmd.OnOffLine;
   END_TRANSITION
   STEP ResultNG:   // S326, max time T#10S, warning time T#7S
              N    "AutoProcessData".C_Glue.PartStatus:=352
   END_STEP
   TRANSITION Trans321 FROM ResultNG TO "MES Check OK_1"   // T333
      := "AutoProcessData".C_Glue.PartStatus = 352;
   END_TRANSITION
   STEP Step315:   // S328, max time T#10S, warning time T#7S
   END_STEP
   TRANSITION Trans326 FROM Step315 TO "MES Check OK_1"   // T335
      := TRUE;
   END_TRANSITION
   STEP ok_1:   // S329, max time T#10S, warning time T#7S
      interlock C := "AutoProcessData".C_Glue.PartStatus = 380;
      (C)     N    "AutoProcessData".C_Glue.PartStatus:=399
   END_STEP
   TRANSITION Trans327 FROM ok_1 TO Step315   // T336
      := #ok_1.T > t#200MS;
   END_TRANSITION

   // sequencer 7: S400-S499 RobotGluePick
   STEP RobotGluePick:   // S400, max time T#10S, warning time T#7S
   END_STEP
   TRANSITION Trans92 FROM RobotGluePick TO ServoHomePos_6   // T400
      := TRUE;
   END_TRANSITION
   STEP "C-LocationCylinderToWP_1":   // S120, max time T#10S, warning time T#7S
              R    "ST10Cylinder".Cy[9].Inout.AutoGoHome
              S    "ST10Cylinder".Cy[9].Inout.AutoGoWork
   END_STEP
   TRANSITION Trans768 FROM "C-LocationCylinderToWP_1" TO CheckAxisXPos   // T121
      := "ST10Cylinder".Cy[9].In.WorkPositionSensor AND NOT "ST10Cylinder".Cy[9].In.HomePositionSensor;
   END_TRANSITION
   STEP RequestRobotGluePick:   // S282, max time T#10S, warning time T#7S
              N    "AutoProcessControl".C_Glue.Robot2PickPrimit
   END_STEP
   TRANSITION Trans93 FROM RequestRobotGluePick TO WaitRobotFinishTask_2   // T282
      := "KukaRobot2_CtrlDB".sROBtoPLC.User.Cycle.DO269_GluePickInside AND NOT "KukaRobot2_CtrlDB".sROBtoPLC.User.Cycle.DO270_GluePickFinish;
   END_TRANSITION
   STEP Axis_XYToHomePos_1:   // S86, max time T#10S, warning time T#7S
      interlock C := NOT "IAI_DeviceCtl".IAIServo[#X_Axis].Point[1].Achieve;
      (C)     N    "IAI_DeviceCtl".IAIServo[#X_Axis].Point[1].Start
   END_STEP
   TRANSITION Trans103 FROM Axis_XYToHomePos_1 TO Axis_ZToHomePos_1   // T96
      := "IAI_DeviceCtl".IAIServo[#X_Axis].Point[1].Achieve;
   END_TRANSITION
   STEP Step87:   // S87, max time T#10S, warning time T#7S
   END_STEP
   STEP "CheckServo returns toHome Pos_5":   // S99, max time T#10S, warning time T#7S
   END_STEP
   TRANSITION Trans119 FROM "CheckServo returns toHome Pos_5" TO "C-LocationCylinderToWP_1"   // T112
      := "ServoV90_DeviceCtl".V90Servo[3].Point[1].Achieve;
   END_TRANSITION
   STEP WaitRobotFinishTask_2:   // S289, max time T#10S, warning time T#7S
   END_STEP
   TRANSITION Trans94 FROM WaitRobotFinishTask_2 TO Step87   // T289
      := "KukaRobot2_CtrlDB".sROBtoPLC.User.Cycle.DO270_GluePickFinish;
   END_TRANSITION
   STEP "Process  Finish":   // S290, max time T#10S, warning time T#7S
              S    #ioPM_Inface.ProcessComplete
              R    #ioPM_Inface.ProcessStart
   END_STEP
   TRANSITION Trans290 FROM "Process  Finish" TO ProcessStart   // T290, jump
      := TRUE;
   END_TRANSITION
   STEP CheckAxisXPos:   // S147, max time T#10S, warning time T#7S
   END_STEP
   TRANSITION Trans159 FROM CheckAxisXPos TO RequestRobotGluePick   // T156
      := "IAI_DeviceCtl".IAIServo[#X_Axis].Point[1].Achieve;
   END_TRANSITION
   STEP ServoHomePos_6:   // S144, max time T#10S, warning time T#7S
          S1  S    "ServoV90_A3".IO.ioAutoHome
   END_STEP
   TRANSITION Trans157 FROM ServoHomePos_6 TO Step145   // T154
      := ("ServoV90_A3".Out.oActPosition >= (-5)) AND ("ServoV90_A3".Out.oActPosition <= 5);
   END_TRANSITION
   STEP Step145:   // S145, max time T#10S, warning time T#7S
   END_STEP
   TRANSITION Trans158 FROM Step145 TO ("CheckServo returns toHome Pos_5", Step160)   // T155
      := TRUE;
   END_TRANSITION
   STEP Step146:   // S146, max time T#10S, warning time T#7S
   END_STEP
   STEP Axis_ZToHomePos_1:   // S80, max time T#10S, warning time T#7S
      interlock C := NOT "IAI_DeviceCtl".IAIServo[#Z_Axis].Point[1].Achieve;
      (C)     N    "IAI_DeviceCtl".IAIServo[#Z_Axis].Point[1].Start
   END_STEP
   TRANSITION Trans100 FROM Axis_ZToHomePos_1 TO Step146   // T89
      := "IAI_DeviceCtl".IAIServo[#Z_Axis].Point[1].Achieve;
   END_TRANSITION
   STEP Step160:   // S160, max time T#10S, warning time T#7S
   END_STEP
   TRANSITION Trans168 FROM Step160 TO (Axis_XYToHomePos_1, Axis_XYToHomePos_2)   // T164
      := TRUE;
   END_TRANSITION
   STEP Step161:   // S161, max time T#10S, warning time T#7S
   END_STEP
   TRANSITION Trans104 FROM (Step87, Step146, Step161) TO "Process  Finish"   // T97
      := TRUE;
   END_TRANSITION
   STEP Axis_XYToHomePos_2:   // S156, max time T#10S, warning time T#7S
      interlock C := NOT "IAI_DeviceCtl".IAIServo[#Y_axis].Point[1].Achieve;
      (C)     N    "IAI_DeviceCtl".IAIServo[#Y_axis].Point[1].Start
   END_STEP
   TRANSITION Trans169 FROM Axis_XYToHomePos_2 TO Step161   // T165
      := "IAI_DeviceCtl".IAIServo[#Y_axis].Point[1].Achieve;
   END_TRANSITION

   // permanent post-instructions
   NETWORK 1
      #ioPM_Inface.StepNum := #RT_DATA.S_DISPLAY;
   NETWORK 2
      IF #iSysInface.Reset THEN #AlarmID := 0; END_IF;
   NETWORK 3
      #TON[10].TON(IN := #工件放行中, PT := T#0.5S);
      IF #TON[10].Q THEN #工件放行中 := FALSE; END_IF;
END_FUNCTION_BLOCK

FUNCTION_BLOCK "ST10_Flow8_FRobot_2"   // FB1078, GRAPH
// stored: AcknowledgeErrorsRequired false, AutoNumber false, GraphVersion 6.0, InitialValuesAcquisition false, SetENOAutomatically false
   // inherited from GRAPH_BASE
   VAR_INPUT
      INIT_SQ { ExternalAccessible := 'False'; ExternalVisible := 'False'; ExternalWritable := 'False'} : Bool := false;   // Set sequence to initial state
      iSysInface : "RCS_SysComInterface_V1";
   END_VAR
   VAR_IN_OUT
      ioPM_Inface : "RCS_PMInterface_V1";
      ioStatus : Int;
      Auto_Run_after_NG_box_closed : Bool;
   END_VAR
   VAR
      sCtrlMode { S7_SetPoint := 'True'} : "SysFlowCtrlGraph";
      sUpdMES_Data : Bool;   // 更新MES数据
      工件放行中 : Bool;
      前站站号 { ExternalAccessible := 'False'; ExternalVisible := 'False'; ExternalWritable := 'False'} : UInt;
      本站站号 { ExternalAccessible := 'False'; ExternalVisible := 'False'; ExternalWritable := 'False'} : UInt;
      弹窗Temp : Array[1..10] of Int;
      AlarmID : Int;
      TON { S7_SetPoint := 'True'} : Array[0..10] of TON_TIME;
      TOF { S7_SetPoint := 'True'} : Array[0..10] of TOF_TIME;
      sUP { S7_SetPoint := 'True'} : Array[0..10] of Bool;
      更新RFID完成 : Bool;
   END_VAR
   VAR_TEMP
      Tempresult : USInt;
      本站站号乘10 : UInt;
   END_VAR
   VAR CONSTANT
      Gripper_empty : Int := 0;
      "Gripper_have_OK_part_NO-MES" : Int := 199;
      Gripper_have_OK_part : Int := 110;
      Gripper_have_uknown_part : Int := 100;
      Gripper_Product_DMC_not_readable : Int := 155;
   END_VAR
   // // TON[0] : 托盘流入1托盘到位传感器
   // // TON[1] : 托盘流入1托盘到位传感器
   // // TON[2] : 托盘流入1产品有无传感器
   // // TON[3] : 托盘流入1产品有无传感器
   // // TON[4] : 托盘流入1姿态检测光电2
   // // TON[5] : 托盘流入1姿态检测光电3
   // // TON[0].Q : 托盘流入1托盘到位
   // // TON[1].Q : 托盘流入1托盘无
   // // TON[2].Q : 托盘流入1有产品
   // // TON[3].Q : 托盘流入1无产品
   // // TON[4].Q : 托盘流入1姿态检测光电2
   // // TON[5].Q : 托盘流入1姿态检测光电3
BEGIN
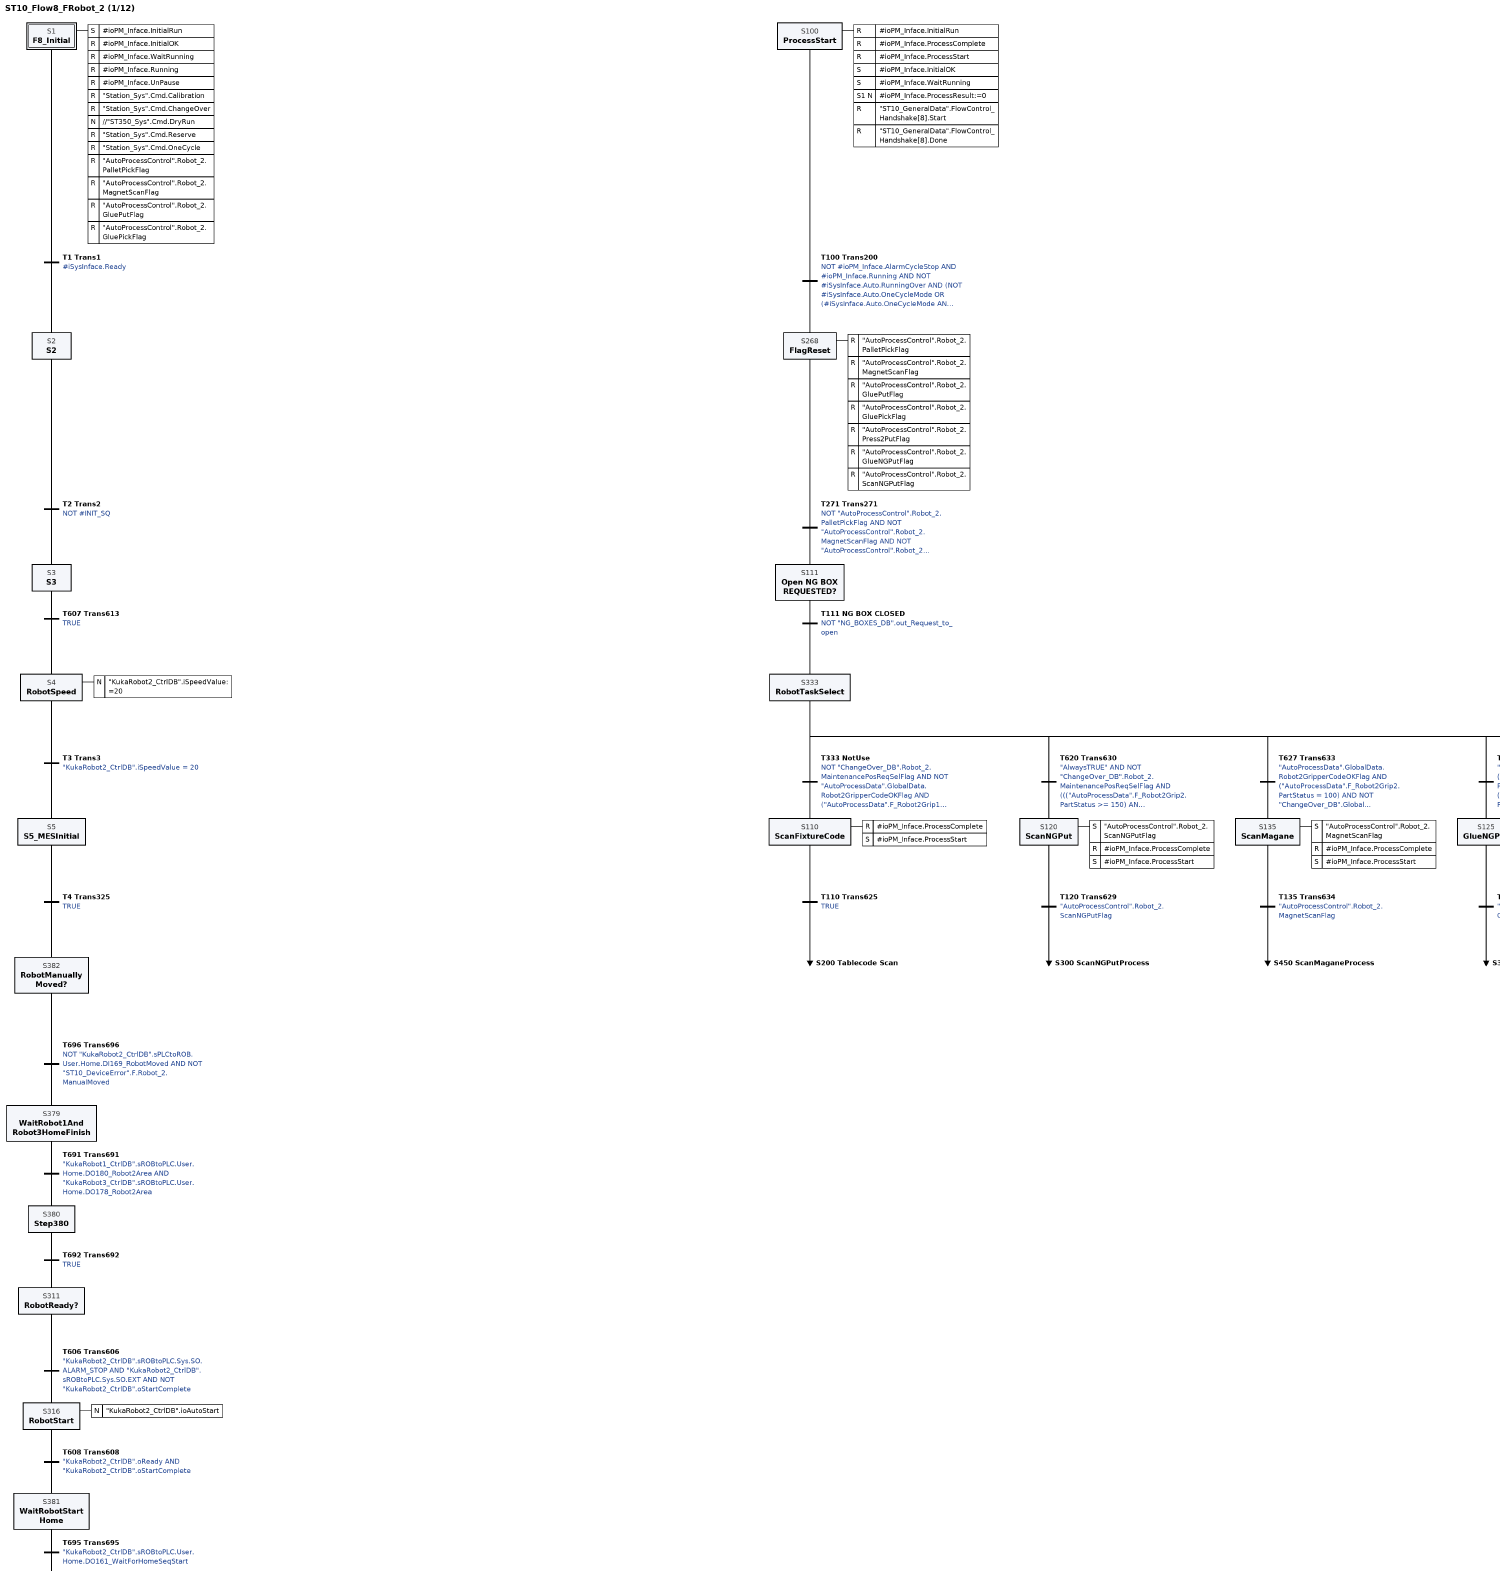
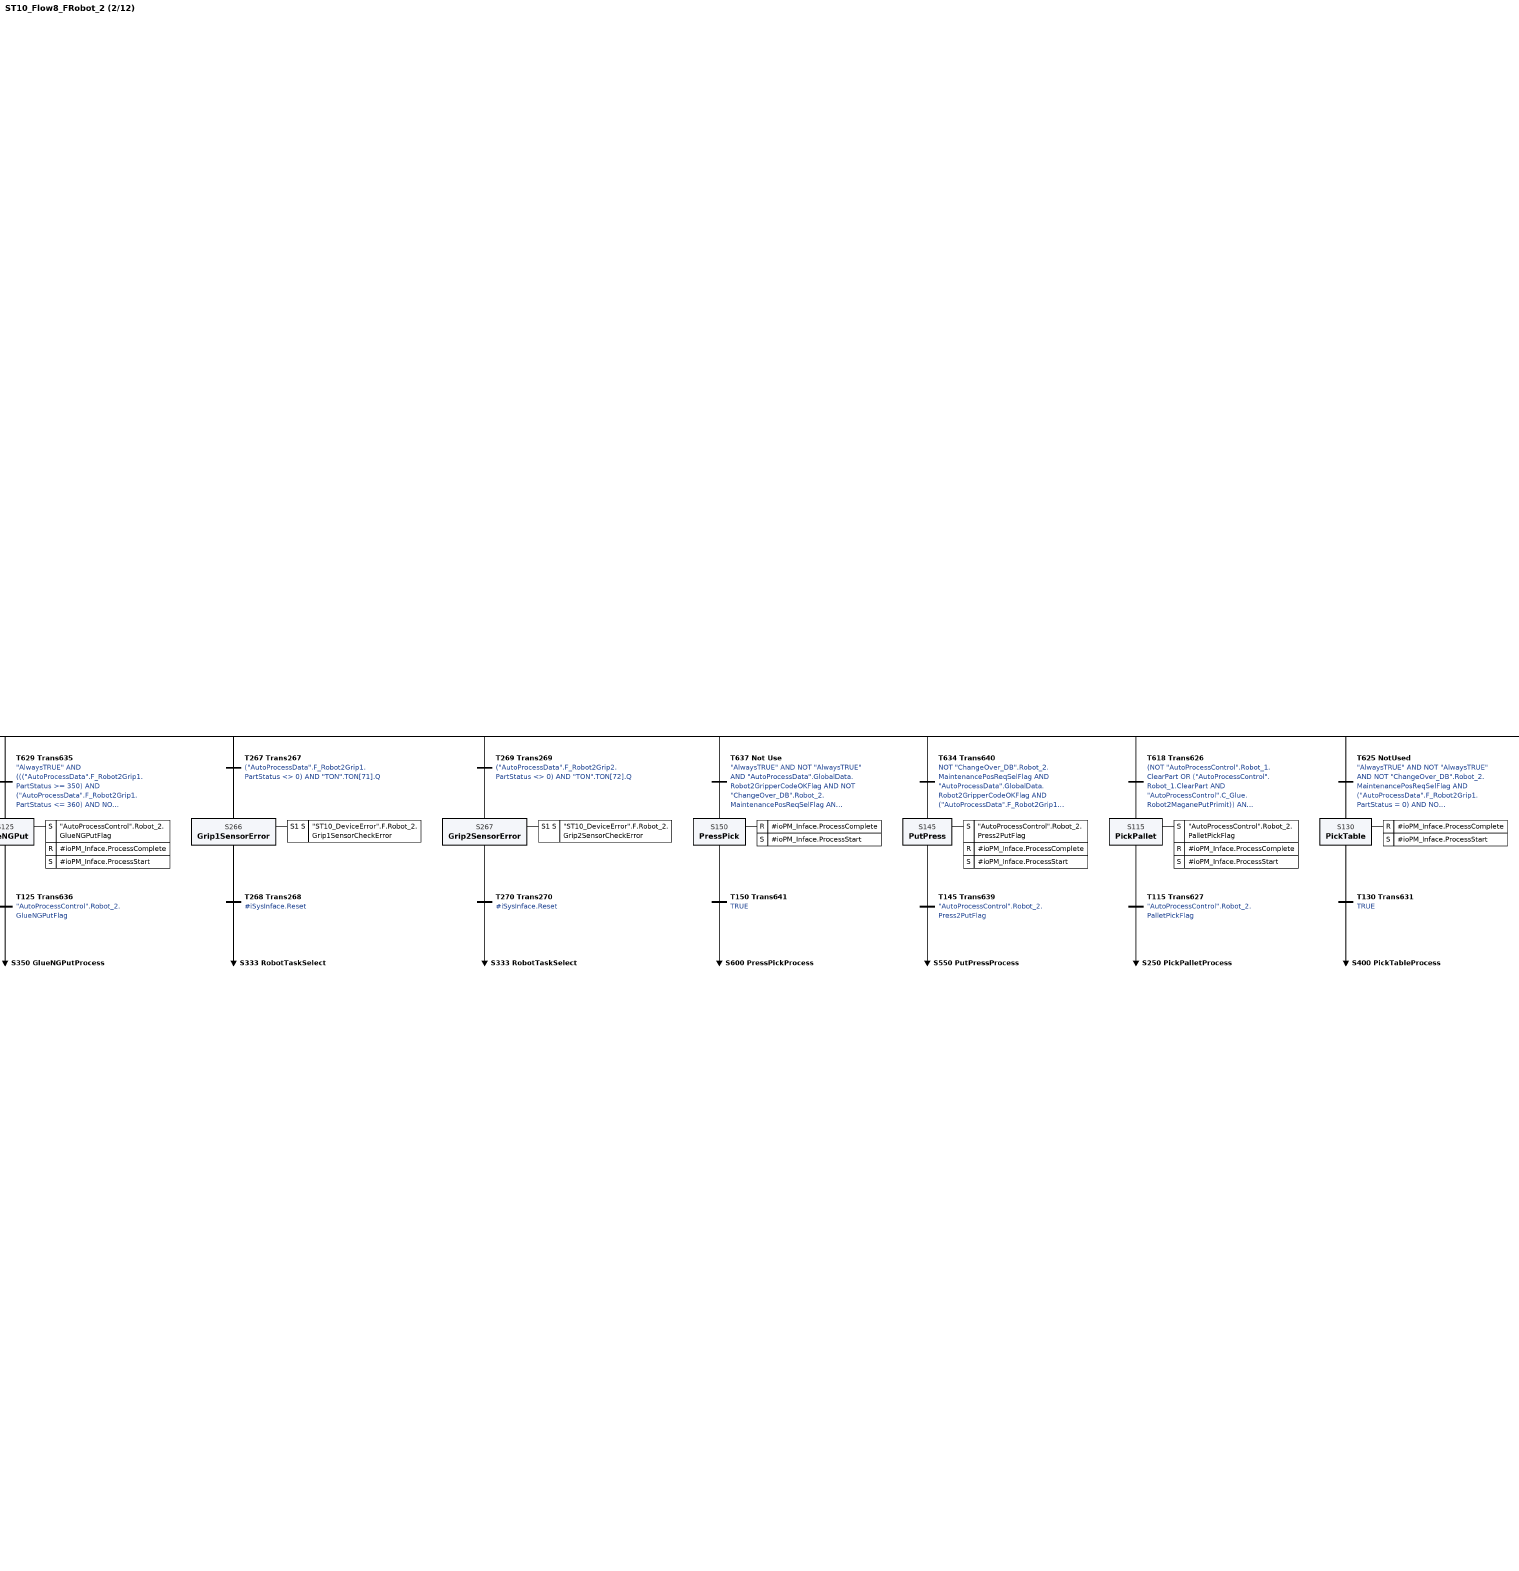
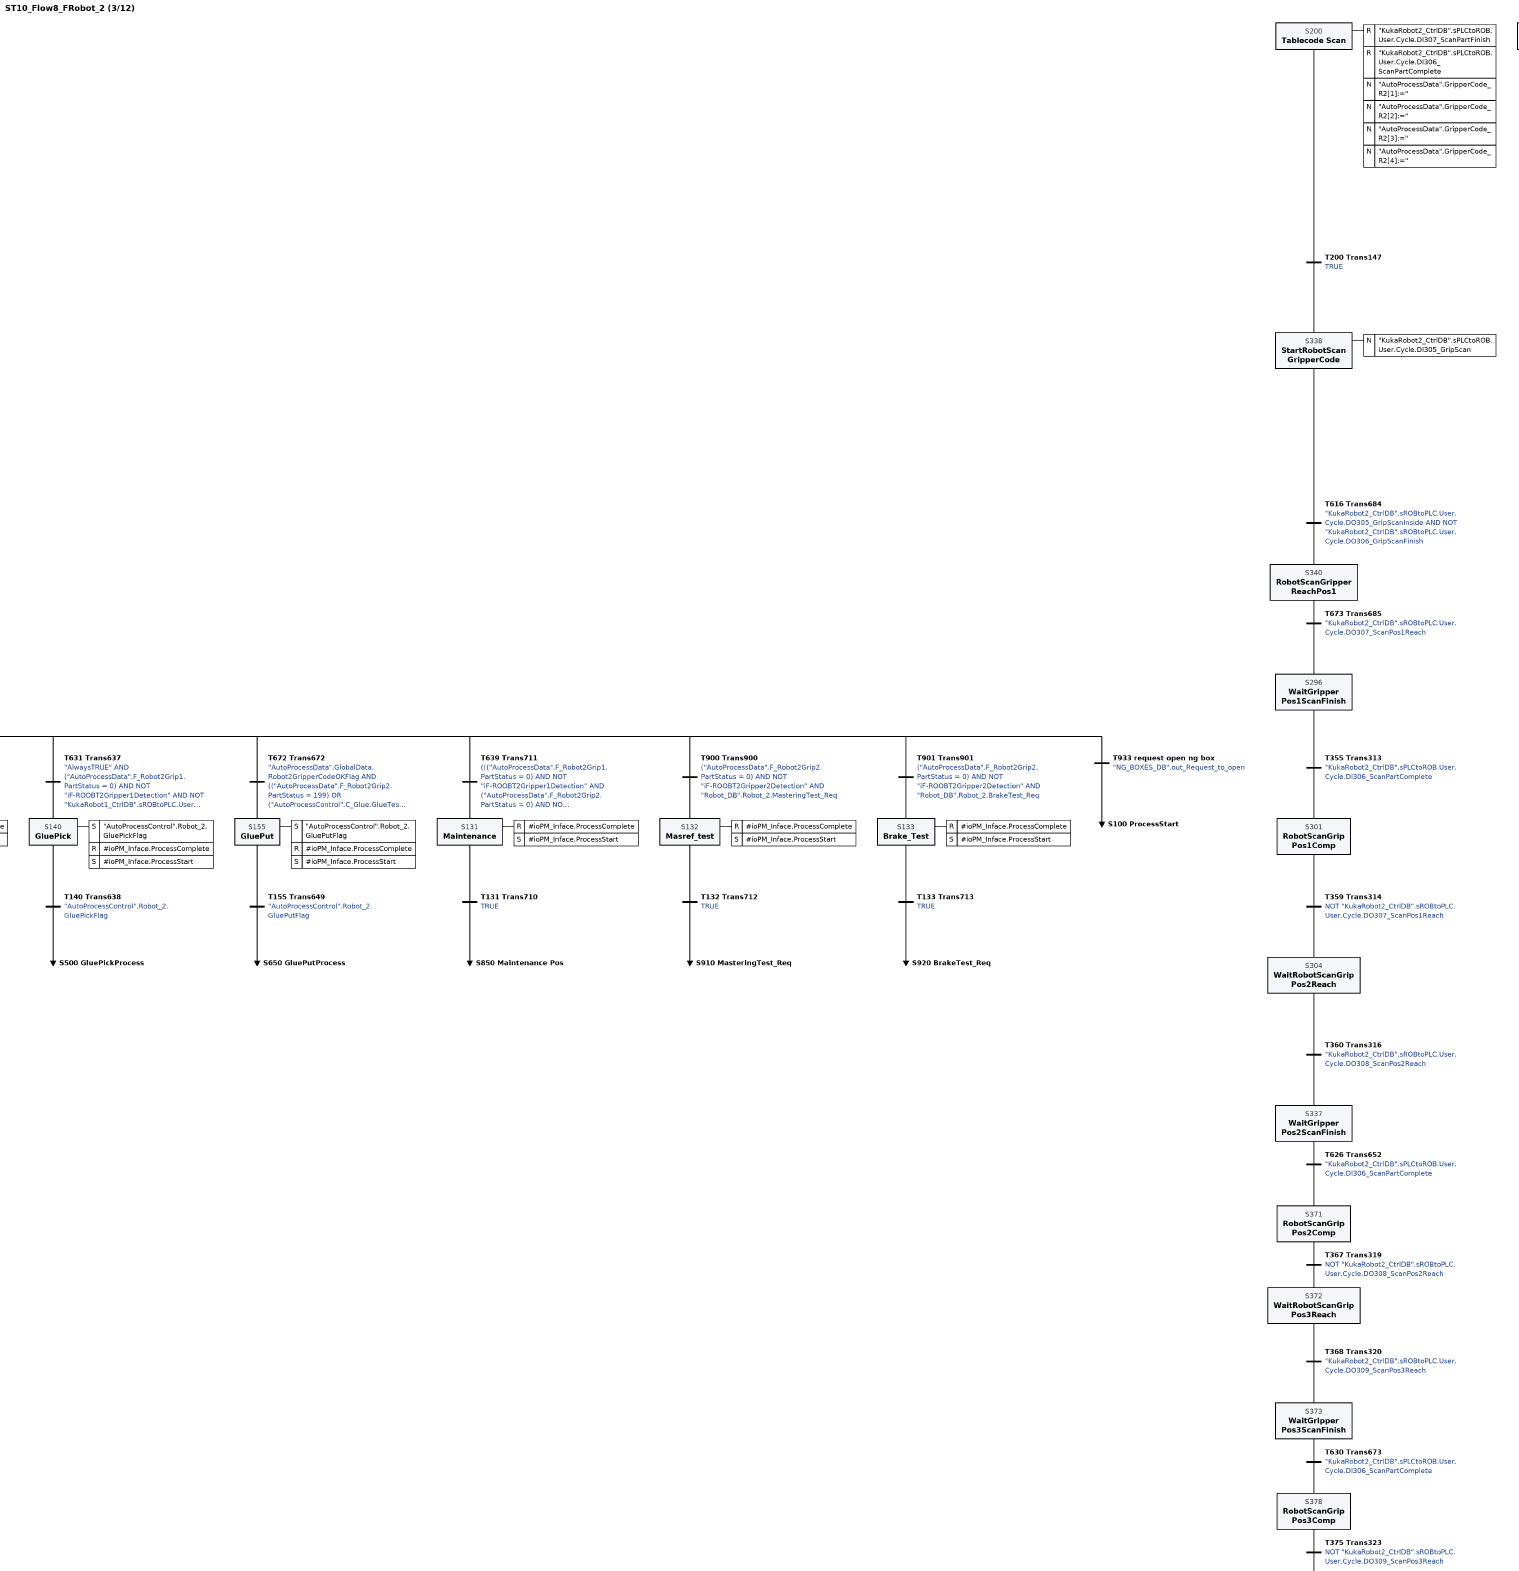
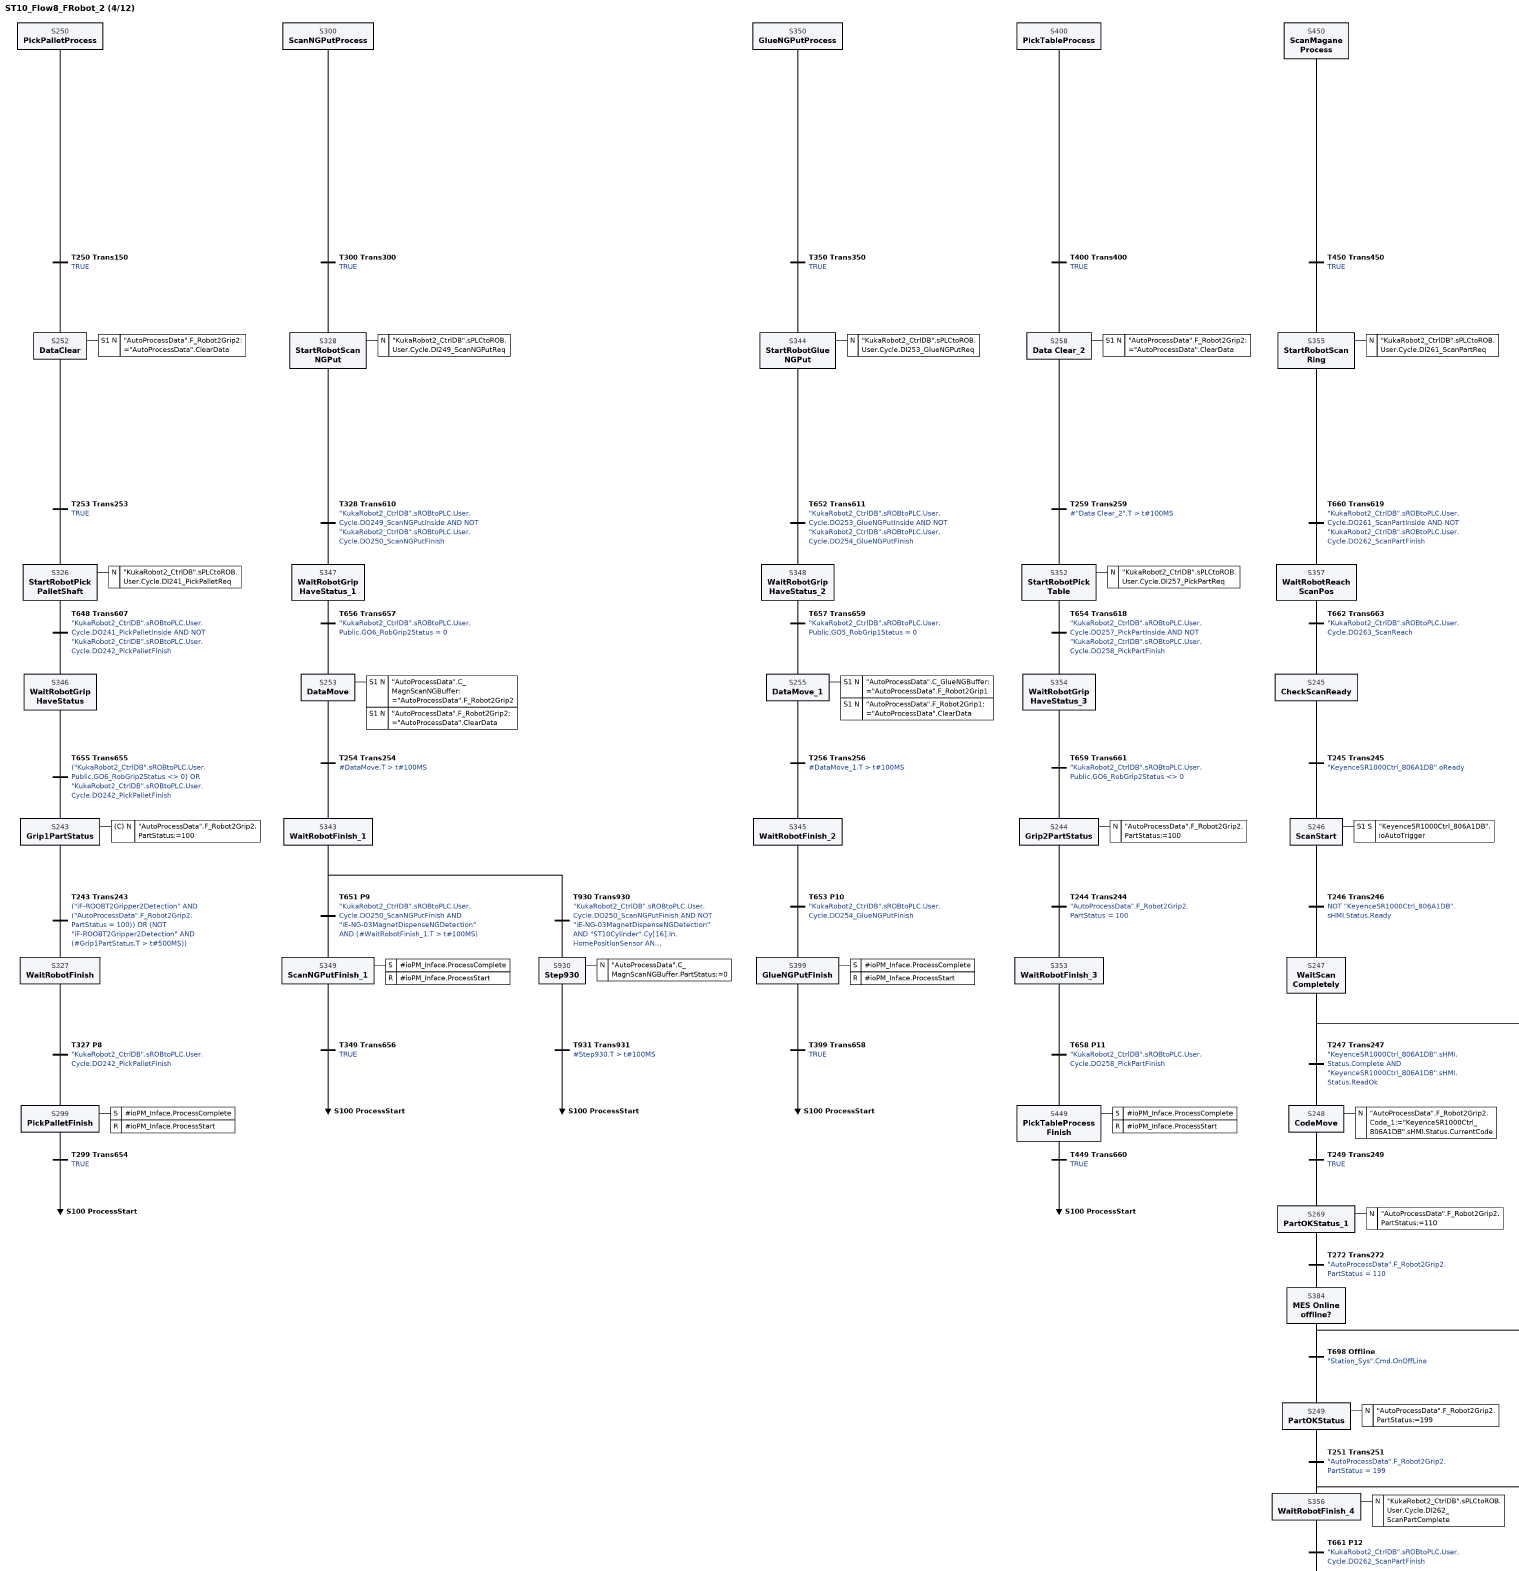
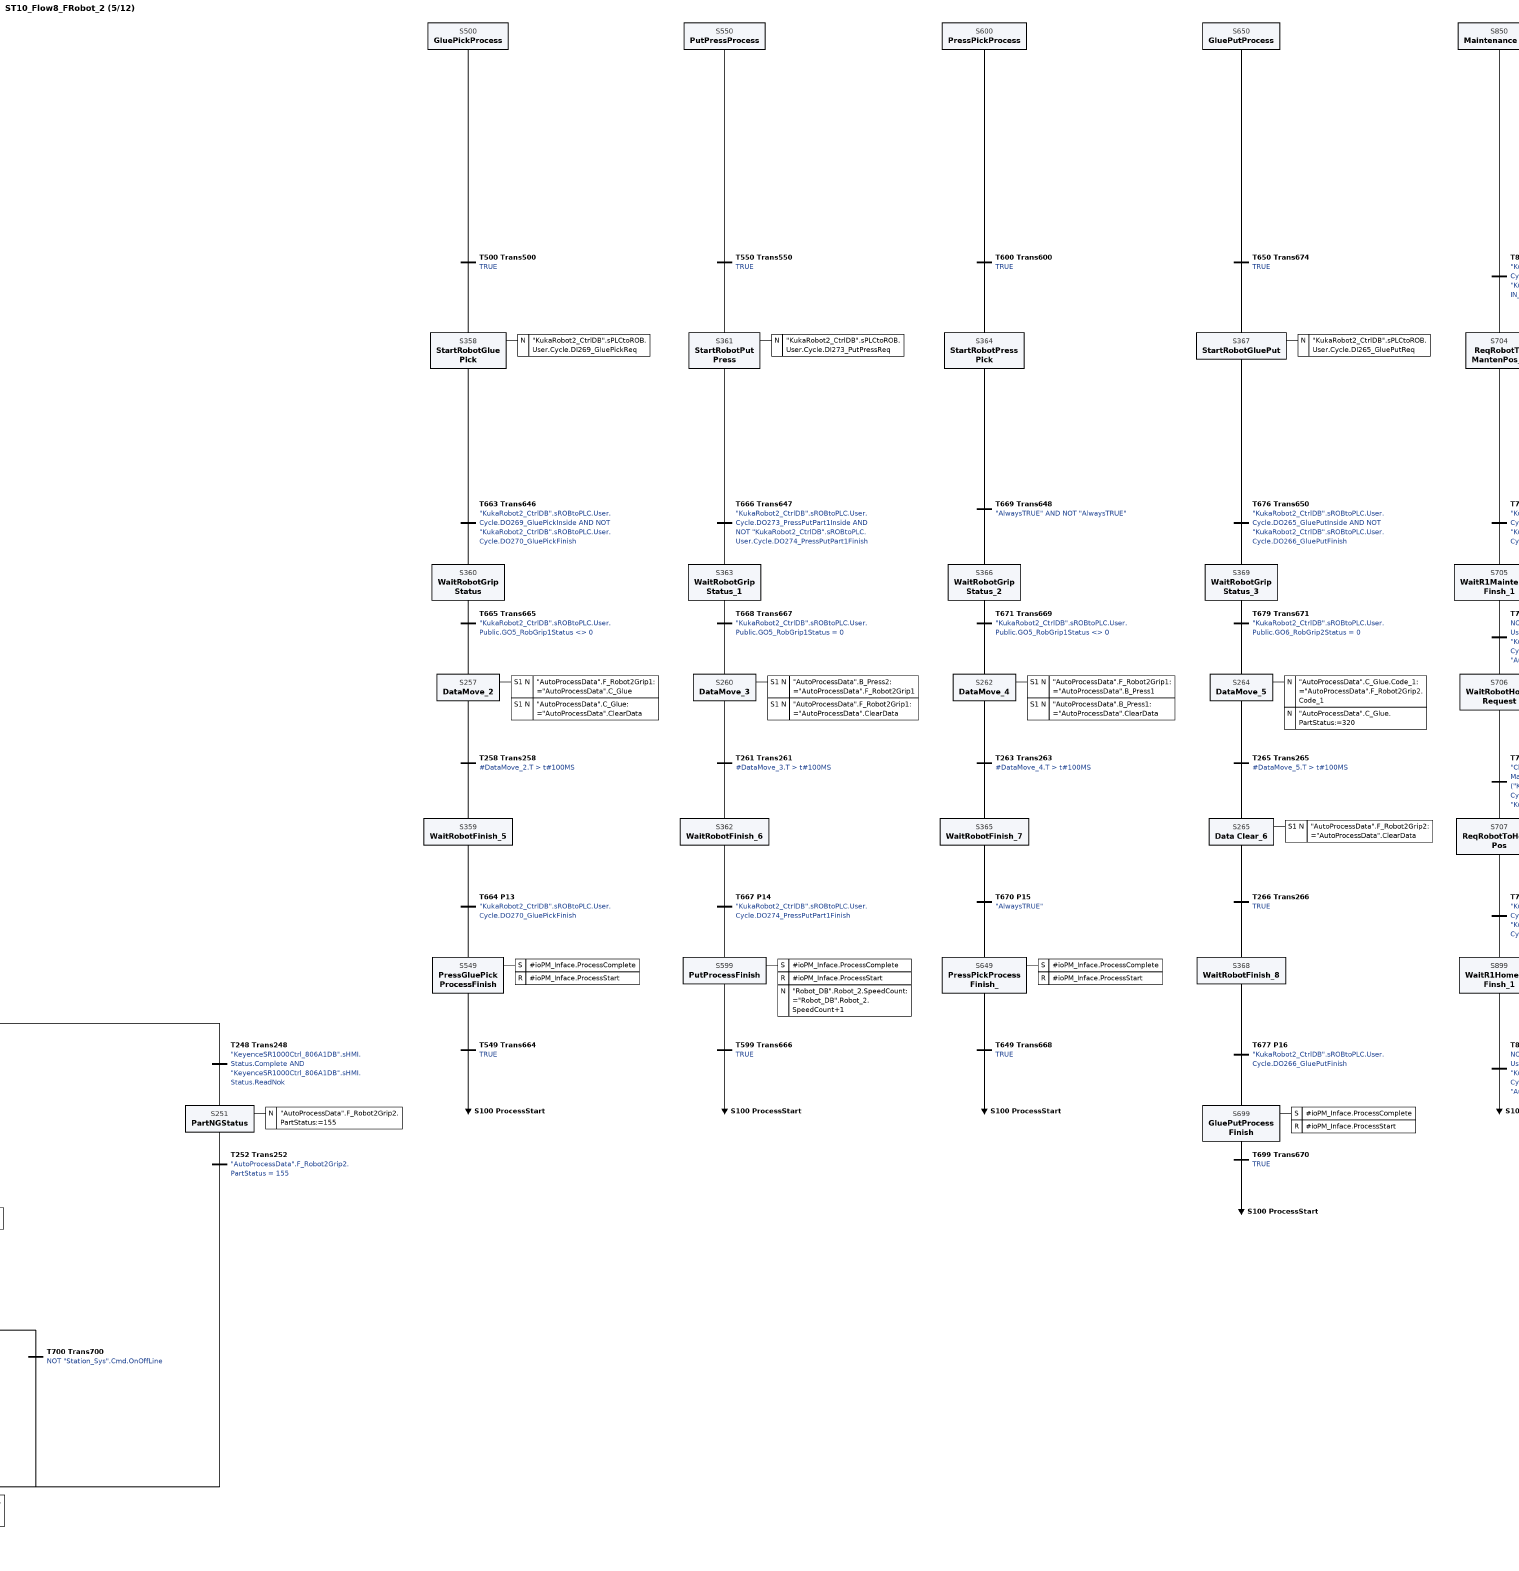
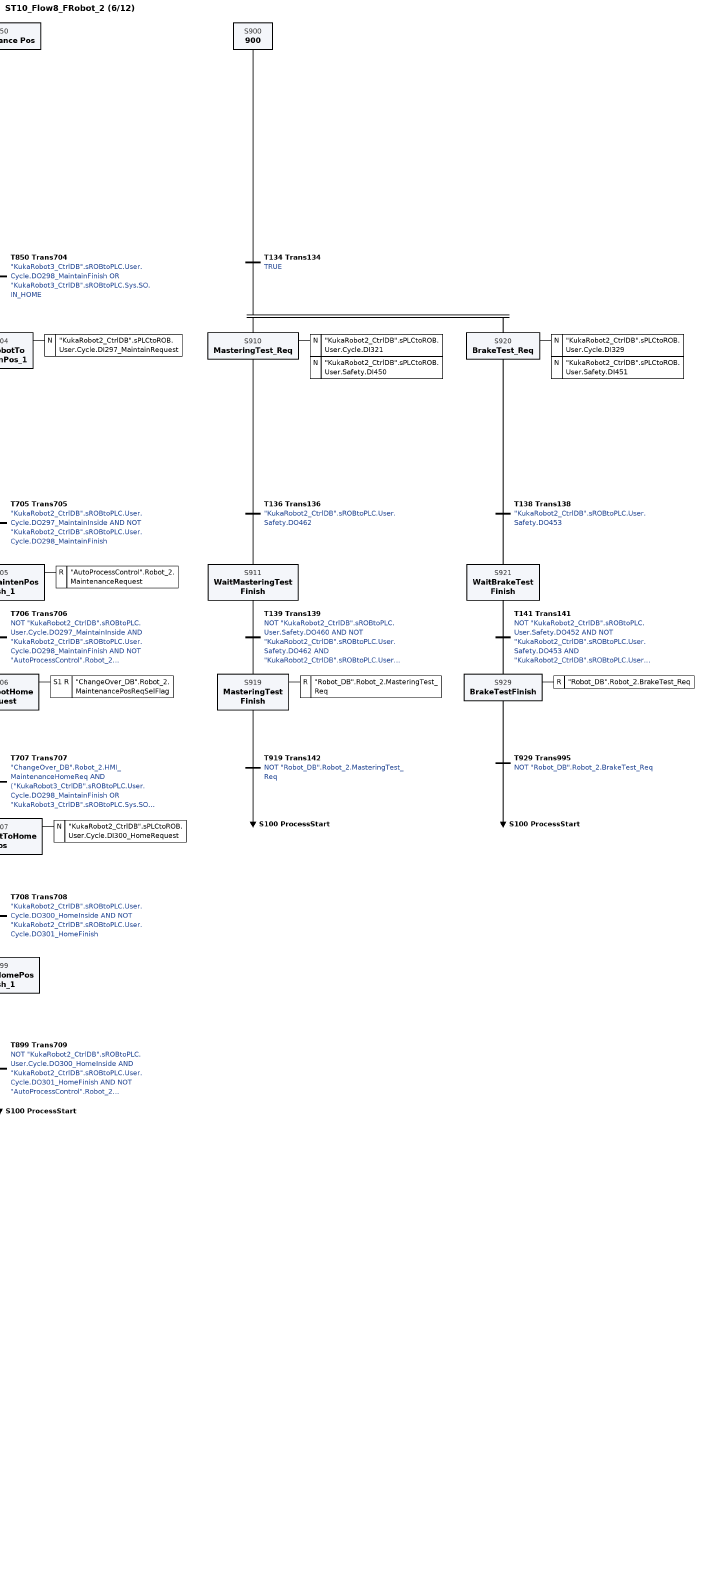
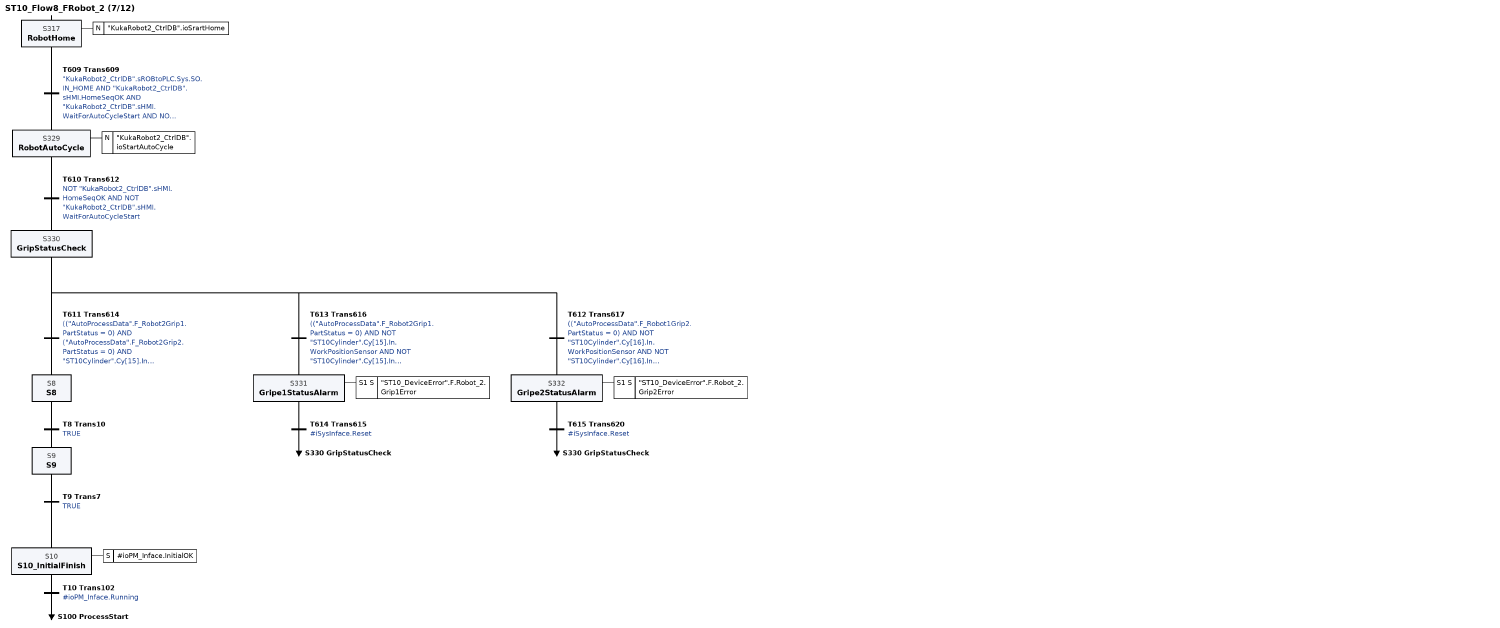
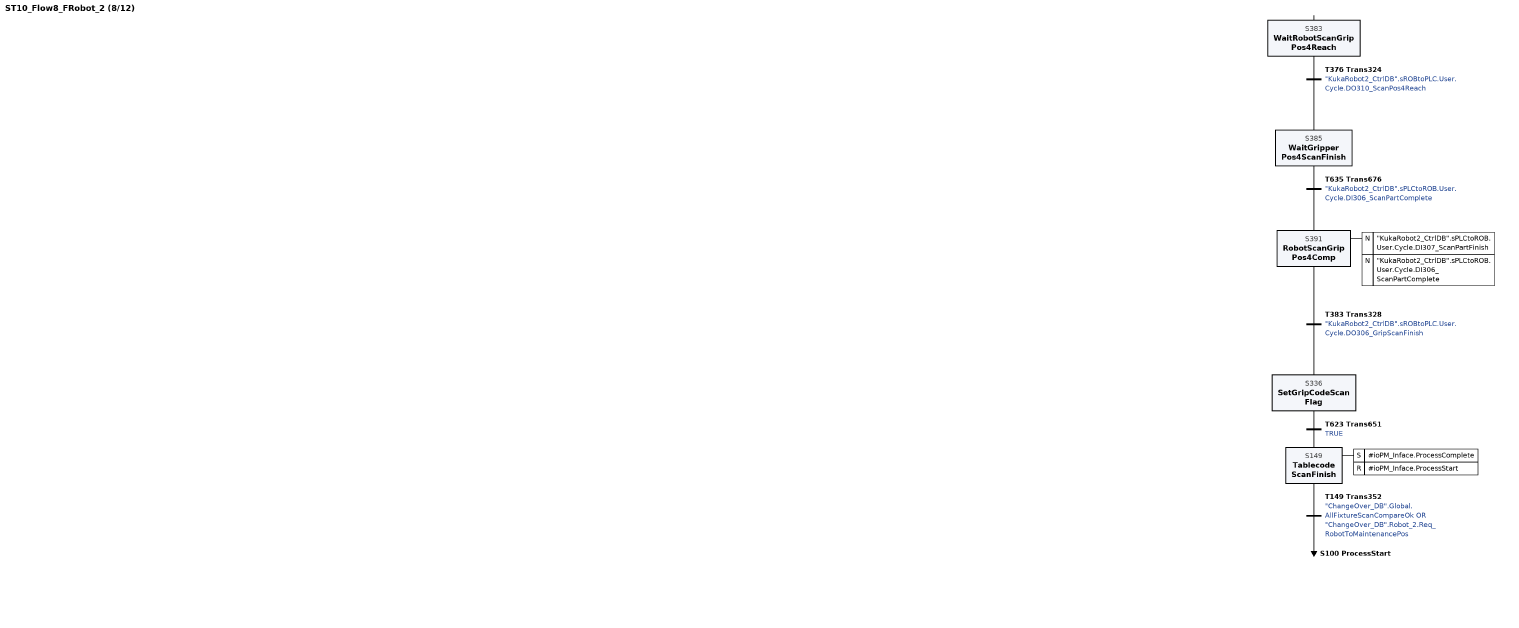
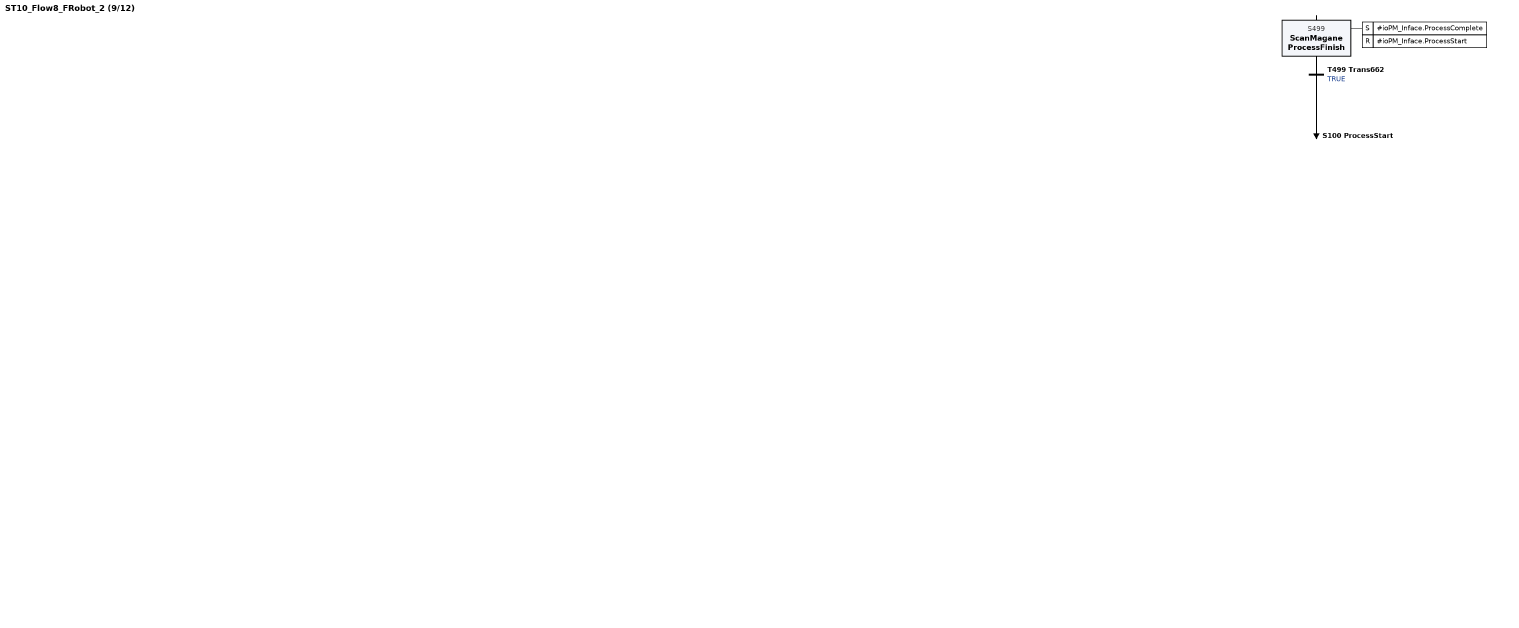
   // permanent pre-instructions
   NETWORK 1
      #TON[10].TON(IN := "AlwaysTRUE" AND "Station_Sys".Alarm.ImmediatelyStop, PT := T#300ms);
      #ioPM_Inface.AlarmImdilyStop := #TON[10].Q;
      #ioPM_Inface.AlarmCycleStop := "AlwaysTRUE" AND "Station_Sys".Alarm.CycleStop;
   NETWORK 2
      IF NOT False THEN
          #sCtrlMode(INIT := #INIT_SQ,   // "SysFlowCtrlGraph"
                     iSysInface := #iSysInface,
                     ioPM_Inface := #ioPM_Inface,
                     ioGraphCtrl := #RT_DATA.MOP);
      END_IF;
   NETWORK 3
      #TON[0].TON(IN := "AlwaysTRUE" AND "iA-Rotating product Check", PT := t#500ms);   // 工位11有托盘
      #TON[1].TOF(IN := "AlwaysTRUE" AND NOT "iA-Rotating product Check", PT := T#300ms);   // 工位无托盘
      #TON[2].TON(IN := "AlwaysTRUE", PT := T#300ms);
      #TON[3].TON(IN := "AlwaysTRUE", PT := T#300ms);
      #TON[4].TON(IN := "AlwaysTRUE", PT := T#300ms);
      #TON[5].TON(IN := "AlwaysTRUE", PT := T#300ms);
   NETWORK 4
      #前站站号 := 345;
      #本站站号 := 350;

